REGION Network 78: ERROR - Descarga por S3
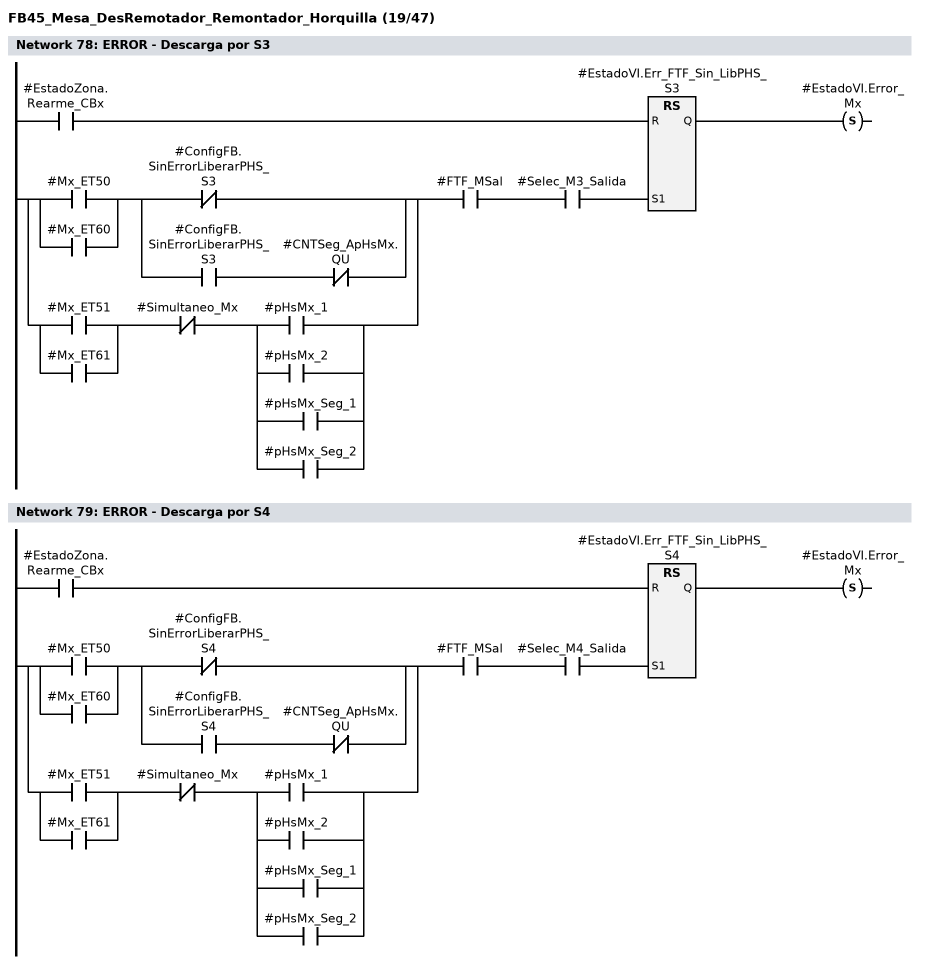
   RUNG wire#powerrail
      Contact( #EstadoZona.Rearme_CBx )
      S_RS(operand := #EstadoVI.Err_FTF_Sin_LibPHS_S3, s1 := wire#w5)
      S_Coil( #EstadoVI.Error_Mx )
   END_RUNG
   RUNG wire#powerrail
      Contact( #Mx_ET50 )
      wire#w1
      I_Contact( #ConfigFB.SinErrorLiberarPHS_S3 )
      wire#w2
      Contact( #FTF_MSal )
      Contact( #Selec_M3_Salida )
   END_RUNG wire#w5
   RUNG wire#powerrail
      Contact( #Mx_ET60 )
   END_RUNG wire#w1
   RUNG wire#w1
      Contact( #ConfigFB.SinErrorLiberarPHS_S3 )
      I_Contact( #CNTSeg_ApHsMx.QU )
   END_RUNG wire#w2
   RUNG wire#powerrail
      Contact( #Mx_ET51 )
      wire#w3
      I_Contact( #Simultaneo_Mx )
      wire#w4
      Contact( #pHsMx_1 )
   END_RUNG wire#w2
   RUNG wire#powerrail
      Contact( #Mx_ET61 )
   END_RUNG wire#w3
   RUNG wire#w4
      Contact( #pHsMx_2 )
   END_RUNG wire#w2
   RUNG wire#w4
      Contact( #pHsMx_Seg_1 )
   END_RUNG wire#w2
   RUNG wire#w4
      Contact( #pHsMx_Seg_2 )
   END_RUNG wire#w2
   // the same network as SCL:
   IF #EstadoZona.Rearme_CBx THEN
       #EstadoVI.Err_FTF_Sin_LibPHS_S3 := FALSE;   // RS flip-flop
   END_IF;
   IF (((#Mx_ET50 OR #Mx_ET60) AND (NOT #ConfigFB.SinErrorLiberarPHS_S3 OR (#ConfigFB.SinErrorLiberarPHS_S3 AND NOT #CNTSeg_ApHsMx.QU))) OR ((#Mx_ET51 OR #Mx_ET61) AND NOT #Simultaneo_Mx AND (#pHsMx_1 OR #pHsMx_2 OR #pHsMx_Seg_1 OR #pHsMx_Seg_2))) AND #FTF_MSal AND #Selec_M3_Salida THEN
       #EstadoVI.Err_FTF_Sin_LibPHS_S3 := TRUE;
   END_IF;
   IF #EstadoVI.Err_FTF_Sin_LibPHS_S3 THEN #EstadoVI.Error_Mx := TRUE; END_IF;
END_REGION

REGION Network 79: ERROR - Descarga por S4
   RUNG wire#powerrail
      Contact( #EstadoZona.Rearme_CBx )
      S_RS(operand := #EstadoVI.Err_FTF_Sin_LibPHS_S4, s1 := wire#w5)
      S_Coil( #EstadoVI.Error_Mx )
   END_RUNG
   RUNG wire#powerrail
      Contact( #Mx_ET50 )
      wire#w1
      I_Contact( #ConfigFB.SinErrorLiberarPHS_S4 )
      wire#w2
      Contact( #FTF_MSal )
      Contact( #Selec_M4_Salida )
   END_RUNG wire#w5
   RUNG wire#powerrail
      Contact( #Mx_ET60 )
   END_RUNG wire#w1
   RUNG wire#w1
      Contact( #ConfigFB.SinErrorLiberarPHS_S4 )
      I_Contact( #CNTSeg_ApHsMx.QU )
   END_RUNG wire#w2
   RUNG wire#powerrail
      Contact( #Mx_ET51 )
      wire#w3
      I_Contact( #Simultaneo_Mx )
      wire#w4
      Contact( #pHsMx_1 )
   END_RUNG wire#w2
   RUNG wire#powerrail
      Contact( #Mx_ET61 )
   END_RUNG wire#w3
   RUNG wire#w4
      Contact( #pHsMx_2 )
   END_RUNG wire#w2
   RUNG wire#w4
      Contact( #pHsMx_Seg_1 )
   END_RUNG wire#w2
   RUNG wire#w4
      Contact( #pHsMx_Seg_2 )
   END_RUNG wire#w2
   // the same network as SCL:
   IF #EstadoZona.Rearme_CBx THEN
       #EstadoVI.Err_FTF_Sin_LibPHS_S4 := FALSE;   // RS flip-flop
   END_IF;
   IF (((#Mx_ET50 OR #Mx_ET60) AND (NOT #ConfigFB.SinErrorLiberarPHS_S4 OR (#ConfigFB.SinErrorLiberarPHS_S4 AND NOT #CNTSeg_ApHsMx.QU))) OR ((#Mx_ET51 OR #Mx_ET61) AND NOT #Simultaneo_Mx AND (#pHsMx_1 OR #pHsMx_2 OR #pHsMx_Seg_1 OR #pHsMx_Seg_2))) AND #FTF_MSal AND #Selec_M4_Salida THEN
       #EstadoVI.Err_FTF_Sin_LibPHS_S4 := TRUE;
   END_IF;
   IF #EstadoVI.Err_FTF_Sin_LibPHS_S4 THEN #EstadoVI.Error_Mx := TRUE; END_IF;
END_REGION

REGION Network 80: TMP - ERROR - Tout Avance E1E3
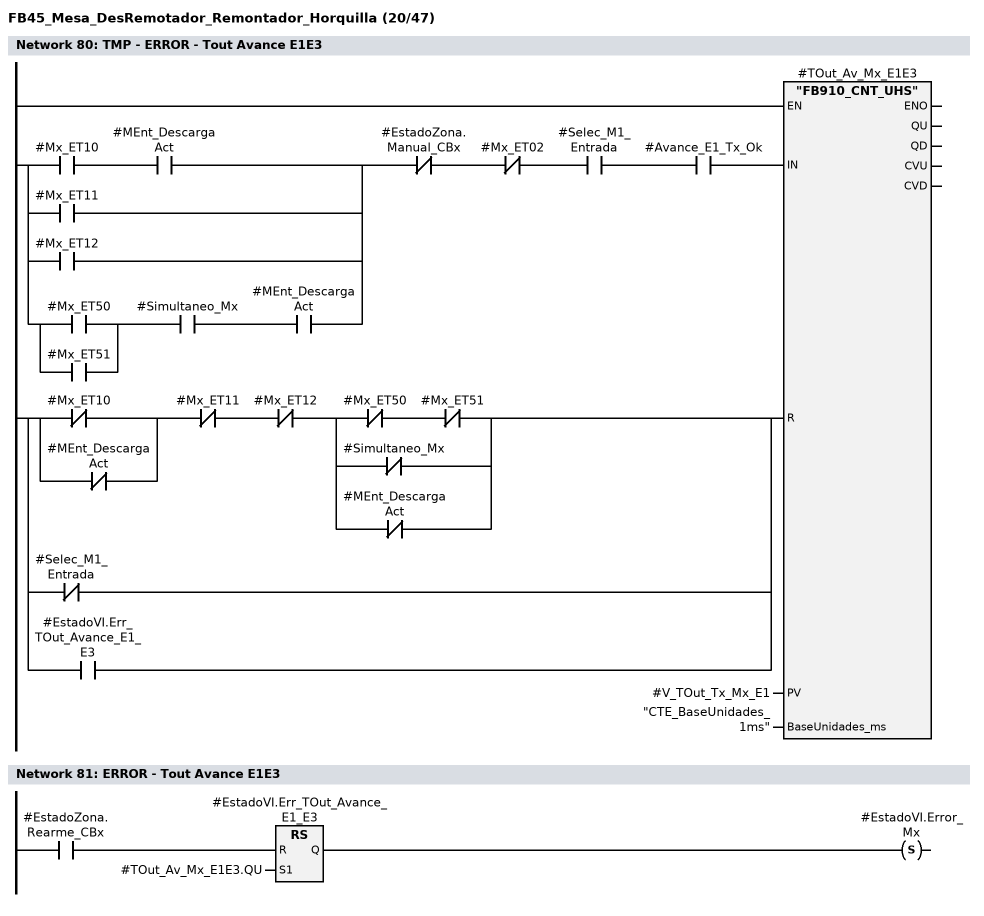
   RUNG wire#powerrail
      #TOut_Av_Mx_E1E3(IN := wire#w3, R := wire#w6, PV := #V_TOut_Tx_Mx_E1, BaseUnidades_ms := "CTE_BaseUnidades_1ms", QU =>, QD =>, CVU =>, CVD =>)
   END_RUNG
   RUNG wire#powerrail
      Contact( #Mx_ET10 )
      Contact( #MEnt_DescargaAct )
      wire#w1
      I_Contact( #EstadoZona.Manual_CBx )
      I_Contact( #Mx_ET02 )
      Contact( #Selec_M1_Entrada )
      Contact( #Avance_E1_Tx_Ok )
   END_RUNG wire#w3
   RUNG wire#powerrail
      Contact( #Mx_ET11 )
   END_RUNG wire#w1
   RUNG wire#powerrail
      Contact( #Mx_ET12 )
   END_RUNG wire#w1
   RUNG wire#powerrail
      Contact( #Mx_ET50 )
      wire#w2
      Contact( #Simultaneo_Mx )
      Contact( #MEnt_DescargaAct )
   END_RUNG wire#w1
   RUNG wire#powerrail
      Contact( #Mx_ET51 )
   END_RUNG wire#w2
   RUNG wire#powerrail
      I_Contact( #Mx_ET10 )
      wire#w4
      I_Contact( #Mx_ET11 )
      I_Contact( #Mx_ET12 )
      wire#w5
      I_Contact( #Mx_ET50 )
      I_Contact( #Mx_ET51 )
   END_RUNG wire#w6
   RUNG wire#powerrail
      I_Contact( #MEnt_DescargaAct )
   END_RUNG wire#w4
   RUNG wire#w5
      I_Contact( #Simultaneo_Mx )
   END_RUNG wire#w6
   RUNG wire#w5
      I_Contact( #MEnt_DescargaAct )
   END_RUNG wire#w6
   RUNG wire#powerrail
      I_Contact( #Selec_M1_Entrada )
   END_RUNG wire#w6
   RUNG wire#powerrail
      Contact( #EstadoVI.Err_TOut_Avance_E1_E3 )
   END_RUNG wire#w6
   // the same network as SCL:
   #TOut_Av_Mx_E1E3(IN := ((#Mx_ET10 AND #MEnt_DescargaAct) OR #Mx_ET11 OR #Mx_ET12 OR ((#Mx_ET50 OR #Mx_ET51) AND #Simultaneo_Mx AND #MEnt_DescargaAct)) AND NOT #EstadoZona.Manual_CBx AND NOT #Mx_ET02 AND #Selec_M1_Entrada AND #Avance_E1_Tx_Ok,   // "FB910_CNT_UHS"
                    R := ((NOT #Mx_ET10 OR NOT #MEnt_DescargaAct) AND NOT #Mx_ET11 AND NOT #Mx_ET12 AND ((NOT #Mx_ET50 AND NOT #Mx_ET51) OR NOT #Simultaneo_Mx OR NOT #MEnt_DescargaAct)) OR NOT #Selec_M1_Entrada OR #EstadoVI.Err_TOut_Avance_E1_E3,
                    PV := #V_TOut_Tx_Mx_E1,
                    BaseUnidades_ms := "CTE_BaseUnidades_1ms");
END_REGION

REGION Network 81: ERROR - Tout Avance E1E3
   RUNG wire#powerrail
      Contact( #EstadoZona.Rearme_CBx )
      S_RS(operand := #EstadoVI.Err_TOut_Avance_E1_E3, s1 := #TOut_Av_Mx_E1E3.QU)
      S_Coil( #EstadoVI.Error_Mx )
   END_RUNG
   // the same network as SCL:
   IF #EstadoZona.Rearme_CBx THEN
       #EstadoVI.Err_TOut_Avance_E1_E3 := FALSE;   // RS flip-flop
   END_IF;
   IF #TOut_Av_Mx_E1E3.QU THEN #EstadoVI.Err_TOut_Avance_E1_E3 := TRUE; END_IF;
   IF #EstadoVI.Err_TOut_Avance_E1_E3 THEN #EstadoVI.Error_Mx := TRUE; END_IF;
END_REGION

REGION Network 82: TMP - ERROR - Tout Retroceso E1E3
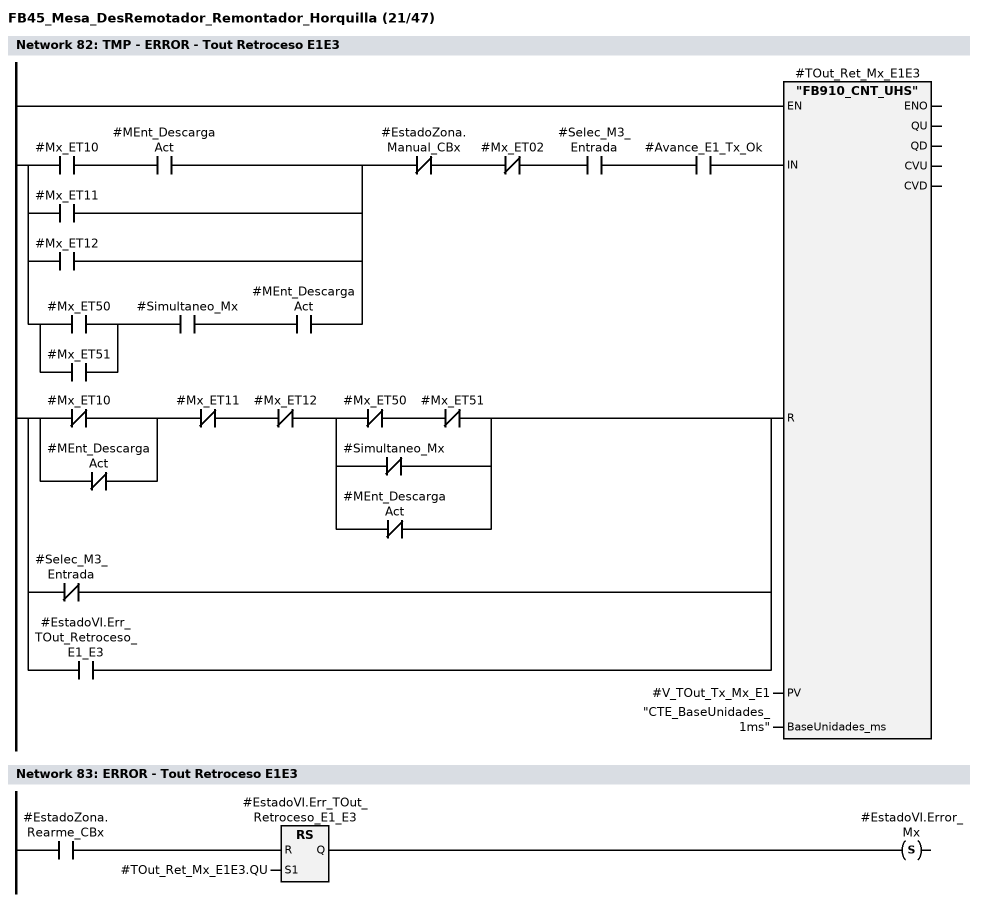
   RUNG wire#powerrail
      #TOut_Ret_Mx_E1E3(IN := wire#w3, R := wire#w6, PV := #V_TOut_Tx_Mx_E1, BaseUnidades_ms := "CTE_BaseUnidades_1ms", QU =>, QD =>, CVU =>, CVD =>)
   END_RUNG
   RUNG wire#powerrail
      Contact( #Mx_ET10 )
      Contact( #MEnt_DescargaAct )
      wire#w1
      I_Contact( #EstadoZona.Manual_CBx )
      I_Contact( #Mx_ET02 )
      Contact( #Selec_M3_Entrada )
      Contact( #Avance_E1_Tx_Ok )
   END_RUNG wire#w3
   RUNG wire#powerrail
      Contact( #Mx_ET11 )
   END_RUNG wire#w1
   RUNG wire#powerrail
      Contact( #Mx_ET12 )
   END_RUNG wire#w1
   RUNG wire#powerrail
      Contact( #Mx_ET50 )
      wire#w2
      Contact( #Simultaneo_Mx )
      Contact( #MEnt_DescargaAct )
   END_RUNG wire#w1
   RUNG wire#powerrail
      Contact( #Mx_ET51 )
   END_RUNG wire#w2
   RUNG wire#powerrail
      I_Contact( #Mx_ET10 )
      wire#w4
      I_Contact( #Mx_ET11 )
      I_Contact( #Mx_ET12 )
      wire#w5
      I_Contact( #Mx_ET50 )
      I_Contact( #Mx_ET51 )
   END_RUNG wire#w6
   RUNG wire#powerrail
      I_Contact( #MEnt_DescargaAct )
   END_RUNG wire#w4
   RUNG wire#w5
      I_Contact( #Simultaneo_Mx )
   END_RUNG wire#w6
   RUNG wire#w5
      I_Contact( #MEnt_DescargaAct )
   END_RUNG wire#w6
   RUNG wire#powerrail
      I_Contact( #Selec_M3_Entrada )
   END_RUNG wire#w6
   RUNG wire#powerrail
      Contact( #EstadoVI.Err_TOut_Retroceso_E1_E3 )
   END_RUNG wire#w6
   // the same network as SCL:
   #TOut_Ret_Mx_E1E3(IN := ((#Mx_ET10 AND #MEnt_DescargaAct) OR #Mx_ET11 OR #Mx_ET12 OR ((#Mx_ET50 OR #Mx_ET51) AND #Simultaneo_Mx AND #MEnt_DescargaAct)) AND NOT #EstadoZona.Manual_CBx AND NOT #Mx_ET02 AND #Selec_M3_Entrada AND #Avance_E1_Tx_Ok,   // "FB910_CNT_UHS"
                     R := ((NOT #Mx_ET10 OR NOT #MEnt_DescargaAct) AND NOT #Mx_ET11 AND NOT #Mx_ET12 AND ((NOT #Mx_ET50 AND NOT #Mx_ET51) OR NOT #Simultaneo_Mx OR NOT #MEnt_DescargaAct)) OR NOT #Selec_M3_Entrada OR #EstadoVI.Err_TOut_Retroceso_E1_E3,
                     PV := #V_TOut_Tx_Mx_E1,
                     BaseUnidades_ms := "CTE_BaseUnidades_1ms");
END_REGION

REGION Network 83: ERROR - Tout Retroceso E1E3
   RUNG wire#powerrail
      Contact( #EstadoZona.Rearme_CBx )
      S_RS(operand := #EstadoVI.Err_TOut_Retroceso_E1_E3, s1 := #TOut_Ret_Mx_E1E3.QU)
      S_Coil( #EstadoVI.Error_Mx )
   END_RUNG
   // the same network as SCL:
   IF #EstadoZona.Rearme_CBx THEN
       #EstadoVI.Err_TOut_Retroceso_E1_E3 := FALSE;   // RS flip-flop
   END_IF;
   IF #TOut_Ret_Mx_E1E3.QU THEN #EstadoVI.Err_TOut_Retroceso_E1_E3 := TRUE; END_IF;
   IF #EstadoVI.Err_TOut_Retroceso_E1_E3 THEN #EstadoVI.Error_Mx := TRUE; END_IF;
END_REGION

REGION Network 84: TMP - ERROR - Tout Avance E2E4
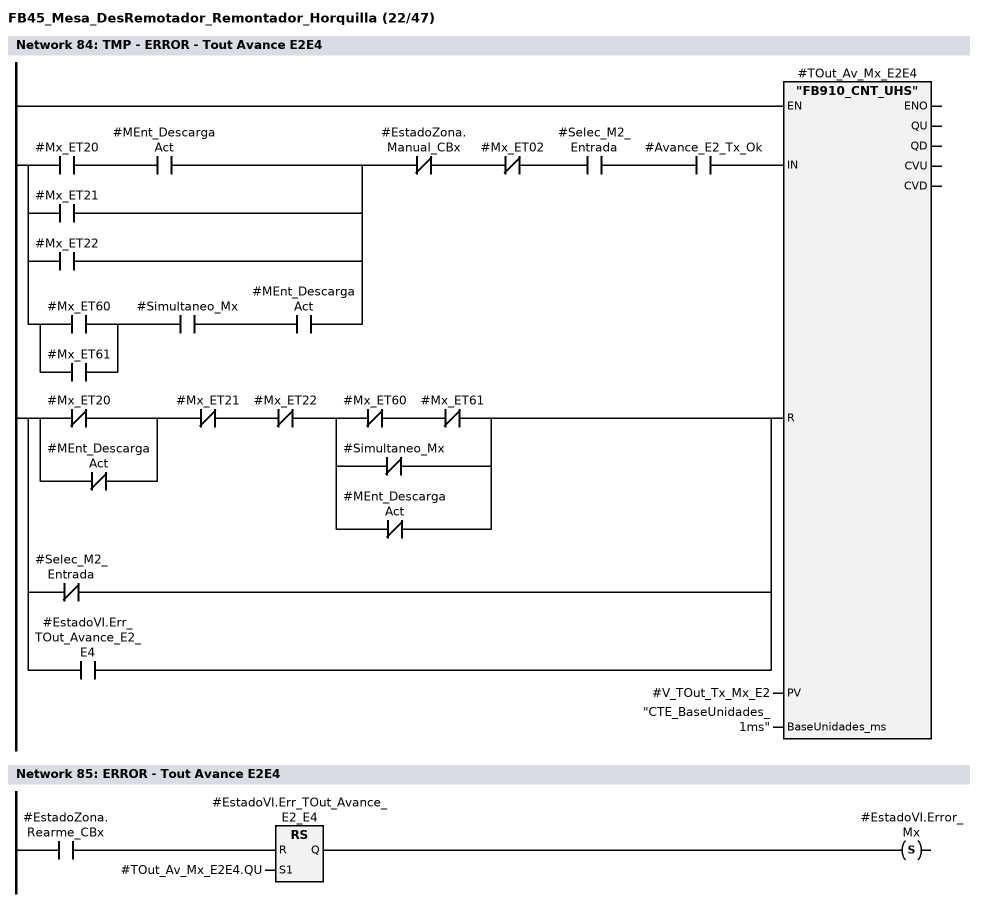
   RUNG wire#powerrail
      #TOut_Av_Mx_E2E4(IN := wire#w3, R := wire#w6, PV := #V_TOut_Tx_Mx_E2, BaseUnidades_ms := "CTE_BaseUnidades_1ms", QU =>, QD =>, CVU =>, CVD =>)
   END_RUNG
   RUNG wire#powerrail
      Contact( #Mx_ET20 )
      Contact( #MEnt_DescargaAct )
      wire#w1
      I_Contact( #EstadoZona.Manual_CBx )
      I_Contact( #Mx_ET02 )
      Contact( #Selec_M2_Entrada )
      Contact( #Avance_E2_Tx_Ok )
   END_RUNG wire#w3
   RUNG wire#powerrail
      Contact( #Mx_ET21 )
   END_RUNG wire#w1
   RUNG wire#powerrail
      Contact( #Mx_ET22 )
   END_RUNG wire#w1
   RUNG wire#powerrail
      Contact( #Mx_ET60 )
      wire#w2
      Contact( #Simultaneo_Mx )
      Contact( #MEnt_DescargaAct )
   END_RUNG wire#w1
   RUNG wire#powerrail
      Contact( #Mx_ET61 )
   END_RUNG wire#w2
   RUNG wire#powerrail
      I_Contact( #Mx_ET20 )
      wire#w4
      I_Contact( #Mx_ET21 )
      I_Contact( #Mx_ET22 )
      wire#w5
      I_Contact( #Mx_ET60 )
      I_Contact( #Mx_ET61 )
   END_RUNG wire#w6
   RUNG wire#powerrail
      I_Contact( #MEnt_DescargaAct )
   END_RUNG wire#w4
   RUNG wire#w5
      I_Contact( #Simultaneo_Mx )
   END_RUNG wire#w6
   RUNG wire#w5
      I_Contact( #MEnt_DescargaAct )
   END_RUNG wire#w6
   RUNG wire#powerrail
      I_Contact( #Selec_M2_Entrada )
   END_RUNG wire#w6
   RUNG wire#powerrail
      Contact( #EstadoVI.Err_TOut_Avance_E2_E4 )
   END_RUNG wire#w6
   // the same network as SCL:
   #TOut_Av_Mx_E2E4(IN := ((#Mx_ET20 AND #MEnt_DescargaAct) OR #Mx_ET21 OR #Mx_ET22 OR ((#Mx_ET60 OR #Mx_ET61) AND #Simultaneo_Mx AND #MEnt_DescargaAct)) AND NOT #EstadoZona.Manual_CBx AND NOT #Mx_ET02 AND #Selec_M2_Entrada AND #Avance_E2_Tx_Ok,   // "FB910_CNT_UHS"
                    R := ((NOT #Mx_ET20 OR NOT #MEnt_DescargaAct) AND NOT #Mx_ET21 AND NOT #Mx_ET22 AND ((NOT #Mx_ET60 AND NOT #Mx_ET61) OR NOT #Simultaneo_Mx OR NOT #MEnt_DescargaAct)) OR NOT #Selec_M2_Entrada OR #EstadoVI.Err_TOut_Avance_E2_E4,
                    PV := #V_TOut_Tx_Mx_E2,
                    BaseUnidades_ms := "CTE_BaseUnidades_1ms");
END_REGION

REGION Network 85: ERROR - Tout Avance E2E4
   RUNG wire#powerrail
      Contact( #EstadoZona.Rearme_CBx )
      S_RS(operand := #EstadoVI.Err_TOut_Avance_E2_E4, s1 := #TOut_Av_Mx_E2E4.QU)
      S_Coil( #EstadoVI.Error_Mx )
   END_RUNG
   // the same network as SCL:
   IF #EstadoZona.Rearme_CBx THEN
       #EstadoVI.Err_TOut_Avance_E2_E4 := FALSE;   // RS flip-flop
   END_IF;
   IF #TOut_Av_Mx_E2E4.QU THEN #EstadoVI.Err_TOut_Avance_E2_E4 := TRUE; END_IF;
   IF #EstadoVI.Err_TOut_Avance_E2_E4 THEN #EstadoVI.Error_Mx := TRUE; END_IF;
END_REGION

REGION Network 86: TMP - ERROR - Tout Retroceso E2E4
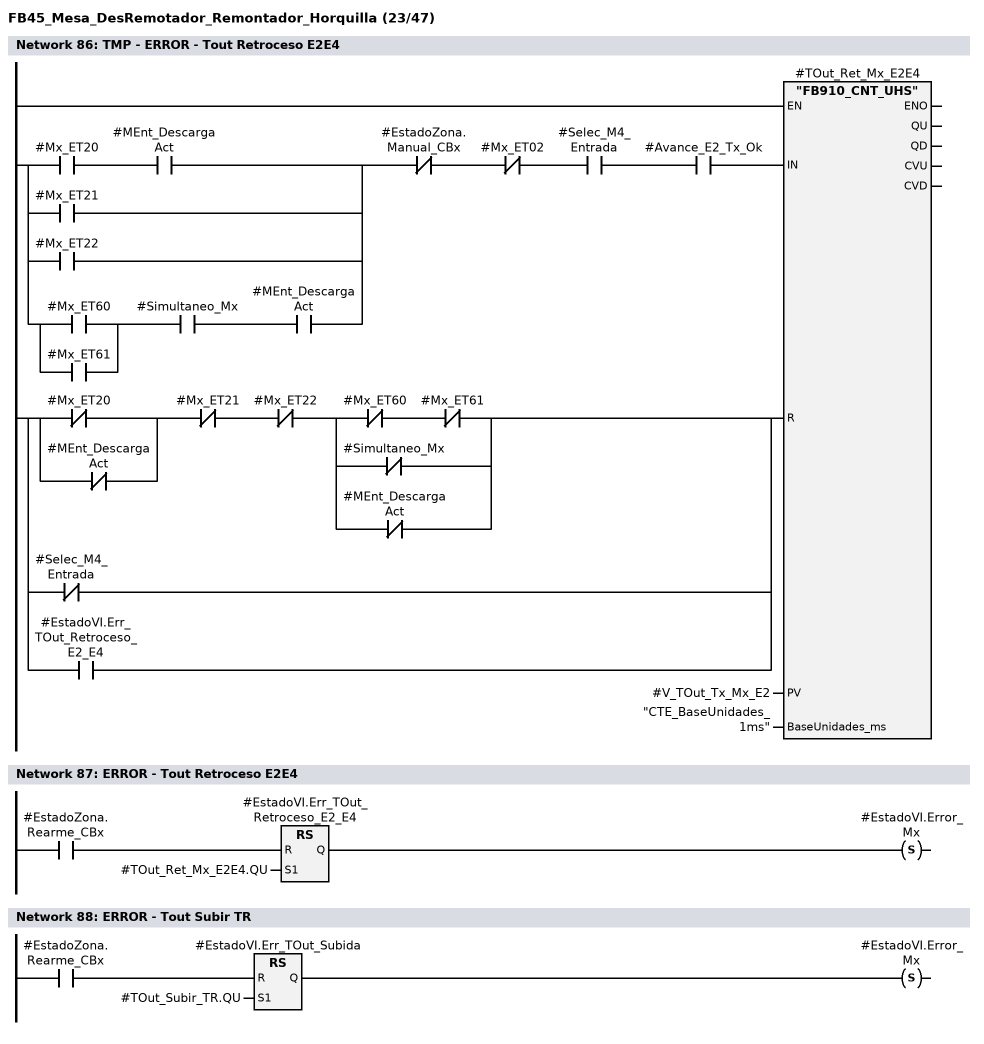
   RUNG wire#powerrail
      #TOut_Ret_Mx_E2E4(IN := wire#w3, R := wire#w6, PV := #V_TOut_Tx_Mx_E2, BaseUnidades_ms := "CTE_BaseUnidades_1ms", QU =>, QD =>, CVU =>, CVD =>)
   END_RUNG
   RUNG wire#powerrail
      Contact( #Mx_ET20 )
      Contact( #MEnt_DescargaAct )
      wire#w1
      I_Contact( #EstadoZona.Manual_CBx )
      I_Contact( #Mx_ET02 )
      Contact( #Selec_M4_Entrada )
      Contact( #Avance_E2_Tx_Ok )
   END_RUNG wire#w3
   RUNG wire#powerrail
      Contact( #Mx_ET21 )
   END_RUNG wire#w1
   RUNG wire#powerrail
      Contact( #Mx_ET22 )
   END_RUNG wire#w1
   RUNG wire#powerrail
      Contact( #Mx_ET60 )
      wire#w2
      Contact( #Simultaneo_Mx )
      Contact( #MEnt_DescargaAct )
   END_RUNG wire#w1
   RUNG wire#powerrail
      Contact( #Mx_ET61 )
   END_RUNG wire#w2
   RUNG wire#powerrail
      I_Contact( #Mx_ET20 )
      wire#w4
      I_Contact( #Mx_ET21 )
      I_Contact( #Mx_ET22 )
      wire#w5
      I_Contact( #Mx_ET60 )
      I_Contact( #Mx_ET61 )
   END_RUNG wire#w6
   RUNG wire#powerrail
      I_Contact( #MEnt_DescargaAct )
   END_RUNG wire#w4
   RUNG wire#w5
      I_Contact( #Simultaneo_Mx )
   END_RUNG wire#w6
   RUNG wire#w5
      I_Contact( #MEnt_DescargaAct )
   END_RUNG wire#w6
   RUNG wire#powerrail
      I_Contact( #Selec_M4_Entrada )
   END_RUNG wire#w6
   RUNG wire#powerrail
      Contact( #EstadoVI.Err_TOut_Retroceso_E2_E4 )
   END_RUNG wire#w6
   // the same network as SCL:
   #TOut_Ret_Mx_E2E4(IN := ((#Mx_ET20 AND #MEnt_DescargaAct) OR #Mx_ET21 OR #Mx_ET22 OR ((#Mx_ET60 OR #Mx_ET61) AND #Simultaneo_Mx AND #MEnt_DescargaAct)) AND NOT #EstadoZona.Manual_CBx AND NOT #Mx_ET02 AND #Selec_M4_Entrada AND #Avance_E2_Tx_Ok,   // "FB910_CNT_UHS"
                     R := ((NOT #Mx_ET20 OR NOT #MEnt_DescargaAct) AND NOT #Mx_ET21 AND NOT #Mx_ET22 AND ((NOT #Mx_ET60 AND NOT #Mx_ET61) OR NOT #Simultaneo_Mx OR NOT #MEnt_DescargaAct)) OR NOT #Selec_M4_Entrada OR #EstadoVI.Err_TOut_Retroceso_E2_E4,
                     PV := #V_TOut_Tx_Mx_E2,
                     BaseUnidades_ms := "CTE_BaseUnidades_1ms");
END_REGION

REGION Network 87: ERROR - Tout Retroceso E2E4
   RUNG wire#powerrail
      Contact( #EstadoZona.Rearme_CBx )
      S_RS(operand := #EstadoVI.Err_TOut_Retroceso_E2_E4, s1 := #TOut_Ret_Mx_E2E4.QU)
      S_Coil( #EstadoVI.Error_Mx )
   END_RUNG
   // the same network as SCL:
   IF #EstadoZona.Rearme_CBx THEN
       #EstadoVI.Err_TOut_Retroceso_E2_E4 := FALSE;   // RS flip-flop
   END_IF;
   IF #TOut_Ret_Mx_E2E4.QU THEN #EstadoVI.Err_TOut_Retroceso_E2_E4 := TRUE; END_IF;
   IF #EstadoVI.Err_TOut_Retroceso_E2_E4 THEN #EstadoVI.Error_Mx := TRUE; END_IF;
END_REGION

REGION Network 88: ERROR - Tout Subir TR
   RUNG wire#powerrail
      Contact( #EstadoZona.Rearme_CBx )
      S_RS(operand := #EstadoVI.Err_TOut_Subida, s1 := #TOut_Subir_TR.QU)
      S_Coil( #EstadoVI.Error_Mx )
   END_RUNG
   // the same network as SCL:
   IF #EstadoZona.Rearme_CBx THEN
       #EstadoVI.Err_TOut_Subida := FALSE;   // RS flip-flop
   END_IF;
   IF #TOut_Subir_TR.QU THEN #EstadoVI.Err_TOut_Subida := TRUE; END_IF;
   IF #EstadoVI.Err_TOut_Subida THEN #EstadoVI.Error_Mx := TRUE; END_IF;
END_REGION

REGION Network 89: TMP - ERROR - Tout Bajar Transfer
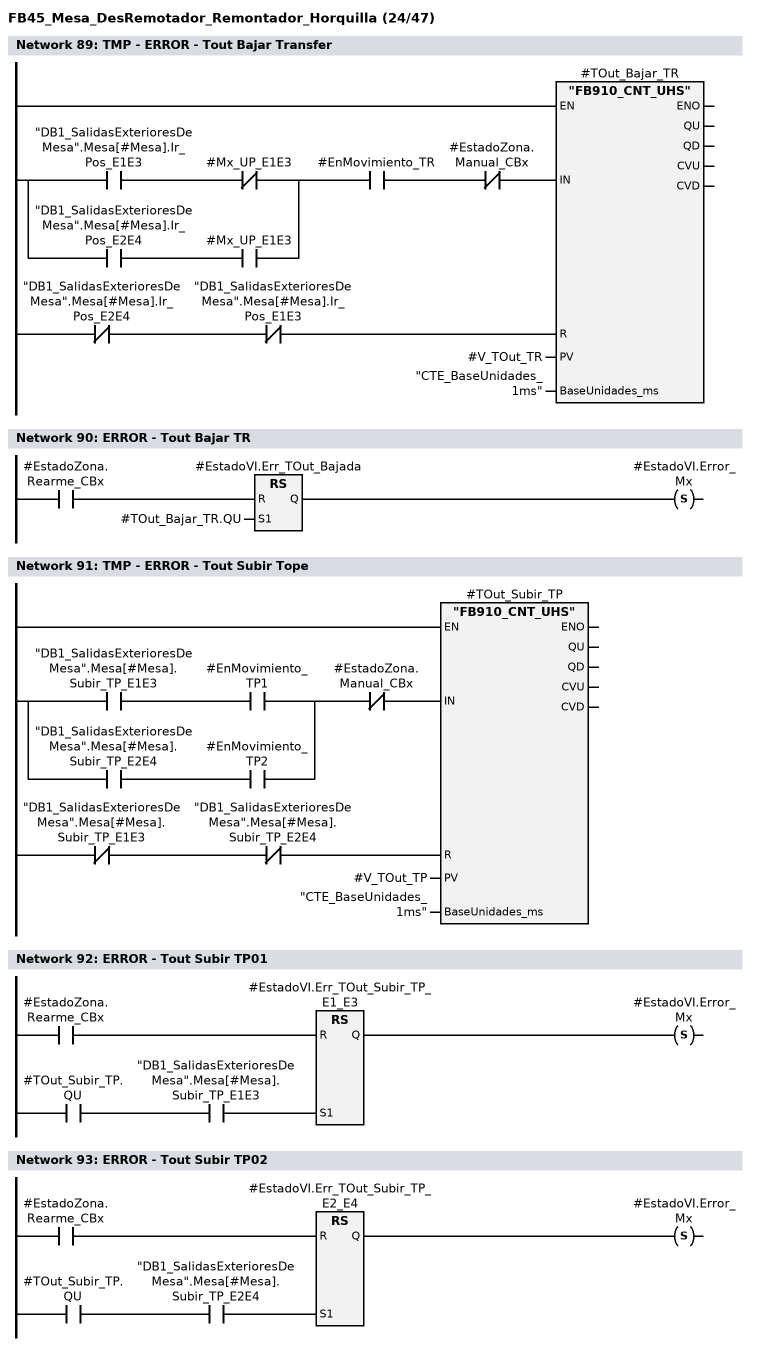
   RUNG wire#powerrail
      #TOut_Bajar_TR(IN := wire#w2, R := wire#w3, PV := #V_TOut_TR, BaseUnidades_ms := "CTE_BaseUnidades_1ms", QU =>, QD =>, CVU =>, CVD =>)
   END_RUNG
   RUNG wire#powerrail
      Contact( "DB1_SalidasExterioresDeMesa".Mesa[#Mesa].Ir_Pos_E1E3 )
      I_Contact( #Mx_UP_E1E3 )
      wire#w1
      Contact( #EnMovimiento_TR )
      I_Contact( #EstadoZona.Manual_CBx )
   END_RUNG wire#w2
   RUNG wire#powerrail
      Contact( "DB1_SalidasExterioresDeMesa".Mesa[#Mesa].Ir_Pos_E2E4 )
      Contact( #Mx_UP_E1E3 )
   END_RUNG wire#w1
   RUNG wire#powerrail
      I_Contact( "DB1_SalidasExterioresDeMesa".Mesa[#Mesa].Ir_Pos_E2E4 )
      I_Contact( "DB1_SalidasExterioresDeMesa".Mesa[#Mesa].Ir_Pos_E1E3 )
   END_RUNG wire#w3
   // the same network as SCL:
   #TOut_Bajar_TR(IN := (("DB1_SalidasExterioresDeMesa".Mesa[#Mesa].Ir_Pos_E1E3 AND NOT #Mx_UP_E1E3) OR ("DB1_SalidasExterioresDeMesa".Mesa[#Mesa].Ir_Pos_E2E4 AND #Mx_UP_E1E3)) AND #EnMovimiento_TR AND NOT #EstadoZona.Manual_CBx,   // "FB910_CNT_UHS"
                  R := NOT "DB1_SalidasExterioresDeMesa".Mesa[#Mesa].Ir_Pos_E2E4 AND NOT "DB1_SalidasExterioresDeMesa".Mesa[#Mesa].Ir_Pos_E1E3,
                  PV := #V_TOut_TR,
                  BaseUnidades_ms := "CTE_BaseUnidades_1ms");
END_REGION

REGION Network 90: ERROR - Tout Bajar TR
   RUNG wire#powerrail
      Contact( #EstadoZona.Rearme_CBx )
      S_RS(operand := #EstadoVI.Err_TOut_Bajada, s1 := #TOut_Bajar_TR.QU)
      S_Coil( #EstadoVI.Error_Mx )
   END_RUNG
   // the same network as SCL:
   IF #EstadoZona.Rearme_CBx THEN
       #EstadoVI.Err_TOut_Bajada := FALSE;   // RS flip-flop
   END_IF;
   IF #TOut_Bajar_TR.QU THEN #EstadoVI.Err_TOut_Bajada := TRUE; END_IF;
   IF #EstadoVI.Err_TOut_Bajada THEN #EstadoVI.Error_Mx := TRUE; END_IF;
END_REGION

REGION Network 91: TMP - ERROR - Tout Subir Tope
   RUNG wire#powerrail
      #TOut_Subir_TP(IN := wire#w2, R := wire#w3, PV := #V_TOut_TP, BaseUnidades_ms := "CTE_BaseUnidades_1ms", QU =>, QD =>, CVU =>, CVD =>)
   END_RUNG
   RUNG wire#powerrail
      Contact( "DB1_SalidasExterioresDeMesa".Mesa[#Mesa].Subir_TP_E1E3 )
      Contact( #EnMovimiento_TP1 )
      wire#w1
      I_Contact( #EstadoZona.Manual_CBx )
   END_RUNG wire#w2
   RUNG wire#powerrail
      Contact( "DB1_SalidasExterioresDeMesa".Mesa[#Mesa].Subir_TP_E2E4 )
      Contact( #EnMovimiento_TP2 )
   END_RUNG wire#w1
   RUNG wire#powerrail
      I_Contact( "DB1_SalidasExterioresDeMesa".Mesa[#Mesa].Subir_TP_E1E3 )
      I_Contact( "DB1_SalidasExterioresDeMesa".Mesa[#Mesa].Subir_TP_E2E4 )
   END_RUNG wire#w3
   // the same network as SCL:
   #TOut_Subir_TP(IN := (("DB1_SalidasExterioresDeMesa".Mesa[#Mesa].Subir_TP_E1E3 AND #EnMovimiento_TP1) OR ("DB1_SalidasExterioresDeMesa".Mesa[#Mesa].Subir_TP_E2E4 AND #EnMovimiento_TP2)) AND NOT #EstadoZona.Manual_CBx,   // "FB910_CNT_UHS"
                  R := NOT "DB1_SalidasExterioresDeMesa".Mesa[#Mesa].Subir_TP_E1E3 AND NOT "DB1_SalidasExterioresDeMesa".Mesa[#Mesa].Subir_TP_E2E4,
                  PV := #V_TOut_TP,
                  BaseUnidades_ms := "CTE_BaseUnidades_1ms");
END_REGION

REGION Network 92: ERROR - Tout Subir TP01
   RUNG wire#powerrail
      Contact( #EstadoZona.Rearme_CBx )
      S_RS(operand := #EstadoVI.Err_TOut_Subir_TP_E1_E3, s1 := wire#w1)
      S_Coil( #EstadoVI.Error_Mx )
   END_RUNG
   RUNG wire#powerrail
      Contact( #TOut_Subir_TP.QU )
      Contact( "DB1_SalidasExterioresDeMesa".Mesa[#Mesa].Subir_TP_E1E3 )
   END_RUNG wire#w1
   // the same network as SCL:
   IF #EstadoZona.Rearme_CBx THEN
       #EstadoVI.Err_TOut_Subir_TP_E1_E3 := FALSE;   // RS flip-flop
   END_IF;
   IF #TOut_Subir_TP.QU AND "DB1_SalidasExterioresDeMesa".Mesa[#Mesa].Subir_TP_E1E3 THEN
       #EstadoVI.Err_TOut_Subir_TP_E1_E3 := TRUE;
   END_IF;
   IF #EstadoVI.Err_TOut_Subir_TP_E1_E3 THEN #EstadoVI.Error_Mx := TRUE; END_IF;
END_REGION

REGION Network 93: ERROR - Tout Subir TP02
   RUNG wire#powerrail
      Contact( #EstadoZona.Rearme_CBx )
      S_RS(operand := #EstadoVI.Err_TOut_Subir_TP_E2_E4, s1 := wire#w1)
      S_Coil( #EstadoVI.Error_Mx )
   END_RUNG
   RUNG wire#powerrail
      Contact( #TOut_Subir_TP.QU )
      Contact( "DB1_SalidasExterioresDeMesa".Mesa[#Mesa].Subir_TP_E2E4 )
   END_RUNG wire#w1
   // the same network as SCL:
   IF #EstadoZona.Rearme_CBx THEN
       #EstadoVI.Err_TOut_Subir_TP_E2_E4 := FALSE;   // RS flip-flop
   END_IF;
   IF #TOut_Subir_TP.QU AND "DB1_SalidasExterioresDeMesa".Mesa[#Mesa].Subir_TP_E2E4 THEN
       #EstadoVI.Err_TOut_Subir_TP_E2_E4 := TRUE;
   END_IF;
   IF #EstadoVI.Err_TOut_Subir_TP_E2_E4 THEN #EstadoVI.Error_Mx := TRUE; END_IF;
END_REGION

REGION Network 94: TMP - ERROR - Tout Bajar Tope
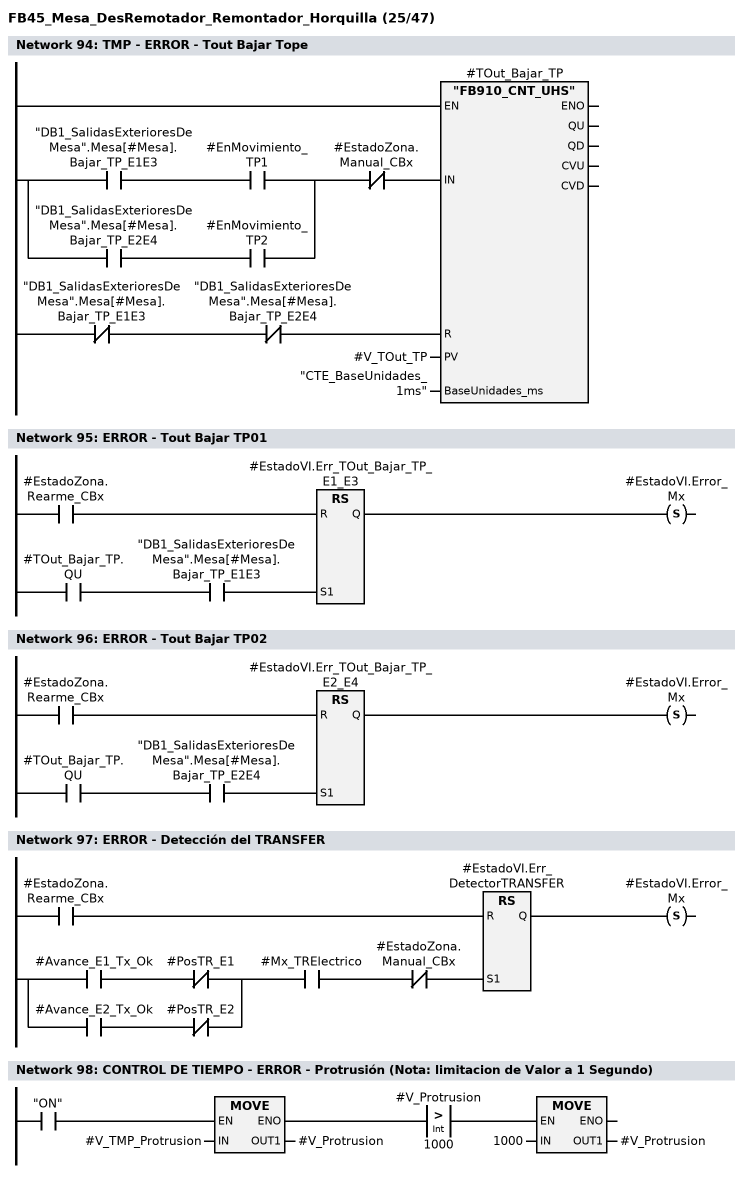
   RUNG wire#powerrail
      #TOut_Bajar_TP(IN := wire#w2, R := wire#w3, PV := #V_TOut_TP, BaseUnidades_ms := "CTE_BaseUnidades_1ms", QU =>, QD =>, CVU =>, CVD =>)
   END_RUNG
   RUNG wire#powerrail
      Contact( "DB1_SalidasExterioresDeMesa".Mesa[#Mesa].Bajar_TP_E1E3 )
      Contact( #EnMovimiento_TP1 )
      wire#w1
      I_Contact( #EstadoZona.Manual_CBx )
   END_RUNG wire#w2
   RUNG wire#powerrail
      Contact( "DB1_SalidasExterioresDeMesa".Mesa[#Mesa].Bajar_TP_E2E4 )
      Contact( #EnMovimiento_TP2 )
   END_RUNG wire#w1
   RUNG wire#powerrail
      I_Contact( "DB1_SalidasExterioresDeMesa".Mesa[#Mesa].Bajar_TP_E1E3 )
      I_Contact( "DB1_SalidasExterioresDeMesa".Mesa[#Mesa].Bajar_TP_E2E4 )
   END_RUNG wire#w3
   // the same network as SCL:
   #TOut_Bajar_TP(IN := (("DB1_SalidasExterioresDeMesa".Mesa[#Mesa].Bajar_TP_E1E3 AND #EnMovimiento_TP1) OR ("DB1_SalidasExterioresDeMesa".Mesa[#Mesa].Bajar_TP_E2E4 AND #EnMovimiento_TP2)) AND NOT #EstadoZona.Manual_CBx,   // "FB910_CNT_UHS"
                  R := NOT "DB1_SalidasExterioresDeMesa".Mesa[#Mesa].Bajar_TP_E1E3 AND NOT "DB1_SalidasExterioresDeMesa".Mesa[#Mesa].Bajar_TP_E2E4,
                  PV := #V_TOut_TP,
                  BaseUnidades_ms := "CTE_BaseUnidades_1ms");
END_REGION

REGION Network 95: ERROR - Tout Bajar TP01
   RUNG wire#powerrail
      Contact( #EstadoZona.Rearme_CBx )
      S_RS(operand := #EstadoVI.Err_TOut_Bajar_TP_E1_E3, s1 := wire#w1)
      S_Coil( #EstadoVI.Error_Mx )
   END_RUNG
   RUNG wire#powerrail
      Contact( #TOut_Bajar_TP.QU )
      Contact( "DB1_SalidasExterioresDeMesa".Mesa[#Mesa].Bajar_TP_E1E3 )
   END_RUNG wire#w1
   // the same network as SCL:
   IF #EstadoZona.Rearme_CBx THEN
       #EstadoVI.Err_TOut_Bajar_TP_E1_E3 := FALSE;   // RS flip-flop
   END_IF;
   IF #TOut_Bajar_TP.QU AND "DB1_SalidasExterioresDeMesa".Mesa[#Mesa].Bajar_TP_E1E3 THEN
       #EstadoVI.Err_TOut_Bajar_TP_E1_E3 := TRUE;
   END_IF;
   IF #EstadoVI.Err_TOut_Bajar_TP_E1_E3 THEN #EstadoVI.Error_Mx := TRUE; END_IF;
END_REGION

REGION Network 96: ERROR - Tout Bajar TP02
   RUNG wire#powerrail
      Contact( #EstadoZona.Rearme_CBx )
      S_RS(operand := #EstadoVI.Err_TOut_Bajar_TP_E2_E4, s1 := wire#w1)
      S_Coil( #EstadoVI.Error_Mx )
   END_RUNG
   RUNG wire#powerrail
      Contact( #TOut_Bajar_TP.QU )
      Contact( "DB1_SalidasExterioresDeMesa".Mesa[#Mesa].Bajar_TP_E2E4 )
   END_RUNG wire#w1
   // the same network as SCL:
   IF #EstadoZona.Rearme_CBx THEN
       #EstadoVI.Err_TOut_Bajar_TP_E2_E4 := FALSE;   // RS flip-flop
   END_IF;
   IF #TOut_Bajar_TP.QU AND "DB1_SalidasExterioresDeMesa".Mesa[#Mesa].Bajar_TP_E2E4 THEN
       #EstadoVI.Err_TOut_Bajar_TP_E2_E4 := TRUE;
   END_IF;
   IF #EstadoVI.Err_TOut_Bajar_TP_E2_E4 THEN #EstadoVI.Error_Mx := TRUE; END_IF;
END_REGION

REGION Network 97: ERROR - Detección del TRANSFER
   RUNG wire#powerrail
      Contact( #EstadoZona.Rearme_CBx )
      S_RS(operand := #EstadoVI.Err_DetectorTRANSFER, s1 := wire#w2)
      S_Coil( #EstadoVI.Error_Mx )
   END_RUNG
   RUNG wire#powerrail
      Contact( #Avance_E1_Tx_Ok )
      I_Contact( #PosTR_E1 )
      wire#w1
      Contact( #Mx_TRElectrico )
      I_Contact( #EstadoZona.Manual_CBx )
   END_RUNG wire#w2
   RUNG wire#powerrail
      Contact( #Avance_E2_Tx_Ok )
      I_Contact( #PosTR_E2 )
   END_RUNG wire#w1
   // the same network as SCL:
   IF #EstadoZona.Rearme_CBx THEN
       #EstadoVI.Err_DetectorTRANSFER := FALSE;   // RS flip-flop
   END_IF;
   IF ((#Avance_E1_Tx_Ok AND NOT #PosTR_E1) OR (#Avance_E2_Tx_Ok AND NOT #PosTR_E2)) AND #Mx_TRElectrico AND NOT #EstadoZona.Manual_CBx THEN
       #EstadoVI.Err_DetectorTRANSFER := TRUE;
   END_IF;
   IF #EstadoVI.Err_DetectorTRANSFER THEN #EstadoVI.Error_Mx := TRUE; END_IF;
END_REGION

REGION Network 98: CONTROL DE TIEMPO - ERROR - Protrusión (Nota: limitacion de Valor a 1 Segundo)
   RUNG wire#powerrail
      Contact( "ON" )
      Move(in := #V_TMP_Protrusion, out1 => #V_Protrusion)
      { S7_Templates := "SrcType := Int" } GT_Contact(in1 := #V_Protrusion, in2 := 1000)
      Move(in := 1000, out1 => #V_Protrusion)
   END_RUNG
   // the same network as SCL:
   IF "ON" THEN #V_Protrusion := #V_TMP_Protrusion; END_IF;
   IF "ON" AND (#V_Protrusion > 1000) THEN #V_Protrusion := 1000; END_IF;
END_REGION

REGION Network 99: TMP - ERROR - Protrusión
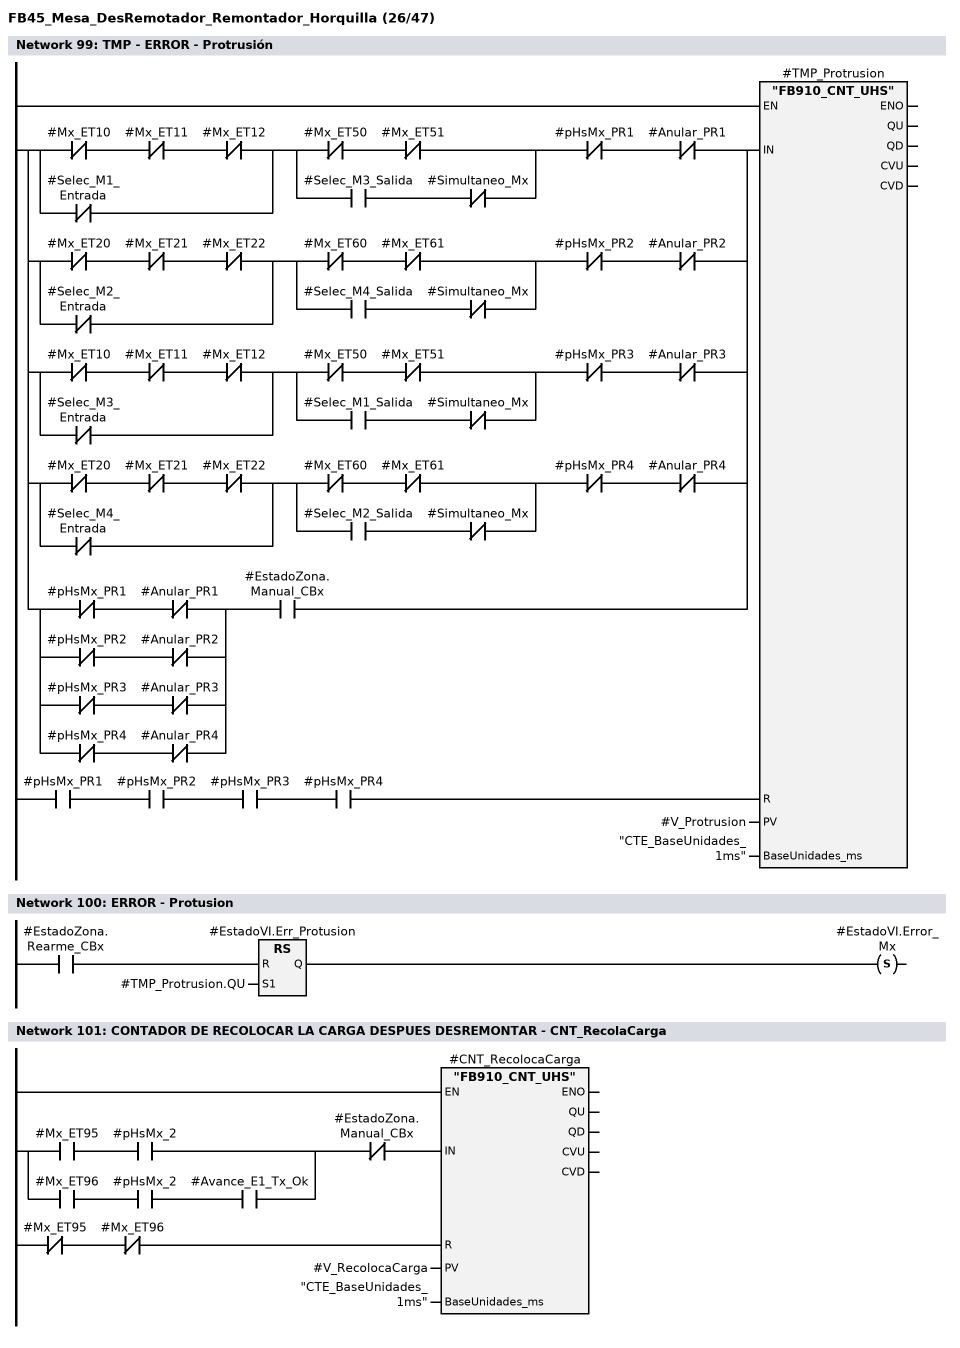
   RUNG wire#powerrail
      #TMP_Protrusion(IN := wire#w10, R := wire#w11, PV := #V_Protrusion, BaseUnidades_ms := "CTE_BaseUnidades_1ms", QU =>, QD =>, CVU =>, CVD =>)
   END_RUNG
   RUNG wire#powerrail
      I_Contact( #Mx_ET10 )
      I_Contact( #Mx_ET11 )
      I_Contact( #Mx_ET12 )
      wire#w1
      I_Contact( #Mx_ET50 )
      I_Contact( #Mx_ET51 )
      wire#w2
      I_Contact( #pHsMx_PR1 )
      I_Contact( #Anular_PR1 )
   END_RUNG wire#w10
   RUNG wire#powerrail
      I_Contact( #Selec_M1_Entrada )
   END_RUNG wire#w1
   RUNG wire#w1
      Contact( #Selec_M3_Salida )
      I_Contact( #Simultaneo_Mx )
   END_RUNG wire#w2
   RUNG wire#powerrail
      I_Contact( #Mx_ET20 )
      I_Contact( #Mx_ET21 )
      I_Contact( #Mx_ET22 )
      wire#w3
      I_Contact( #Mx_ET60 )
      I_Contact( #Mx_ET61 )
      wire#w4
      I_Contact( #pHsMx_PR2 )
      I_Contact( #Anular_PR2 )
   END_RUNG wire#w10
   RUNG wire#powerrail
      I_Contact( #Selec_M2_Entrada )
   END_RUNG wire#w3
   RUNG wire#w3
      Contact( #Selec_M4_Salida )
      I_Contact( #Simultaneo_Mx )
   END_RUNG wire#w4
   RUNG wire#powerrail
      I_Contact( #Mx_ET10 )
      I_Contact( #Mx_ET11 )
      I_Contact( #Mx_ET12 )
      wire#w5
      I_Contact( #Mx_ET50 )
      I_Contact( #Mx_ET51 )
      wire#w6
      I_Contact( #pHsMx_PR3 )
      I_Contact( #Anular_PR3 )
   END_RUNG wire#w10
   RUNG wire#powerrail
      I_Contact( #Selec_M3_Entrada )
   END_RUNG wire#w5
   RUNG wire#w5
      Contact( #Selec_M1_Salida )
      I_Contact( #Simultaneo_Mx )
   END_RUNG wire#w6
   RUNG wire#powerrail
      I_Contact( #Mx_ET20 )
      I_Contact( #Mx_ET21 )
      I_Contact( #Mx_ET22 )
      wire#w7
      I_Contact( #Mx_ET60 )
      I_Contact( #Mx_ET61 )
      wire#w8
      I_Contact( #pHsMx_PR4 )
      I_Contact( #Anular_PR4 )
   END_RUNG wire#w10
   RUNG wire#powerrail
      I_Contact( #Selec_M4_Entrada )
   END_RUNG wire#w7
   RUNG wire#w7
      Contact( #Selec_M2_Salida )
      I_Contact( #Simultaneo_Mx )
   END_RUNG wire#w8
   RUNG wire#powerrail
      I_Contact( #pHsMx_PR1 )
      I_Contact( #Anular_PR1 )
      wire#w9
      Contact( #EstadoZona.Manual_CBx )
   END_RUNG wire#w10
   RUNG wire#powerrail
      I_Contact( #pHsMx_PR2 )
      I_Contact( #Anular_PR2 )
   END_RUNG wire#w9
   RUNG wire#powerrail
      I_Contact( #pHsMx_PR3 )
      I_Contact( #Anular_PR3 )
   END_RUNG wire#w9
   RUNG wire#powerrail
      I_Contact( #pHsMx_PR4 )
      I_Contact( #Anular_PR4 )
   END_RUNG wire#w9
   RUNG wire#powerrail
      Contact( #pHsMx_PR1 )
      Contact( #pHsMx_PR2 )
      Contact( #pHsMx_PR3 )
      Contact( #pHsMx_PR4 )
   END_RUNG wire#w11
   // the same network as SCL:
   #TMP_Protrusion(IN := (((NOT #Mx_ET10 AND NOT #Mx_ET11 AND NOT #Mx_ET12) OR NOT #Selec_M1_Entrada) AND ((NOT #Mx_ET50 AND NOT #Mx_ET51) OR (#Selec_M3_Salida AND NOT #Simultaneo_Mx)) AND NOT #pHsMx_PR1 AND NOT #Anular_PR1) OR (((NOT #Mx_ET20 AND NOT #Mx_ET21 AND NOT #Mx_ET22) OR NOT #Selec_M2_Entrada) AND ((NOT #Mx_ET60 AND NOT #Mx_ET61) OR (#Selec_M4_Salida AND NOT #Simultaneo_Mx)) AND NOT #pHsMx_PR2 AND NOT #Anular_PR2) OR (((NOT #Mx_ET10 AND NOT #Mx_ET11 AND NOT #Mx_ET12) OR NOT #Selec_M3_Entrada) AND ((NOT #Mx_ET50 AND NOT #Mx_ET51) OR (#Selec_M1_Salida AND NOT #Simultaneo_Mx)) AND NOT #pHsMx_PR3 AND NOT #Anular_PR3) OR (((NOT #Mx_ET20 AND NOT #Mx_ET21 AND NOT #Mx_ET22) OR NOT #Selec_M4_Entrada) AND ((NOT #Mx_ET60 AND NOT #Mx_ET61) OR (#Selec_M2_Salida AND NOT #Simultaneo_Mx)) AND NOT #pHsMx_PR4 AND NOT #Anular_PR4) OR (((NOT #pHsMx_PR1 AND NOT #Anular_PR1) OR (NOT #pHsMx_PR2 AND NOT #Anular_PR2) OR (NOT #pHsMx_PR3 AND NOT #Anular_PR3) OR (NOT #pHsMx_PR4 AND NOT #Anular_PR4)) AND #EstadoZona.Manual_CBx),   // "FB910_CNT_UHS"
                   R := #pHsMx_PR1 AND #pHsMx_PR2 AND #pHsMx_PR3 AND #pHsMx_PR4,
                   PV := #V_Protrusion,
                   BaseUnidades_ms := "CTE_BaseUnidades_1ms");
END_REGION

REGION Network 100: ERROR - Protusion
   RUNG wire#powerrail
      Contact( #EstadoZona.Rearme_CBx )
      S_RS(operand := #EstadoVI.Err_Protusion, s1 := #TMP_Protrusion.QU)
      S_Coil( #EstadoVI.Error_Mx )
   END_RUNG
   // the same network as SCL:
   IF #EstadoZona.Rearme_CBx THEN
       #EstadoVI.Err_Protusion := FALSE;   // RS flip-flop
   END_IF;
   IF #TMP_Protrusion.QU THEN #EstadoVI.Err_Protusion := TRUE; END_IF;
   IF #EstadoVI.Err_Protusion THEN #EstadoVI.Error_Mx := TRUE; END_IF;
END_REGION

REGION Network 101: CONTADOR DE RECOLOCAR LA CARGA DESPUES DESREMONTAR - CNT_RecolaCarga
   RUNG wire#powerrail
      #CNT_RecolocaCarga(IN := wire#w2, R := wire#w3, PV := #V_RecolocaCarga, BaseUnidades_ms := "CTE_BaseUnidades_1ms", QU =>, QD =>, CVU =>, CVD =>)
   END_RUNG
   RUNG wire#powerrail
      Contact( #Mx_ET95 )
      Contact( #pHsMx_2 )
      wire#w1
      I_Contact( #EstadoZona.Manual_CBx )
   END_RUNG wire#w2
   RUNG wire#powerrail
      Contact( #Mx_ET96 )
      Contact( #pHsMx_2 )
      Contact( #Avance_E1_Tx_Ok )
   END_RUNG wire#w1
   RUNG wire#powerrail
      I_Contact( #Mx_ET95 )
      I_Contact( #Mx_ET96 )
   END_RUNG wire#w3
   // the same network as SCL:
   #CNT_RecolocaCarga(IN := ((#Mx_ET95 AND #pHsMx_2) OR (#Mx_ET96 AND #pHsMx_2 AND #Avance_E1_Tx_Ok)) AND NOT #EstadoZona.Manual_CBx,   // "FB910_CNT_UHS"
                      R := NOT #Mx_ET95 AND NOT #Mx_ET96,
                      PV := #V_RecolocaCarga,
                      BaseUnidades_ms := "CTE_BaseUnidades_1ms");
END_REGION

REGION Network 102: CONTADOR DE AUSENCIA DE LA "pHsSeg" DE CNTSeg - CNTApHs_CNTSeg_E1E3
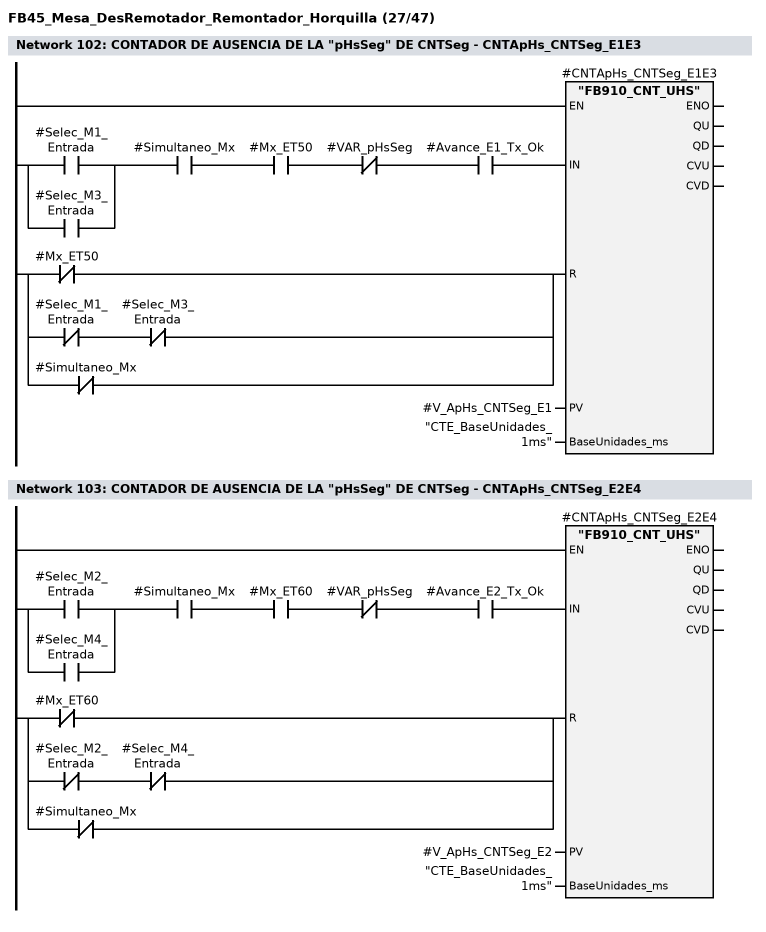
   RUNG wire#powerrail
      #CNTApHs_CNTSeg_E1E3(IN := wire#w2, R := wire#w3, PV := #V_ApHs_CNTSeg_E1, BaseUnidades_ms := "CTE_BaseUnidades_1ms", QU =>, QD =>, CVU =>, CVD =>)
   END_RUNG
   RUNG wire#powerrail
      Contact( #Selec_M1_Entrada )
      wire#w1
      Contact( #Simultaneo_Mx )
      Contact( #Mx_ET50 )
      I_Contact( #VAR_pHsSeg )
      Contact( #Avance_E1_Tx_Ok )
   END_RUNG wire#w2
   RUNG wire#powerrail
      Contact( #Selec_M3_Entrada )
   END_RUNG wire#w1
   RUNG wire#powerrail
      I_Contact( #Mx_ET50 )
   END_RUNG wire#w3
   RUNG wire#powerrail
      I_Contact( #Selec_M1_Entrada )
      I_Contact( #Selec_M3_Entrada )
   END_RUNG wire#w3
   RUNG wire#powerrail
      I_Contact( #Simultaneo_Mx )
   END_RUNG wire#w3
   // the same network as SCL:
   #CNTApHs_CNTSeg_E1E3(IN := (#Selec_M1_Entrada OR #Selec_M3_Entrada) AND #Simultaneo_Mx AND #Mx_ET50 AND NOT #VAR_pHsSeg AND #Avance_E1_Tx_Ok,   // "FB910_CNT_UHS"
                        R := NOT #Mx_ET50 OR (NOT #Selec_M1_Entrada AND NOT #Selec_M3_Entrada) OR NOT #Simultaneo_Mx,
                        PV := #V_ApHs_CNTSeg_E1,
                        BaseUnidades_ms := "CTE_BaseUnidades_1ms");
END_REGION

REGION Network 103: CONTADOR DE AUSENCIA DE LA "pHsSeg" DE CNTSeg - CNTApHs_CNTSeg_E2E4
   RUNG wire#powerrail
      #CNTApHs_CNTSeg_E2E4(IN := wire#w2, R := wire#w3, PV := #V_ApHs_CNTSeg_E2, BaseUnidades_ms := "CTE_BaseUnidades_1ms", QU =>, QD =>, CVU =>, CVD =>)
   END_RUNG
   RUNG wire#powerrail
      Contact( #Selec_M2_Entrada )
      wire#w1
      Contact( #Simultaneo_Mx )
      Contact( #Mx_ET60 )
      I_Contact( #VAR_pHsSeg )
      Contact( #Avance_E2_Tx_Ok )
   END_RUNG wire#w2
   RUNG wire#powerrail
      Contact( #Selec_M4_Entrada )
   END_RUNG wire#w1
   RUNG wire#powerrail
      I_Contact( #Mx_ET60 )
   END_RUNG wire#w3
   RUNG wire#powerrail
      I_Contact( #Selec_M2_Entrada )
      I_Contact( #Selec_M4_Entrada )
   END_RUNG wire#w3
   RUNG wire#powerrail
      I_Contact( #Simultaneo_Mx )
   END_RUNG wire#w3
   // the same network as SCL:
   #CNTApHs_CNTSeg_E2E4(IN := (#Selec_M2_Entrada OR #Selec_M4_Entrada) AND #Simultaneo_Mx AND #Mx_ET60 AND NOT #VAR_pHsSeg AND #Avance_E2_Tx_Ok,   // "FB910_CNT_UHS"
                        R := NOT #Mx_ET60 OR (NOT #Selec_M2_Entrada AND NOT #Selec_M4_Entrada) OR NOT #Simultaneo_Mx,
                        PV := #V_ApHs_CNTSeg_E2,
                        BaseUnidades_ms := "CTE_BaseUnidades_1ms");
END_REGION

REGION Network 104: CONTADOR DE SEGURIDAD DE PRESENCIA - CNTSeg_pHsMx_E1E3
   // VAR_pHsSeg ---> Inicio del CNT de Seguridad (Ha funcionar) ---- NOTA : Diferente con FB264
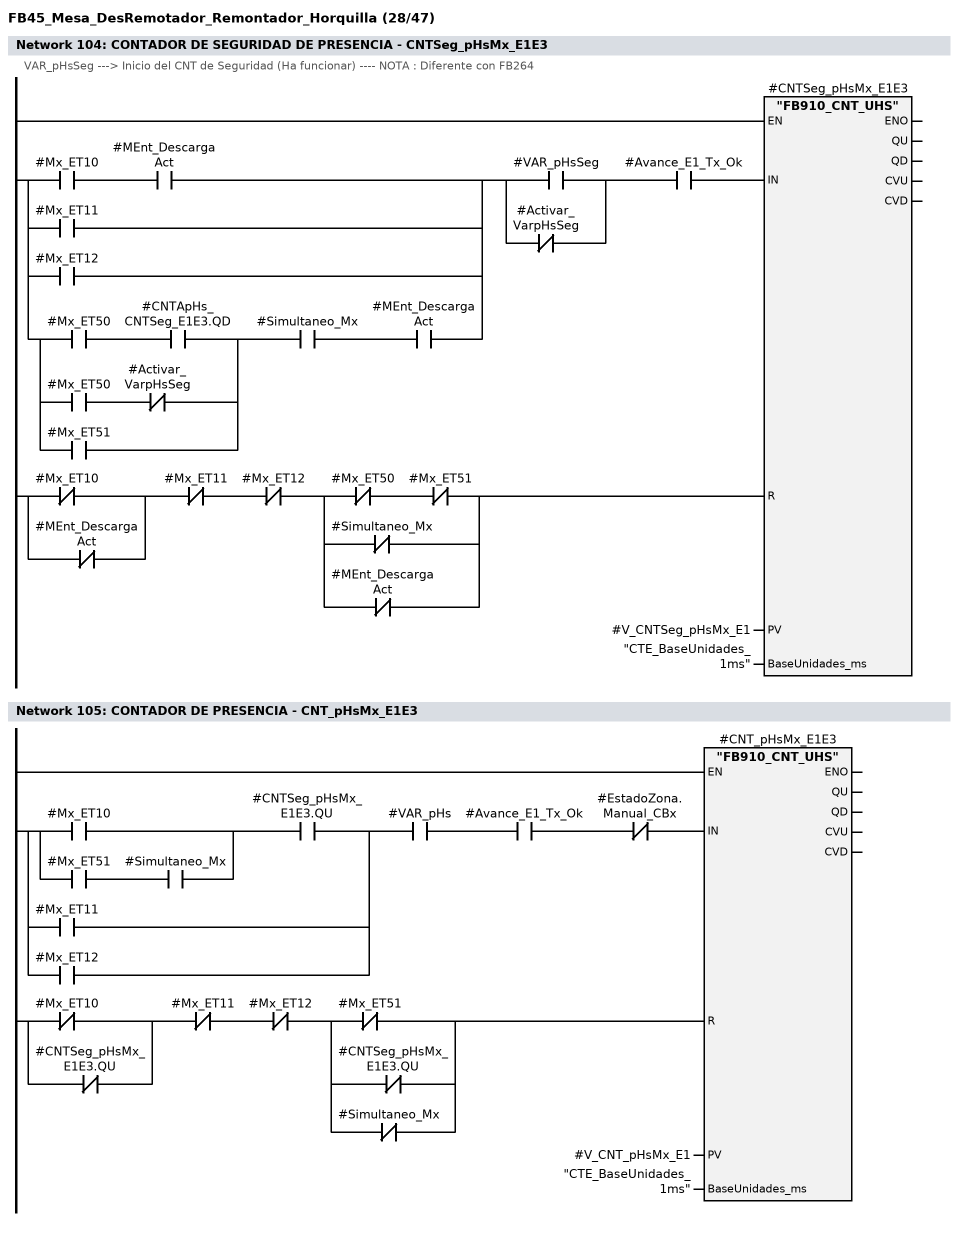
   RUNG wire#powerrail
      #CNTSeg_pHsMx_E1E3(IN := wire#w4, R := wire#w7, PV := #V_CNTSeg_pHsMx_E1, BaseUnidades_ms := "CTE_BaseUnidades_1ms", QU =>, QD =>, CVU =>, CVD =>)
   END_RUNG
   RUNG wire#powerrail
      Contact( #Mx_ET10 )
      Contact( #MEnt_DescargaAct )
      wire#w1
      Contact( #VAR_pHsSeg )
      wire#w3
      Contact( #Avance_E1_Tx_Ok )
   END_RUNG wire#w4
   RUNG wire#powerrail
      Contact( #Mx_ET11 )
   END_RUNG wire#w1
   RUNG wire#powerrail
      Contact( #Mx_ET12 )
   END_RUNG wire#w1
   RUNG wire#powerrail
      Contact( #Mx_ET50 )
      Contact( #CNTApHs_CNTSeg_E1E3.QD )
      wire#w2
      Contact( #Simultaneo_Mx )
      Contact( #MEnt_DescargaAct )
   END_RUNG wire#w1
   RUNG wire#powerrail
      Contact( #Mx_ET50 )
      I_Contact( #Activar_VarpHsSeg )
   END_RUNG wire#w2
   RUNG wire#powerrail
      Contact( #Mx_ET51 )
   END_RUNG wire#w2
   RUNG wire#w1
      I_Contact( #Activar_VarpHsSeg )
   END_RUNG wire#w3
   RUNG wire#powerrail
      I_Contact( #Mx_ET10 )
      wire#w5
      I_Contact( #Mx_ET11 )
      I_Contact( #Mx_ET12 )
      wire#w6
      I_Contact( #Mx_ET50 )
      I_Contact( #Mx_ET51 )
   END_RUNG wire#w7
   RUNG wire#powerrail
      I_Contact( #MEnt_DescargaAct )
   END_RUNG wire#w5
   RUNG wire#w6
      I_Contact( #Simultaneo_Mx )
   END_RUNG wire#w7
   RUNG wire#w6
      I_Contact( #MEnt_DescargaAct )
   END_RUNG wire#w7
   // the same network as SCL:
   #CNTSeg_pHsMx_E1E3(IN := ((#Mx_ET10 AND #MEnt_DescargaAct) OR #Mx_ET11 OR #Mx_ET12 OR (((#Mx_ET50 AND #CNTApHs_CNTSeg_E1E3.QD) OR (#Mx_ET50 AND NOT #Activar_VarpHsSeg) OR #Mx_ET51) AND #Simultaneo_Mx AND #MEnt_DescargaAct)) AND (#VAR_pHsSeg OR NOT #Activar_VarpHsSeg) AND #Avance_E1_Tx_Ok,   // "FB910_CNT_UHS"
                      R := (NOT #Mx_ET10 OR NOT #MEnt_DescargaAct) AND NOT #Mx_ET11 AND NOT #Mx_ET12 AND ((NOT #Mx_ET50 AND NOT #Mx_ET51) OR NOT #Simultaneo_Mx OR NOT #MEnt_DescargaAct),
                      PV := #V_CNTSeg_pHsMx_E1,
                      BaseUnidades_ms := "CTE_BaseUnidades_1ms");
END_REGION

REGION Network 105: CONTADOR DE PRESENCIA - CNT_pHsMx_E1E3
   RUNG wire#powerrail
      #CNT_pHsMx_E1E3(IN := wire#w3, R := wire#w6, PV := #V_CNT_pHsMx_E1, BaseUnidades_ms := "CTE_BaseUnidades_1ms", QU =>, QD =>, CVU =>, CVD =>)
   END_RUNG
   RUNG wire#powerrail
      Contact( #Mx_ET10 )
      wire#w1
      Contact( #CNTSeg_pHsMx_E1E3.QU )
      wire#w2
      Contact( #VAR_pHs )
      Contact( #Avance_E1_Tx_Ok )
      I_Contact( #EstadoZona.Manual_CBx )
   END_RUNG wire#w3
   RUNG wire#powerrail
      Contact( #Mx_ET51 )
      Contact( #Simultaneo_Mx )
   END_RUNG wire#w1
   RUNG wire#powerrail
      Contact( #Mx_ET11 )
   END_RUNG wire#w2
   RUNG wire#powerrail
      Contact( #Mx_ET12 )
   END_RUNG wire#w2
   RUNG wire#powerrail
      I_Contact( #Mx_ET10 )
      wire#w4
      I_Contact( #Mx_ET11 )
      I_Contact( #Mx_ET12 )
      wire#w5
      I_Contact( #Mx_ET51 )
   END_RUNG wire#w6
   RUNG wire#powerrail
      I_Contact( #CNTSeg_pHsMx_E1E3.QU )
   END_RUNG wire#w4
   RUNG wire#w5
      I_Contact( #CNTSeg_pHsMx_E1E3.QU )
   END_RUNG wire#w6
   RUNG wire#w5
      I_Contact( #Simultaneo_Mx )
   END_RUNG wire#w6
   // the same network as SCL:
   #CNT_pHsMx_E1E3(IN := (((#Mx_ET10 OR (#Mx_ET51 AND #Simultaneo_Mx)) AND #CNTSeg_pHsMx_E1E3.QU) OR #Mx_ET11 OR #Mx_ET12) AND #VAR_pHs AND #Avance_E1_Tx_Ok AND NOT #EstadoZona.Manual_CBx,   // "FB910_CNT_UHS"
                   R := (NOT #Mx_ET10 OR NOT #CNTSeg_pHsMx_E1E3.QU) AND NOT #Mx_ET11 AND NOT #Mx_ET12 AND (NOT #Mx_ET51 OR NOT #CNTSeg_pHsMx_E1E3.QU OR NOT #Simultaneo_Mx),
                   PV := #V_CNT_pHsMx_E1,
                   BaseUnidades_ms := "CTE_BaseUnidades_1ms");
END_REGION

REGION Network 106: DETERMINA PASO ET10 - ET11 (Nota: Control de Tiempo para dar el FTF a la Mesa Anterior)
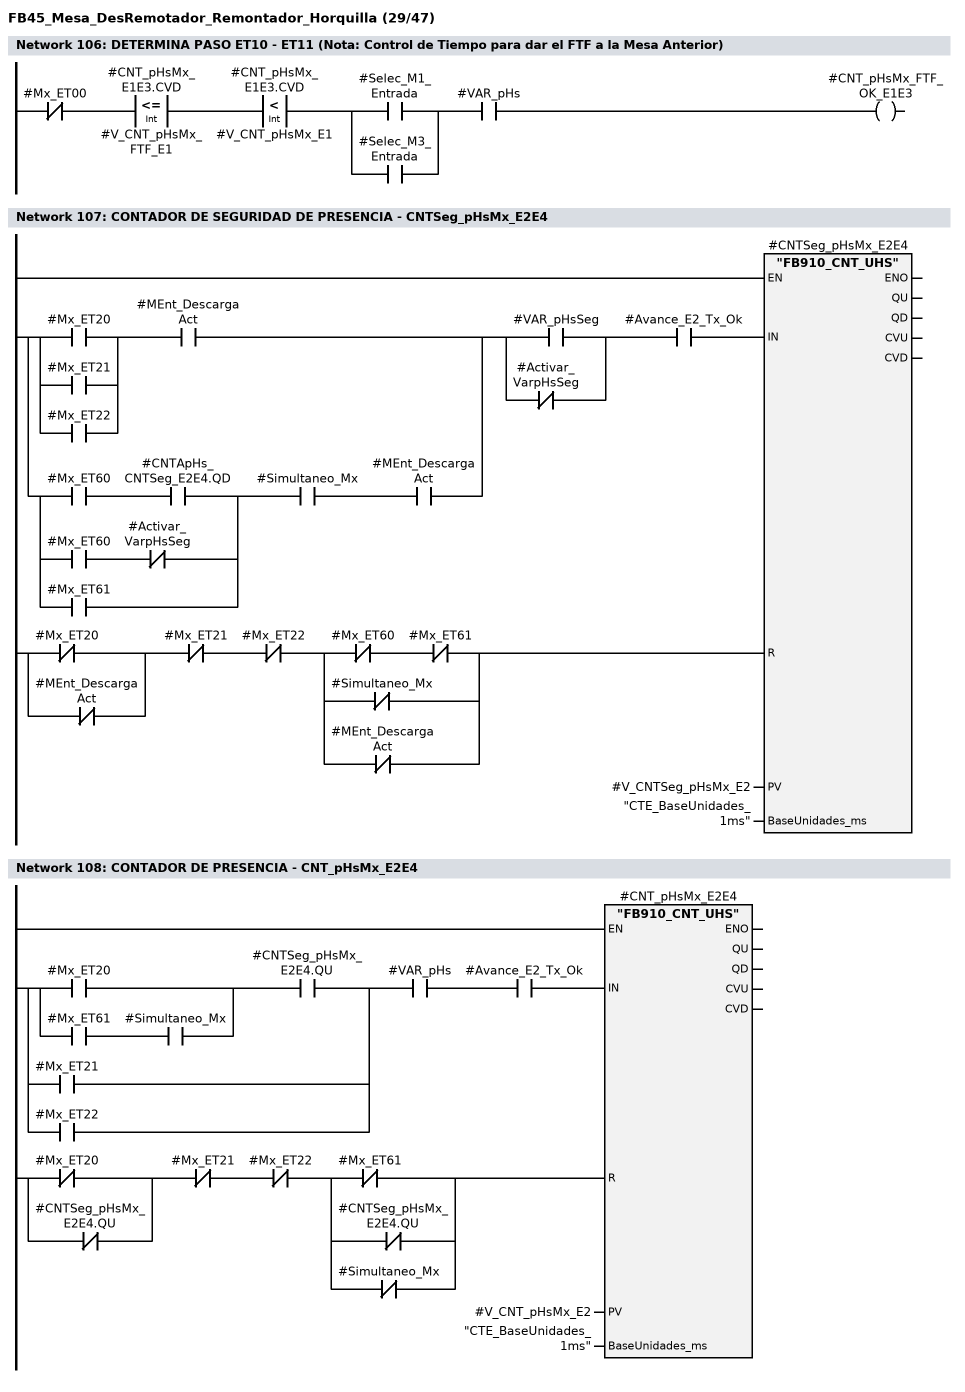
   RUNG wire#powerrail
      I_Contact( #Mx_ET00 )
      { S7_Templates := "SrcType := Int" } LE_Contact(in1 := #CNT_pHsMx_E1E3.CVD, in2 := #V_CNT_pHsMx_FTF_E1)
      { S7_Templates := "SrcType := Int" } LT_Contact(in1 := #CNT_pHsMx_E1E3.CVD, in2 := #V_CNT_pHsMx_E1)
      wire#w1
      Contact( #Selec_M1_Entrada )
      wire#w2
      Contact( #VAR_pHs )
      Coil( #CNT_pHsMx_FTF_OK_E1E3 )
   END_RUNG
   RUNG wire#w1
      Contact( #Selec_M3_Entrada )
   END_RUNG wire#w2
   // the same network as SCL:
   #CNT_pHsMx_FTF_OK_E1E3 := NOT #Mx_ET00 AND (#CNT_pHsMx_E1E3.CVD <= #V_CNT_pHsMx_FTF_E1) AND (#CNT_pHsMx_E1E3.CVD < #V_CNT_pHsMx_E1) AND (#Selec_M1_Entrada OR #Selec_M3_Entrada) AND #VAR_pHs;
END_REGION

REGION Network 107: CONTADOR DE SEGURIDAD DE PRESENCIA - CNTSeg_pHsMx_E2E4
   RUNG wire#powerrail
      #CNTSeg_pHsMx_E2E4(IN := wire#w5, R := wire#w8, PV := #V_CNTSeg_pHsMx_E2, BaseUnidades_ms := "CTE_BaseUnidades_1ms", QU =>, QD =>, CVU =>, CVD =>)
   END_RUNG
   RUNG wire#powerrail
      Contact( #Mx_ET20 )
      wire#w1
      Contact( #MEnt_DescargaAct )
      wire#w2
      Contact( #VAR_pHsSeg )
      wire#w4
      Contact( #Avance_E2_Tx_Ok )
   END_RUNG wire#w5
   RUNG wire#powerrail
      Contact( #Mx_ET21 )
   END_RUNG wire#w1
   RUNG wire#powerrail
      Contact( #Mx_ET22 )
   END_RUNG wire#w1
   RUNG wire#powerrail
      Contact( #Mx_ET60 )
      Contact( #CNTApHs_CNTSeg_E2E4.QD )
      wire#w3
      Contact( #Simultaneo_Mx )
      Contact( #MEnt_DescargaAct )
   END_RUNG wire#w2
   RUNG wire#powerrail
      Contact( #Mx_ET60 )
      I_Contact( #Activar_VarpHsSeg )
   END_RUNG wire#w3
   RUNG wire#powerrail
      Contact( #Mx_ET61 )
   END_RUNG wire#w3
   RUNG wire#w2
      I_Contact( #Activar_VarpHsSeg )
   END_RUNG wire#w4
   RUNG wire#powerrail
      I_Contact( #Mx_ET20 )
      wire#w6
      I_Contact( #Mx_ET21 )
      I_Contact( #Mx_ET22 )
      wire#w7
      I_Contact( #Mx_ET60 )
      I_Contact( #Mx_ET61 )
   END_RUNG wire#w8
   RUNG wire#powerrail
      I_Contact( #MEnt_DescargaAct )
   END_RUNG wire#w6
   RUNG wire#w7
      I_Contact( #Simultaneo_Mx )
   END_RUNG wire#w8
   RUNG wire#w7
      I_Contact( #MEnt_DescargaAct )
   END_RUNG wire#w8
   // the same network as SCL:
   #CNTSeg_pHsMx_E2E4(IN := (((#Mx_ET20 OR #Mx_ET21 OR #Mx_ET22) AND #MEnt_DescargaAct) OR (((#Mx_ET60 AND #CNTApHs_CNTSeg_E2E4.QD) OR (#Mx_ET60 AND NOT #Activar_VarpHsSeg) OR #Mx_ET61) AND #Simultaneo_Mx AND #MEnt_DescargaAct)) AND (#VAR_pHsSeg OR NOT #Activar_VarpHsSeg) AND #Avance_E2_Tx_Ok,   // "FB910_CNT_UHS"
                      R := (NOT #Mx_ET20 OR NOT #MEnt_DescargaAct) AND NOT #Mx_ET21 AND NOT #Mx_ET22 AND ((NOT #Mx_ET60 AND NOT #Mx_ET61) OR NOT #Simultaneo_Mx OR NOT #MEnt_DescargaAct),
                      PV := #V_CNTSeg_pHsMx_E2,
                      BaseUnidades_ms := "CTE_BaseUnidades_1ms");
END_REGION

REGION Network 108: CONTADOR DE PRESENCIA - CNT_pHsMx_E2E4
   RUNG wire#powerrail
      #CNT_pHsMx_E2E4(IN := wire#w3, R := wire#w6, PV := #V_CNT_pHsMx_E2, BaseUnidades_ms := "CTE_BaseUnidades_1ms", QU =>, QD =>, CVU =>, CVD =>)
   END_RUNG
   RUNG wire#powerrail
      Contact( #Mx_ET20 )
      wire#w1
      Contact( #CNTSeg_pHsMx_E2E4.QU )
      wire#w2
      Contact( #VAR_pHs )
      Contact( #Avance_E2_Tx_Ok )
   END_RUNG wire#w3
   RUNG wire#powerrail
      Contact( #Mx_ET61 )
      Contact( #Simultaneo_Mx )
   END_RUNG wire#w1
   RUNG wire#powerrail
      Contact( #Mx_ET21 )
   END_RUNG wire#w2
   RUNG wire#powerrail
      Contact( #Mx_ET22 )
   END_RUNG wire#w2
   RUNG wire#powerrail
      I_Contact( #Mx_ET20 )
      wire#w4
      I_Contact( #Mx_ET21 )
      I_Contact( #Mx_ET22 )
      wire#w5
      I_Contact( #Mx_ET61 )
   END_RUNG wire#w6
   RUNG wire#powerrail
      I_Contact( #CNTSeg_pHsMx_E2E4.QU )
   END_RUNG wire#w4
   RUNG wire#w5
      I_Contact( #CNTSeg_pHsMx_E2E4.QU )
   END_RUNG wire#w6
   RUNG wire#w5
      I_Contact( #Simultaneo_Mx )
   END_RUNG wire#w6
   // the same network as SCL:
   #CNT_pHsMx_E2E4(IN := (((#Mx_ET20 OR (#Mx_ET61 AND #Simultaneo_Mx)) AND #CNTSeg_pHsMx_E2E4.QU) OR #Mx_ET21 OR #Mx_ET22) AND #VAR_pHs AND #Avance_E2_Tx_Ok,   // "FB910_CNT_UHS"
                   R := (NOT #Mx_ET20 OR NOT #CNTSeg_pHsMx_E2E4.QU) AND NOT #Mx_ET21 AND NOT #Mx_ET22 AND (NOT #Mx_ET61 OR NOT #CNTSeg_pHsMx_E2E4.QU OR NOT #Simultaneo_Mx),
                   PV := #V_CNT_pHsMx_E2,
                   BaseUnidades_ms := "CTE_BaseUnidades_1ms");
END_REGION

REGION Network 109: DETERMINA PASO ET20 - ET21 (Nota: Control de Tiempo para dar el FTF a la Mesa Anterior)
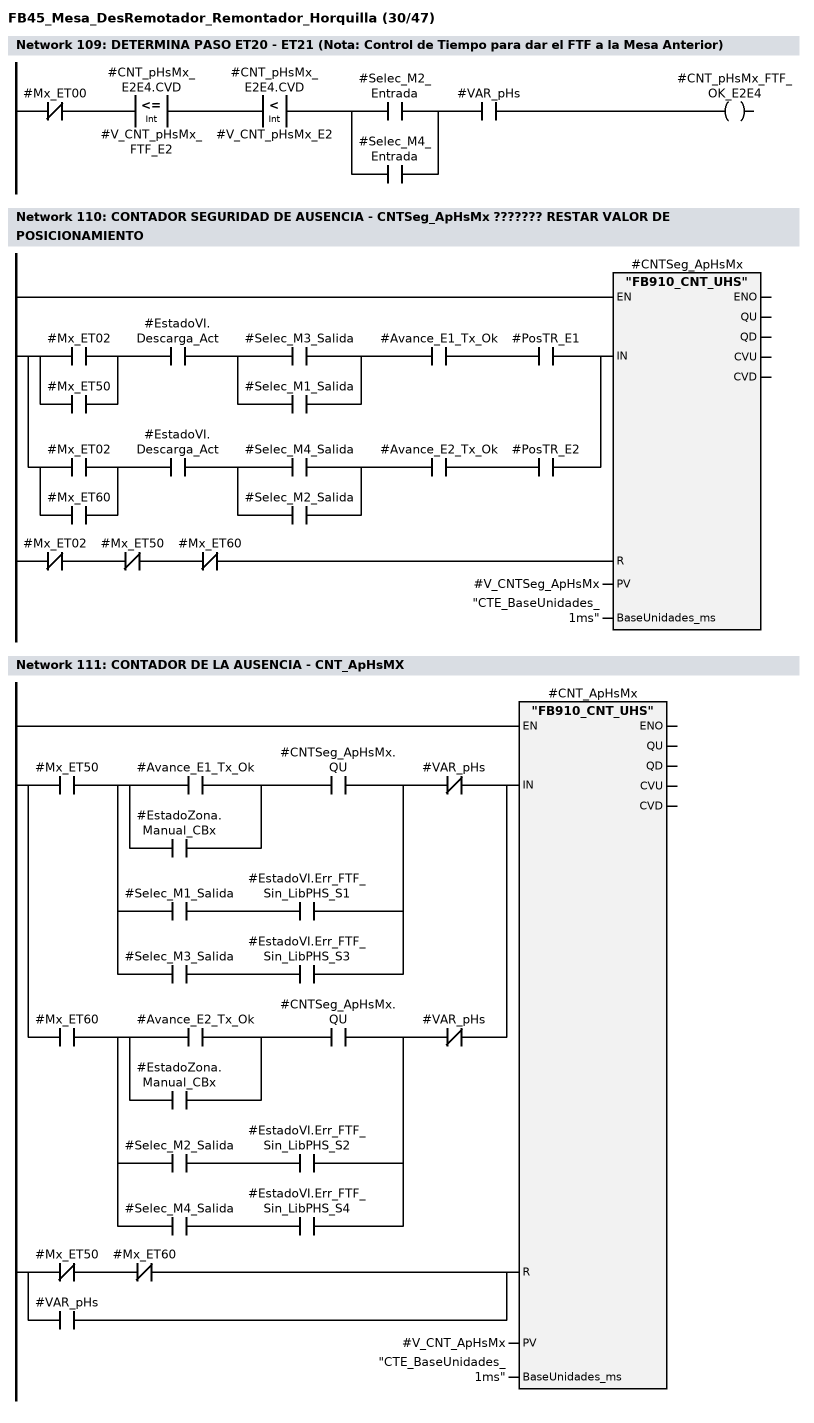
   RUNG wire#powerrail
      I_Contact( #Mx_ET00 )
      { S7_Templates := "SrcType := Int" } LE_Contact(in1 := #CNT_pHsMx_E2E4.CVD, in2 := #V_CNT_pHsMx_FTF_E2)
      { S7_Templates := "SrcType := Int" } LT_Contact(in1 := #CNT_pHsMx_E2E4.CVD, in2 := #V_CNT_pHsMx_E2)
      wire#w1
      Contact( #Selec_M2_Entrada )
      wire#w2
      Contact( #VAR_pHs )
      Coil( #CNT_pHsMx_FTF_OK_E2E4 )
   END_RUNG
   RUNG wire#w1
      Contact( #Selec_M4_Entrada )
   END_RUNG wire#w2
   // the same network as SCL:
   #CNT_pHsMx_FTF_OK_E2E4 := NOT #Mx_ET00 AND (#CNT_pHsMx_E2E4.CVD <= #V_CNT_pHsMx_FTF_E2) AND (#CNT_pHsMx_E2E4.CVD < #V_CNT_pHsMx_E2) AND (#Selec_M2_Entrada OR #Selec_M4_Entrada) AND #VAR_pHs;
END_REGION

REGION Network 110: CONTADOR SEGURIDAD DE AUSENCIA - CNTSeg_ApHsMx ??????? RESTAR VALOR DE POSICIONAMIENTO
   RUNG wire#powerrail
      #CNTSeg_ApHsMx(IN := wire#w7, R := wire#w8, PV := #V_CNTSeg_ApHsMx, BaseUnidades_ms := "CTE_BaseUnidades_1ms", QU =>, QD =>, CVU =>, CVD =>)
   END_RUNG
   RUNG wire#powerrail
      Contact( #Mx_ET02 )
      wire#w1
      Contact( #EstadoVI.Descarga_Act )
      wire#w2
      Contact( #Selec_M3_Salida )
      wire#w3
      Contact( #Avance_E1_Tx_Ok )
      Contact( #PosTR_E1 )
   END_RUNG wire#w7
   RUNG wire#powerrail
      Contact( #Mx_ET50 )
   END_RUNG wire#w1
   RUNG wire#w2
      Contact( #Selec_M1_Salida )
   END_RUNG wire#w3
   RUNG wire#powerrail
      Contact( #Mx_ET02 )
      wire#w4
      Contact( #EstadoVI.Descarga_Act )
      wire#w5
      Contact( #Selec_M4_Salida )
      wire#w6
      Contact( #Avance_E2_Tx_Ok )
      Contact( #PosTR_E2 )
   END_RUNG wire#w7
   RUNG wire#powerrail
      Contact( #Mx_ET60 )
   END_RUNG wire#w4
   RUNG wire#w5
      Contact( #Selec_M2_Salida )
   END_RUNG wire#w6
   RUNG wire#powerrail
      I_Contact( #Mx_ET02 )
      I_Contact( #Mx_ET50 )
      I_Contact( #Mx_ET60 )
   END_RUNG wire#w8
   // the same network as SCL:
   #CNTSeg_ApHsMx(IN := ((#Mx_ET02 OR #Mx_ET50) AND #EstadoVI.Descarga_Act AND (#Selec_M3_Salida OR #Selec_M1_Salida) AND #Avance_E1_Tx_Ok AND #PosTR_E1) OR ((#Mx_ET02 OR #Mx_ET60) AND #EstadoVI.Descarga_Act AND (#Selec_M4_Salida OR #Selec_M2_Salida) AND #Avance_E2_Tx_Ok AND #PosTR_E2),   // "FB910_CNT_UHS"
                  R := NOT #Mx_ET02 AND NOT #Mx_ET50 AND NOT #Mx_ET60,
                  PV := #V_CNTSeg_ApHsMx,
                  BaseUnidades_ms := "CTE_BaseUnidades_1ms");
END_REGION

REGION Network 111: CONTADOR DE LA AUSENCIA - CNT_ApHsMX
   RUNG wire#powerrail
      #CNT_ApHsMx(IN := wire#w7, R := wire#w8, PV := #V_CNT_ApHsMx, BaseUnidades_ms := "CTE_BaseUnidades_1ms", QU =>, QD =>, CVU =>, CVD =>)
   END_RUNG
   RUNG wire#powerrail
      Contact( #Mx_ET50 )
      wire#w1
      Contact( #Avance_E1_Tx_Ok )
      wire#w2
      Contact( #CNTSeg_ApHsMx.QU )
      wire#w3
      I_Contact( #VAR_pHs )
   END_RUNG wire#w7
   RUNG wire#w1
      Contact( #EstadoZona.Manual_CBx )
   END_RUNG wire#w2
   RUNG wire#w1
      Contact( #Selec_M1_Salida )
      Contact( #EstadoVI.Err_FTF_Sin_LibPHS_S1 )
   END_RUNG wire#w3
   RUNG wire#w1
      Contact( #Selec_M3_Salida )
      Contact( #EstadoVI.Err_FTF_Sin_LibPHS_S3 )
   END_RUNG wire#w3
   RUNG wire#powerrail
      Contact( #Mx_ET60 )
      wire#w4
      Contact( #Avance_E2_Tx_Ok )
      wire#w5
      Contact( #CNTSeg_ApHsMx.QU )
      wire#w6
      I_Contact( #VAR_pHs )
   END_RUNG wire#w7
   RUNG wire#w4
      Contact( #EstadoZona.Manual_CBx )
   END_RUNG wire#w5
   RUNG wire#w4
      Contact( #Selec_M2_Salida )
      Contact( #EstadoVI.Err_FTF_Sin_LibPHS_S2 )
   END_RUNG wire#w6
   RUNG wire#w4
      Contact( #Selec_M4_Salida )
      Contact( #EstadoVI.Err_FTF_Sin_LibPHS_S4 )
   END_RUNG wire#w6
   RUNG wire#powerrail
      I_Contact( #Mx_ET50 )
      I_Contact( #Mx_ET60 )
   END_RUNG wire#w8
   RUNG wire#powerrail
      Contact( #VAR_pHs )
   END_RUNG wire#w8
   // the same network as SCL:
   #CNT_ApHsMx(IN := (#Mx_ET50 AND (((#Avance_E1_Tx_Ok OR #EstadoZona.Manual_CBx) AND #CNTSeg_ApHsMx.QU) OR (#Selec_M1_Salida AND #EstadoVI.Err_FTF_Sin_LibPHS_S1) OR (#Selec_M3_Salida AND #EstadoVI.Err_FTF_Sin_LibPHS_S3)) AND NOT #VAR_pHs) OR (#Mx_ET60 AND (((#Avance_E2_Tx_Ok OR #EstadoZona.Manual_CBx) AND #CNTSeg_ApHsMx.QU) OR (#Selec_M2_Salida AND #EstadoVI.Err_FTF_Sin_LibPHS_S2) OR (#Selec_M4_Salida AND #EstadoVI.Err_FTF_Sin_LibPHS_S4)) AND NOT #VAR_pHs),   // "FB910_CNT_UHS"
               R := (NOT #Mx_ET50 AND NOT #Mx_ET60) OR #VAR_pHs,
               PV := #V_CNT_ApHsMx,
               BaseUnidades_ms := "CTE_BaseUnidades_1ms");
END_REGION

REGION Network 112: TEMPORIZADOR DE BLOQUEO DE MESA
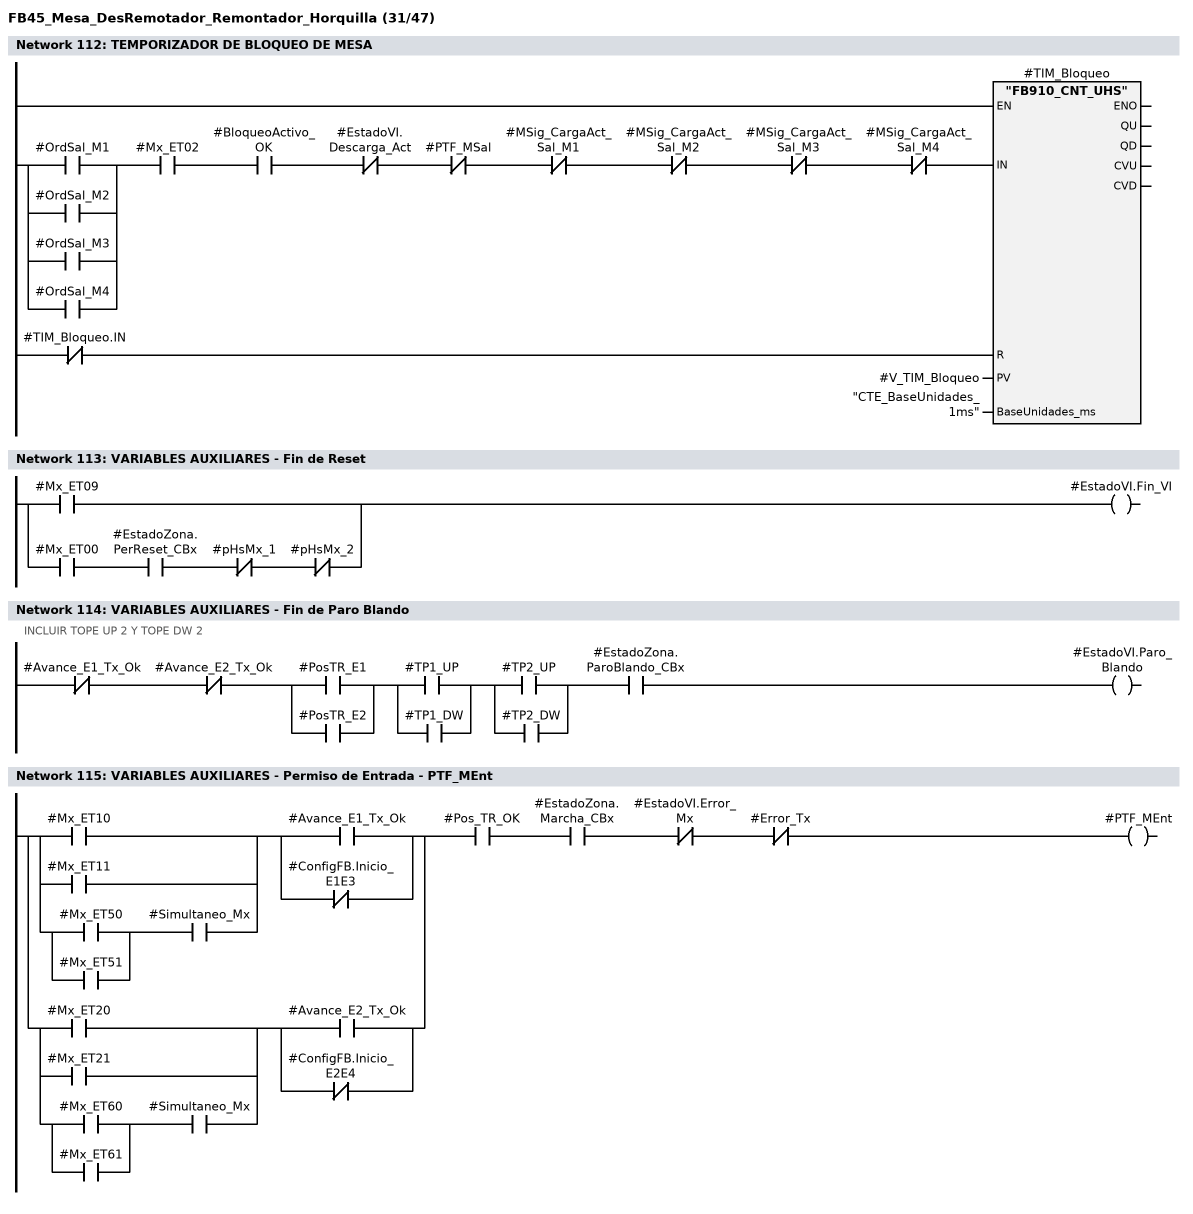
   RUNG wire#powerrail
      #TIM_Bloqueo(IN := wire#w2, R := wire#w3, PV := #V_TIM_Bloqueo, BaseUnidades_ms := "CTE_BaseUnidades_1ms", QU =>, QD =>, CVU =>, CVD =>)
   END_RUNG
   RUNG wire#powerrail
      Contact( #OrdSal_M1 )
      wire#w1
      Contact( #Mx_ET02 )
      Contact( #BloqueoActivo_OK )
      I_Contact( #EstadoVI.Descarga_Act )
      I_Contact( #PTF_MSal )
      I_Contact( #MSig_CargaAct_Sal_M1 )
      I_Contact( #MSig_CargaAct_Sal_M2 )
      I_Contact( #MSig_CargaAct_Sal_M3 )
      I_Contact( #MSig_CargaAct_Sal_M4 )
   END_RUNG wire#w2
   RUNG wire#powerrail
      Contact( #OrdSal_M2 )
   END_RUNG wire#w1
   RUNG wire#powerrail
      Contact( #OrdSal_M3 )
   END_RUNG wire#w1
   RUNG wire#powerrail
      Contact( #OrdSal_M4 )
   END_RUNG wire#w1
   RUNG wire#powerrail
      I_Contact( #TIM_Bloqueo.IN )
   END_RUNG wire#w3
   // the same network as SCL:
   #TIM_Bloqueo(IN := (#OrdSal_M1 OR #OrdSal_M2 OR #OrdSal_M3 OR #OrdSal_M4) AND #Mx_ET02 AND #BloqueoActivo_OK AND NOT #EstadoVI.Descarga_Act AND NOT #PTF_MSal AND NOT #MSig_CargaAct_Sal_M1 AND NOT #MSig_CargaAct_Sal_M2 AND NOT #MSig_CargaAct_Sal_M3 AND NOT #MSig_CargaAct_Sal_M4,   // "FB910_CNT_UHS"
                R := NOT #TIM_Bloqueo.IN,
                PV := #V_TIM_Bloqueo,
                BaseUnidades_ms := "CTE_BaseUnidades_1ms");
END_REGION

REGION Network 113: VARIABLES AUXILIARES - Fin de Reset
   RUNG wire#powerrail
      Contact( #Mx_ET09 )
      wire#w1
      Coil( #EstadoVI.Fin_VI )
   END_RUNG
   RUNG wire#powerrail
      Contact( #Mx_ET00 )
      Contact( #EstadoZona.PerReset_CBx )
      I_Contact( #pHsMx_1 )
      I_Contact( #pHsMx_2 )
   END_RUNG wire#w1
   // the same network as SCL:
   #EstadoVI.Fin_VI := #Mx_ET09 OR (#Mx_ET00 AND #EstadoZona.PerReset_CBx AND NOT #pHsMx_1 AND NOT #pHsMx_2);
END_REGION

REGION Network 114: VARIABLES AUXILIARES - Fin de Paro Blando
   // INCLUIR TOPE UP 2 Y TOPE DW 2
   RUNG wire#powerrail
      I_Contact( #Avance_E1_Tx_Ok )
      I_Contact( #Avance_E2_Tx_Ok )
      wire#w1
      Contact( #PosTR_E1 )
      wire#w2
      Contact( #TP1_UP )
      wire#w3
      Contact( #TP2_UP )
      wire#w4
      Contact( #EstadoZona.ParoBlando_CBx )
      Coil( #EstadoVI.Paro_Blando )
   END_RUNG
   RUNG wire#w1
      Contact( #PosTR_E2 )
   END_RUNG wire#w2
   RUNG wire#w2
      Contact( #TP1_DW )
   END_RUNG wire#w3
   RUNG wire#w3
      Contact( #TP2_DW )
   END_RUNG wire#w4
   // the same network as SCL:
   #EstadoVI.Paro_Blando := NOT #Avance_E1_Tx_Ok AND NOT #Avance_E2_Tx_Ok AND (#PosTR_E1 OR #PosTR_E2) AND (#TP1_UP OR #TP1_DW) AND (#TP2_UP OR #TP2_DW) AND #EstadoZona.ParoBlando_CBx;
END_REGION

REGION Network 115: VARIABLES AUXILIARES - Permiso de Entrada - PTF_MEnt
   RUNG wire#powerrail
      Contact( #Mx_ET10 )
      wire#w1
      Contact( #Avance_E1_Tx_Ok )
      wire#w3
      Contact( #Pos_TR_OK )
      Contact( #EstadoZona.Marcha_CBx )
      I_Contact( #EstadoVI.Error_Mx )
      I_Contact( #Error_Tx )
      Coil( #PTF_MEnt )
   END_RUNG
   RUNG wire#powerrail
      Contact( #Mx_ET11 )
   END_RUNG wire#w1
   RUNG wire#powerrail
      Contact( #Mx_ET50 )
      wire#w2
      Contact( #Simultaneo_Mx )
   END_RUNG wire#w1
   RUNG wire#powerrail
      Contact( #Mx_ET51 )
   END_RUNG wire#w2
   RUNG wire#w1
      I_Contact( #ConfigFB.Inicio_E1E3 )
   END_RUNG wire#w3
   RUNG wire#powerrail
      Contact( #Mx_ET20 )
      wire#w4
      Contact( #Avance_E2_Tx_Ok )
   END_RUNG wire#w3
   RUNG wire#powerrail
      Contact( #Mx_ET21 )
   END_RUNG wire#w4
   RUNG wire#powerrail
      Contact( #Mx_ET60 )
      wire#w5
      Contact( #Simultaneo_Mx )
   END_RUNG wire#w4
   RUNG wire#powerrail
      Contact( #Mx_ET61 )
   END_RUNG wire#w5
   RUNG wire#w4
      I_Contact( #ConfigFB.Inicio_E2E4 )
   END_RUNG wire#w3
   // the same network as SCL:
   #PTF_MEnt := (((#Mx_ET10 OR #Mx_ET11 OR ((#Mx_ET50 OR #Mx_ET51) AND #Simultaneo_Mx)) AND (#Avance_E1_Tx_Ok OR NOT #ConfigFB.Inicio_E1E3)) OR ((#Mx_ET20 OR #Mx_ET21 OR ((#Mx_ET60 OR #Mx_ET61) AND #Simultaneo_Mx)) AND (#Avance_E2_Tx_Ok OR NOT #ConfigFB.Inicio_E2E4))) AND #Pos_TR_OK AND #EstadoZona.Marcha_CBx AND NOT #EstadoVI.Error_Mx AND NOT #Error_Tx;
END_REGION

REGION Network 116: VARIABLES AUXILIARES - Aviso de Salida - AVTF_MSal
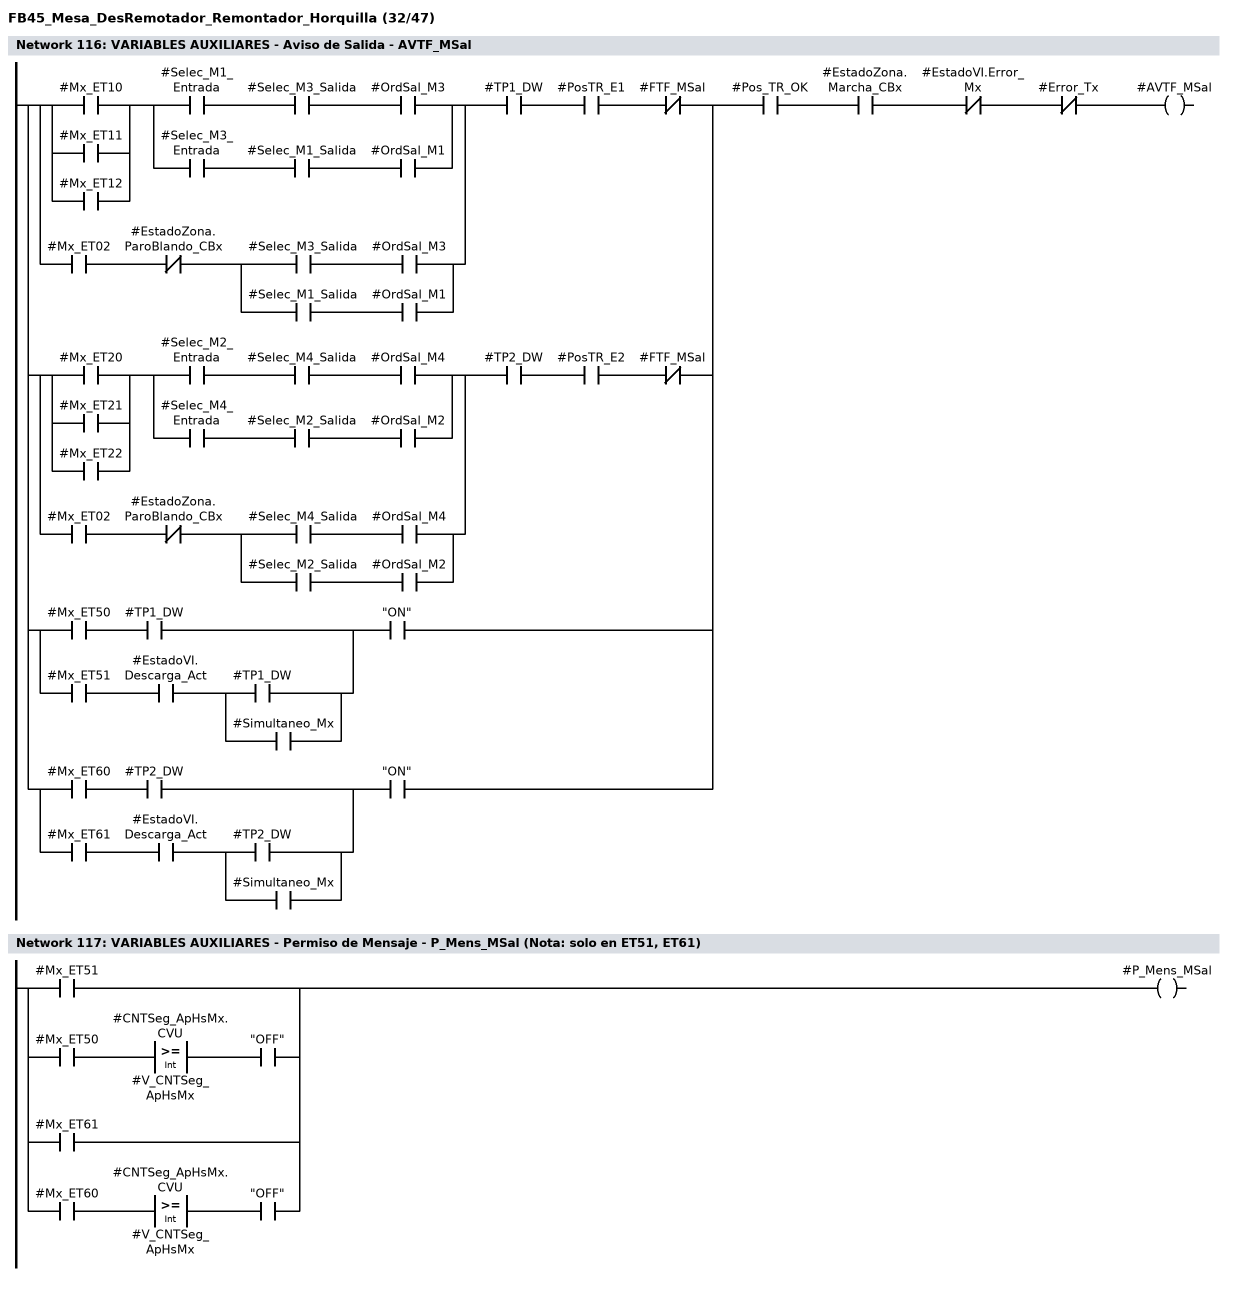
   RUNG wire#powerrail
      Contact( #Mx_ET10 )
      wire#w1
      Contact( #Selec_M1_Entrada )
      Contact( #Selec_M3_Salida )
      Contact( #OrdSal_M3 )
      wire#w2
      Contact( #TP1_DW )
      Contact( #PosTR_E1 )
      I_Contact( #FTF_MSal )
      wire#w4
      Contact( #Pos_TR_OK )
      Contact( #EstadoZona.Marcha_CBx )
      I_Contact( #EstadoVI.Error_Mx )
      I_Contact( #Error_Tx )
      Coil( #AVTF_MSal )
   END_RUNG
   RUNG wire#powerrail
      Contact( #Mx_ET11 )
   END_RUNG wire#w1
   RUNG wire#powerrail
      Contact( #Mx_ET12 )
   END_RUNG wire#w1
   RUNG wire#w1
      Contact( #Selec_M3_Entrada )
      Contact( #Selec_M1_Salida )
      Contact( #OrdSal_M1 )
   END_RUNG wire#w2
   RUNG wire#powerrail
      Contact( #Mx_ET02 )
      I_Contact( #EstadoZona.ParoBlando_CBx )
      wire#w3
      Contact( #Selec_M3_Salida )
      Contact( #OrdSal_M3 )
   END_RUNG wire#w2
   RUNG wire#w3
      Contact( #Selec_M1_Salida )
      Contact( #OrdSal_M1 )
   END_RUNG wire#w2
   RUNG wire#powerrail
      Contact( #Mx_ET20 )
      wire#w5
      Contact( #Selec_M2_Entrada )
      Contact( #Selec_M4_Salida )
      Contact( #OrdSal_M4 )
      wire#w6
      Contact( #TP2_DW )
      Contact( #PosTR_E2 )
      I_Contact( #FTF_MSal )
   END_RUNG wire#w4
   RUNG wire#powerrail
      Contact( #Mx_ET21 )
   END_RUNG wire#w5
   RUNG wire#powerrail
      Contact( #Mx_ET22 )
   END_RUNG wire#w5
   RUNG wire#w5
      Contact( #Selec_M4_Entrada )
      Contact( #Selec_M2_Salida )
      Contact( #OrdSal_M2 )
   END_RUNG wire#w6
   RUNG wire#powerrail
      Contact( #Mx_ET02 )
      I_Contact( #EstadoZona.ParoBlando_CBx )
      wire#w7
      Contact( #Selec_M4_Salida )
      Contact( #OrdSal_M4 )
   END_RUNG wire#w6
   RUNG wire#w7
      Contact( #Selec_M2_Salida )
      Contact( #OrdSal_M2 )
   END_RUNG wire#w6
   RUNG wire#powerrail
      Contact( #Mx_ET50 )
      Contact( #TP1_DW )
      wire#w8
      Contact( "ON" )
   END_RUNG wire#w4
   RUNG wire#powerrail
      Contact( #Mx_ET51 )
      Contact( #EstadoVI.Descarga_Act )
      wire#w9
      Contact( #TP1_DW )
   END_RUNG wire#w8
   RUNG wire#w9
      Contact( #Simultaneo_Mx )
   END_RUNG wire#w8
   RUNG wire#powerrail
      Contact( #Mx_ET60 )
      Contact( #TP2_DW )
      wire#w10
      Contact( "ON" )
   END_RUNG wire#w4
   RUNG wire#powerrail
      Contact( #Mx_ET61 )
      Contact( #EstadoVI.Descarga_Act )
      wire#w11
      Contact( #TP2_DW )
   END_RUNG wire#w10
   RUNG wire#w11
      Contact( #Simultaneo_Mx )
   END_RUNG wire#w10
   // the same network as SCL:
   #AVTF_MSal := (((((#Mx_ET10 OR #Mx_ET11 OR #Mx_ET12) AND ((#Selec_M1_Entrada AND #Selec_M3_Salida AND #OrdSal_M3) OR (#Selec_M3_Entrada AND #Selec_M1_Salida AND #OrdSal_M1))) OR (#Mx_ET02 AND NOT #EstadoZona.ParoBlando_CBx AND ((#Selec_M3_Salida AND #OrdSal_M3) OR (#Selec_M1_Salida AND #OrdSal_M1)))) AND #TP1_DW AND #PosTR_E1 AND NOT #FTF_MSal) OR ((((#Mx_ET20 OR #Mx_ET21 OR #Mx_ET22) AND ((#Selec_M2_Entrada AND #Selec_M4_Salida AND #OrdSal_M4) OR (#Selec_M4_Entrada AND #Selec_M2_Salida AND #OrdSal_M2))) OR (#Mx_ET02 AND NOT #EstadoZona.ParoBlando_CBx AND ((#Selec_M4_Salida AND #OrdSal_M4) OR (#Selec_M2_Salida AND #OrdSal_M2)))) AND #TP2_DW AND #PosTR_E2 AND NOT #FTF_MSal) OR (((#Mx_ET50 AND #TP1_DW) OR (#Mx_ET51 AND #EstadoVI.Descarga_Act AND (#TP1_DW OR #Simultaneo_Mx))) AND "ON") OR (((#Mx_ET60 AND #TP2_DW) OR (#Mx_ET61 AND #EstadoVI.Descarga_Act AND (#TP2_DW OR #Simultaneo_Mx))) AND "ON")) AND #Pos_TR_OK AND #EstadoZona.Marcha_CBx AND NOT #EstadoVI.Error_Mx AND NOT #Error_Tx;
END_REGION

REGION Network 117: VARIABLES AUXILIARES - Permiso de Mensaje - P_Mens_MSal (Nota: solo en ET51, ET61)
   RUNG wire#powerrail
      Contact( #Mx_ET51 )
      wire#w1
      Coil( #P_Mens_MSal )
   END_RUNG
   RUNG wire#powerrail
      Contact( #Mx_ET50 )
      { S7_Templates := "SrcType := Int" } GE_Contact(in1 := #CNTSeg_ApHsMx.CVU, in2 := #V_CNTSeg_ApHsMx)
      Contact( "OFF" )
   END_RUNG wire#w1
   RUNG wire#powerrail
      Contact( #Mx_ET61 )
   END_RUNG wire#w1
   RUNG wire#powerrail
      Contact( #Mx_ET60 )
      { S7_Templates := "SrcType := Int" } GE_Contact(in1 := #CNTSeg_ApHsMx.CVU, in2 := #V_CNTSeg_ApHsMx)
      Contact( "OFF" )
   END_RUNG wire#w1
   // the same network as SCL:
   #P_Mens_MSal := #Mx_ET51 OR (#Mx_ET50 AND (#CNTSeg_ApHsMx.CVU >= #V_CNTSeg_ApHsMx) AND "OFF") OR #Mx_ET61 OR (#Mx_ET60 AND (#CNTSeg_ApHsMx.CVU >= #V_CNTSeg_ApHsMx) AND "OFF");
END_REGION

REGION Network 118: MULTIPLEXADO FINAL SEÑALES DE ENTRADA DE CARGA - PTF_MEnt
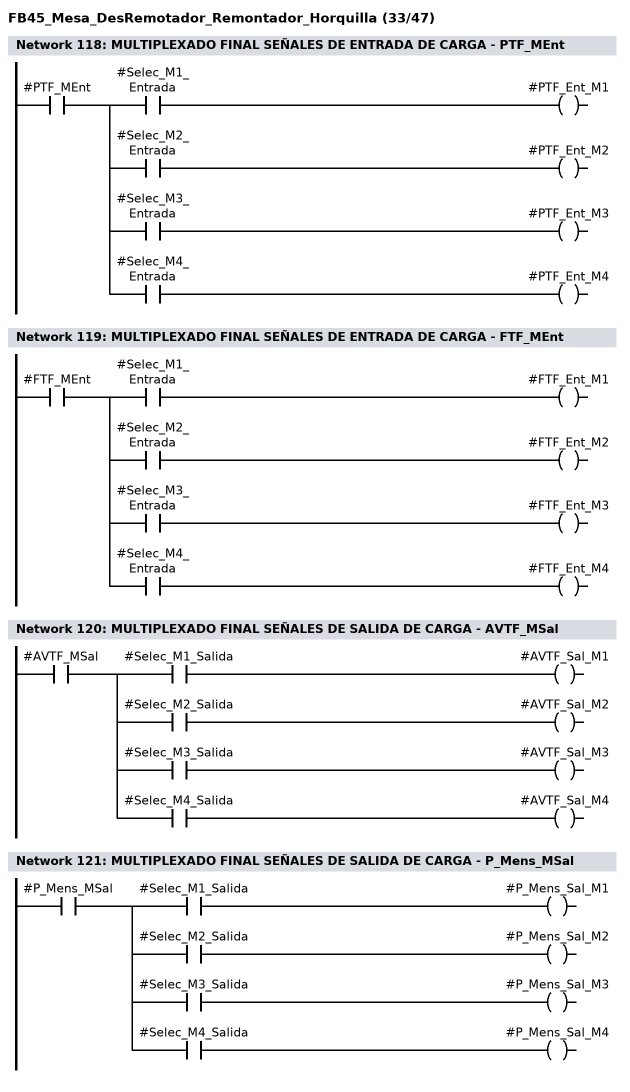
   RUNG wire#powerrail
      Contact( #PTF_MEnt )
      wire#w1
      Contact( #Selec_M1_Entrada )
      Coil( #PTF_Ent_M1 )
   END_RUNG
   RUNG wire#w1
      Contact( #Selec_M2_Entrada )
      Coil( #PTF_Ent_M2 )
   END_RUNG
   RUNG wire#w1
      Contact( #Selec_M3_Entrada )
      Coil( #PTF_Ent_M3 )
   END_RUNG
   RUNG wire#w1
      Contact( #Selec_M4_Entrada )
      Coil( #PTF_Ent_M4 )
   END_RUNG
   // the same network as SCL:
   #PTF_Ent_M1 := #PTF_MEnt AND #Selec_M1_Entrada;
   #PTF_Ent_M2 := #PTF_MEnt AND #Selec_M2_Entrada;
   #PTF_Ent_M3 := #PTF_MEnt AND #Selec_M3_Entrada;
   #PTF_Ent_M4 := #PTF_MEnt AND #Selec_M4_Entrada;
END_REGION

REGION Network 119: MULTIPLEXADO FINAL SEÑALES DE ENTRADA DE CARGA - FTF_MEnt
   RUNG wire#powerrail
      Contact( #FTF_MEnt )
      wire#w1
      Contact( #Selec_M1_Entrada )
      Coil( #FTF_Ent_M1 )
   END_RUNG
   RUNG wire#w1
      Contact( #Selec_M2_Entrada )
      Coil( #FTF_Ent_M2 )
   END_RUNG
   RUNG wire#w1
      Contact( #Selec_M3_Entrada )
      Coil( #FTF_Ent_M3 )
   END_RUNG
   RUNG wire#w1
      Contact( #Selec_M4_Entrada )
      Coil( #FTF_Ent_M4 )
   END_RUNG
   // the same network as SCL:
   #FTF_Ent_M1 := #FTF_MEnt AND #Selec_M1_Entrada;
   #FTF_Ent_M2 := #FTF_MEnt AND #Selec_M2_Entrada;
   #FTF_Ent_M3 := #FTF_MEnt AND #Selec_M3_Entrada;
   #FTF_Ent_M4 := #FTF_MEnt AND #Selec_M4_Entrada;
END_REGION

REGION Network 120: MULTIPLEXADO FINAL SEÑALES DE SALIDA DE CARGA - AVTF_MSal
   RUNG wire#powerrail
      Contact( #AVTF_MSal )
      wire#w1
      Contact( #Selec_M1_Salida )
      Coil( #AVTF_Sal_M1 )
   END_RUNG
   RUNG wire#w1
      Contact( #Selec_M2_Salida )
      Coil( #AVTF_Sal_M2 )
   END_RUNG
   RUNG wire#w1
      Contact( #Selec_M3_Salida )
      Coil( #AVTF_Sal_M3 )
   END_RUNG
   RUNG wire#w1
      Contact( #Selec_M4_Salida )
      Coil( #AVTF_Sal_M4 )
   END_RUNG
   // the same network as SCL:
   #AVTF_Sal_M1 := #AVTF_MSal AND #Selec_M1_Salida;
   #AVTF_Sal_M2 := #AVTF_MSal AND #Selec_M2_Salida;
   #AVTF_Sal_M3 := #AVTF_MSal AND #Selec_M3_Salida;
   #AVTF_Sal_M4 := #AVTF_MSal AND #Selec_M4_Salida;
END_REGION

REGION Network 121: MULTIPLEXADO FINAL SEÑALES DE SALIDA DE CARGA - P_Mens_MSal
   RUNG wire#powerrail
      Contact( #P_Mens_MSal )
      wire#w1
      Contact( #Selec_M1_Salida )
      Coil( #P_Mens_Sal_M1 )
   END_RUNG
   RUNG wire#w1
      Contact( #Selec_M2_Salida )
      Coil( #P_Mens_Sal_M2 )
   END_RUNG
   RUNG wire#w1
      Contact( #Selec_M3_Salida )
      Coil( #P_Mens_Sal_M3 )
   END_RUNG
   RUNG wire#w1
      Contact( #Selec_M4_Salida )
      Coil( #P_Mens_Sal_M4 )
   END_RUNG
   // the same network as SCL:
   #P_Mens_Sal_M1 := #P_Mens_MSal AND #Selec_M1_Salida;
   #P_Mens_Sal_M2 := #P_Mens_MSal AND #Selec_M2_Salida;
   #P_Mens_Sal_M3 := #P_Mens_MSal AND #Selec_M3_Salida;
   #P_Mens_Sal_M4 := #P_Mens_MSal AND #Selec_M4_Salida;
END_REGION

REGION Network 122: VARIABLES AUXILIRES - Memoria de DESREMONTADO
   // dani: 08/09/2018 reseteamos con eta60 y 61 para que no entre en etapa 95
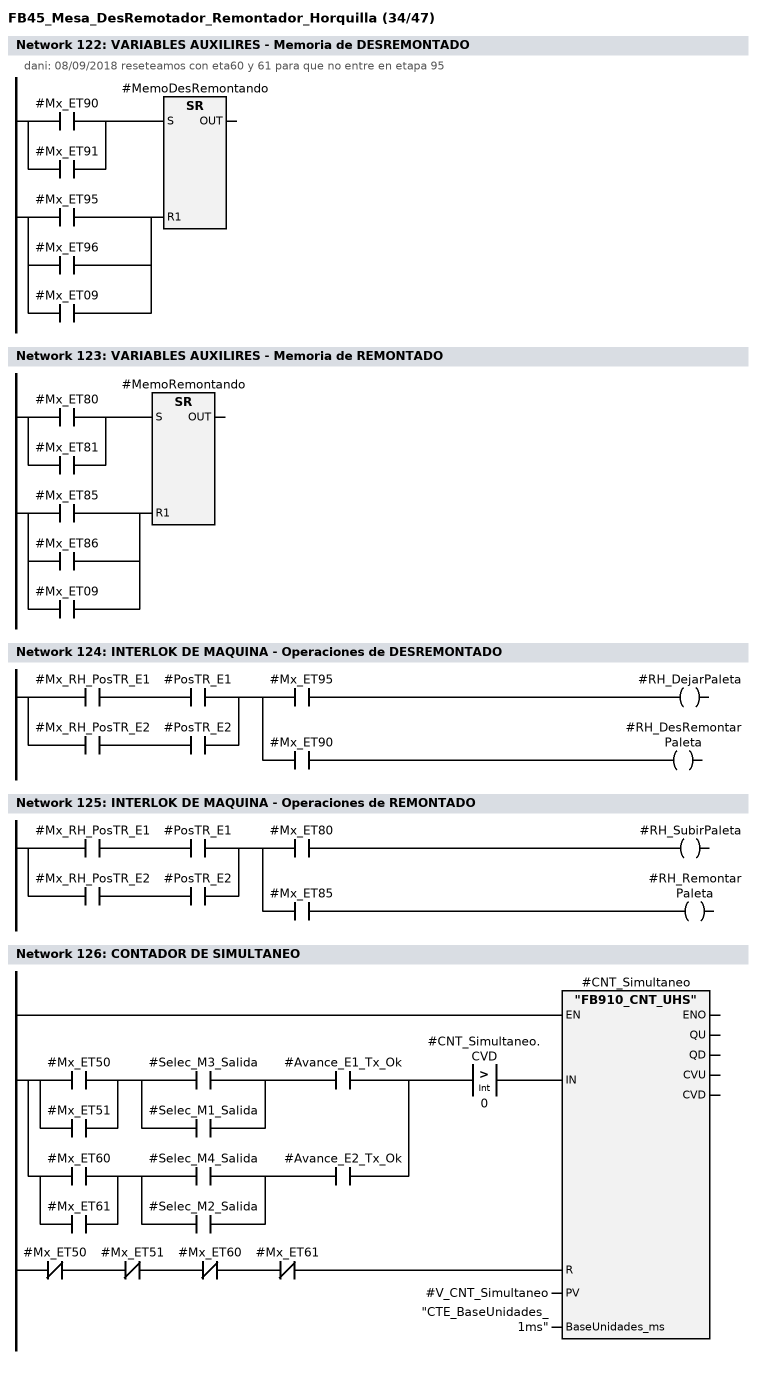
   RUNG wire#powerrail
      Contact( #Mx_ET90 )
      wire#w1
      S_SR(operand := #MemoDesRemontando, r1 := wire#w2)
   END_RUNG
   RUNG wire#powerrail
      Contact( #Mx_ET91 )
   END_RUNG wire#w1
   RUNG wire#powerrail
      Contact( #Mx_ET95 )
   END_RUNG wire#w2
   RUNG wire#powerrail
      Contact( #Mx_ET96 )
   END_RUNG wire#w2
   RUNG wire#powerrail
      Contact( #Mx_ET09 )
   END_RUNG wire#w2
   // the same network as SCL:
   IF #Mx_ET90 OR #Mx_ET91 THEN
       #MemoDesRemontando := TRUE;   // SR flip-flop
   END_IF;
   IF #Mx_ET95 OR #Mx_ET96 OR #Mx_ET09 THEN #MemoDesRemontando := FALSE; END_IF;
END_REGION

REGION Network 123: VARIABLES AUXILIRES - Memoria de REMONTADO
   RUNG wire#powerrail
      Contact( #Mx_ET80 )
      wire#w1
      S_SR(operand := #MemoRemontando, r1 := wire#w2)
   END_RUNG
   RUNG wire#powerrail
      Contact( #Mx_ET81 )
   END_RUNG wire#w1
   RUNG wire#powerrail
      Contact( #Mx_ET85 )
   END_RUNG wire#w2
   RUNG wire#powerrail
      Contact( #Mx_ET86 )
   END_RUNG wire#w2
   RUNG wire#powerrail
      Contact( #Mx_ET09 )
   END_RUNG wire#w2
   // the same network as SCL:
   IF #Mx_ET80 OR #Mx_ET81 THEN
       #MemoRemontando := TRUE;   // SR flip-flop
   END_IF;
   IF #Mx_ET85 OR #Mx_ET86 OR #Mx_ET09 THEN #MemoRemontando := FALSE; END_IF;
END_REGION

REGION Network 124: INTERLOK DE MAQUINA - Operaciones de DESREMONTADO
   RUNG wire#powerrail
      Contact( #Mx_RH_PosTR_E1 )
      Contact( #PosTR_E1 )
      wire#w1
      Contact( #Mx_ET95 )
      Coil( #RH_DejarPaleta )
   END_RUNG
   RUNG wire#powerrail
      Contact( #Mx_RH_PosTR_E2 )
      Contact( #PosTR_E2 )
   END_RUNG wire#w1
   RUNG wire#w1
      Contact( #Mx_ET90 )
      Coil( #RH_DesRemontarPaleta )
   END_RUNG
   // the same network as SCL:
   #_w1 := (#Mx_RH_PosTR_E1 AND #PosTR_E1) OR (#Mx_RH_PosTR_E2 AND #PosTR_E2);
   #RH_DejarPaleta := #_w1 AND #Mx_ET95;
   #RH_DesRemontarPaleta := #_w1 AND #Mx_ET90;
END_REGION

REGION Network 125: INTERLOK DE MAQUINA - Operaciones de REMONTADO
   RUNG wire#powerrail
      Contact( #Mx_RH_PosTR_E1 )
      Contact( #PosTR_E1 )
      wire#w1
      Contact( #Mx_ET80 )
      Coil( #RH_SubirPaleta )
   END_RUNG
   RUNG wire#powerrail
      Contact( #Mx_RH_PosTR_E2 )
      Contact( #PosTR_E2 )
   END_RUNG wire#w1
   RUNG wire#w1
      Contact( #Mx_ET85 )
      Coil( #RH_RemontarPaleta )
   END_RUNG
   // the same network as SCL:
   #_w1 := (#Mx_RH_PosTR_E1 AND #PosTR_E1) OR (#Mx_RH_PosTR_E2 AND #PosTR_E2);
   #RH_SubirPaleta := #_w1 AND #Mx_ET80;
   #RH_RemontarPaleta := #_w1 AND #Mx_ET85;
END_REGION

REGION Network 126: CONTADOR DE SIMULTANEO
   RUNG wire#powerrail
      #CNT_Simultaneo(IN := wire#w6, R := wire#w7, PV := #V_CNT_Simultaneo, BaseUnidades_ms := "CTE_BaseUnidades_1ms", QU =>, QD =>, CVU =>, CVD =>)
   END_RUNG
   RUNG wire#powerrail
      Contact( #Mx_ET50 )
      wire#w1
      Contact( #Selec_M3_Salida )
      wire#w2
      Contact( #Avance_E1_Tx_Ok )
      wire#w3
      { S7_Templates := "SrcType := Int" } GT_Contact(in1 := #CNT_Simultaneo.CVD, in2 := 0)
   END_RUNG wire#w6
   RUNG wire#powerrail
      Contact( #Mx_ET51 )
   END_RUNG wire#w1
   RUNG wire#w1
      Contact( #Selec_M1_Salida )
   END_RUNG wire#w2
   RUNG wire#powerrail
      Contact( #Mx_ET60 )
      wire#w4
      Contact( #Selec_M4_Salida )
      wire#w5
      Contact( #Avance_E2_Tx_Ok )
   END_RUNG wire#w3
   RUNG wire#powerrail
      Contact( #Mx_ET61 )
   END_RUNG wire#w4
   RUNG wire#w4
      Contact( #Selec_M2_Salida )
   END_RUNG wire#w5
   RUNG wire#powerrail
      I_Contact( #Mx_ET50 )
      I_Contact( #Mx_ET51 )
      I_Contact( #Mx_ET60 )
      I_Contact( #Mx_ET61 )
   END_RUNG wire#w7
   // the same network as SCL:
   #CNT_Simultaneo(IN := (((#Mx_ET50 OR #Mx_ET51) AND (#Selec_M3_Salida OR #Selec_M1_Salida) AND #Avance_E1_Tx_Ok) OR ((#Mx_ET60 OR #Mx_ET61) AND (#Selec_M4_Salida OR #Selec_M2_Salida) AND #Avance_E2_Tx_Ok)) AND (#CNT_Simultaneo.CVD > 0),   // "FB910_CNT_UHS"
                   R := NOT #Mx_ET50 AND NOT #Mx_ET51 AND NOT #Mx_ET60 AND NOT #Mx_ET61,
                   PV := #V_CNT_Simultaneo,
                   BaseUnidades_ms := "CTE_BaseUnidades_1ms");
END_REGION

REGION Network 127: CONTROL DE MOVIMIENTO SIMULTANEO
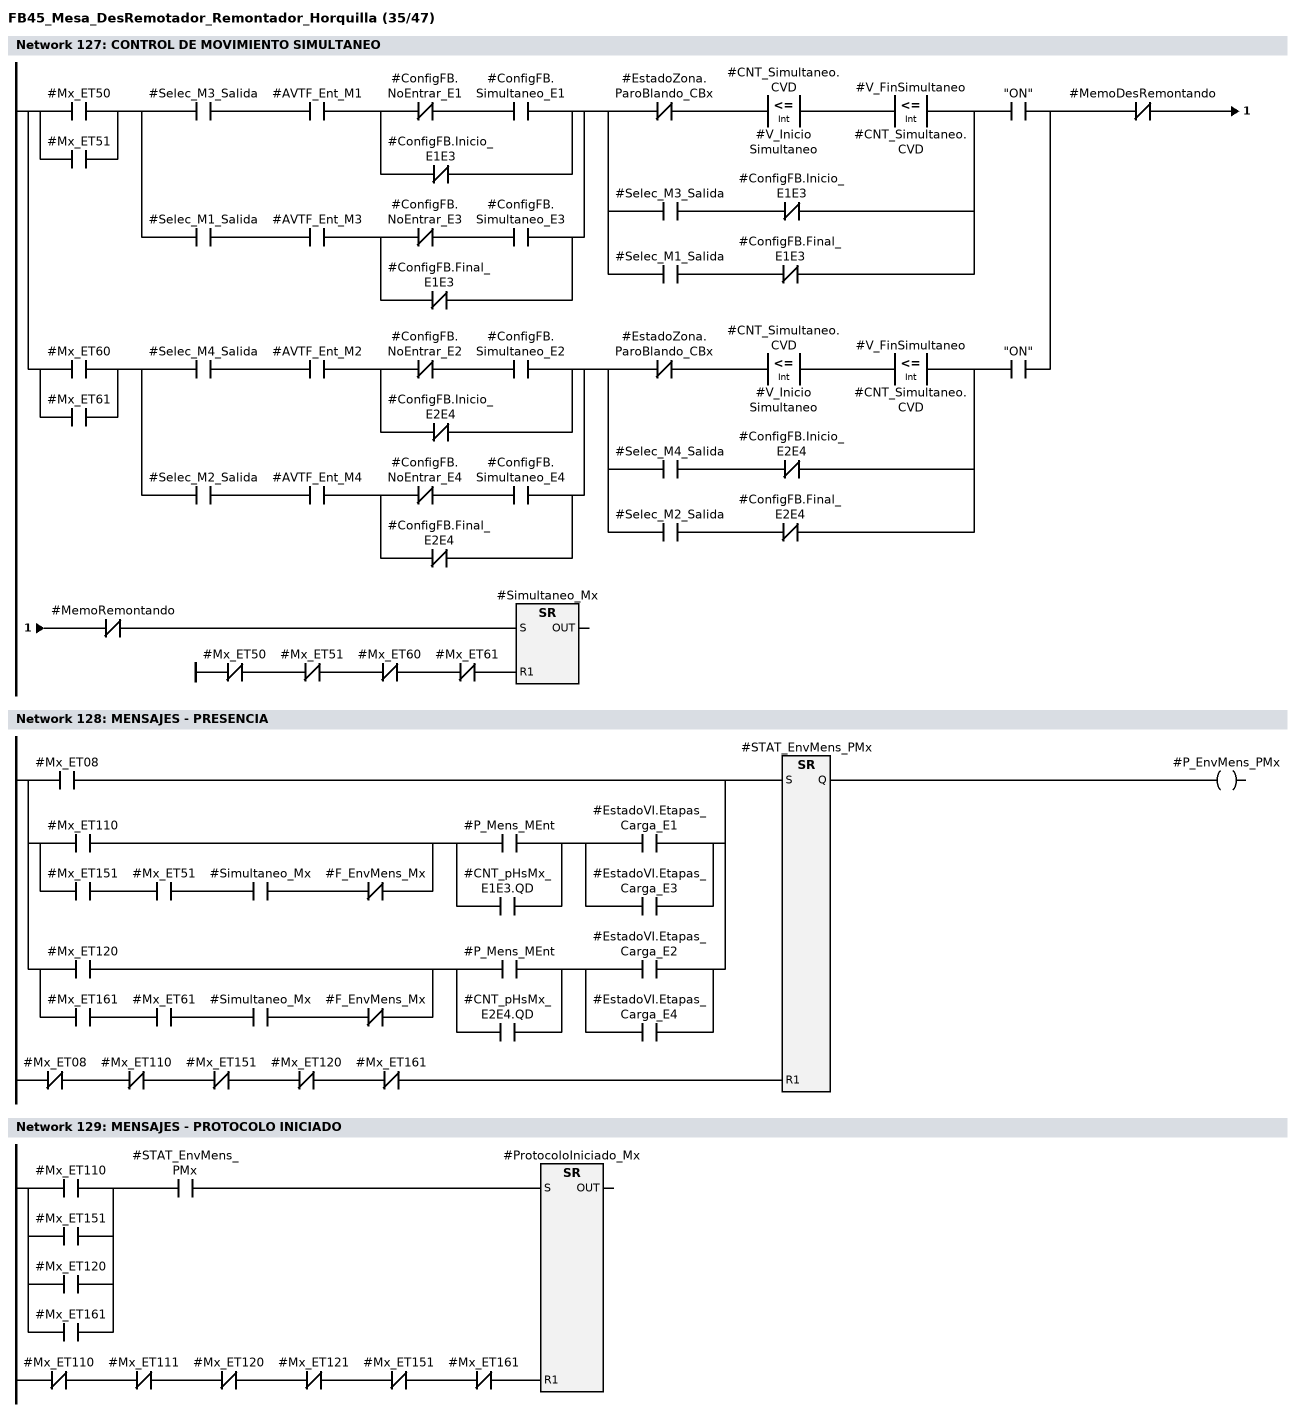
   RUNG wire#powerrail
      Contact( #Mx_ET50 )
      wire#w1
      Contact( #Selec_M3_Salida )
      Contact( #AVTF_Ent_M1 )
      wire#w2
      I_Contact( #ConfigFB.NoEntrar_E1 )
      Contact( #ConfigFB.Simultaneo_E1 )
      wire#w3
      I_Contact( #EstadoZona.ParoBlando_CBx )
      { S7_Templates := "SrcType := Int" } LE_Contact(in1 := #CNT_Simultaneo.CVD, in2 := #V_InicioSimultaneo)
      { S7_Templates := "SrcType := Int" } LE_Contact(in1 := #V_FinSimultaneo, in2 := #CNT_Simultaneo.CVD)
      wire#w5
      Contact( "ON" )
      wire#w6
      I_Contact( #MemoDesRemontando )
      I_Contact( #MemoRemontando )
      S_SR(operand := #Simultaneo_Mx, r1 := wire#w12)
   END_RUNG
   RUNG wire#powerrail
      Contact( #Mx_ET51 )
   END_RUNG wire#w1
   RUNG wire#w2
      I_Contact( #ConfigFB.Inicio_E1E3 )
   END_RUNG wire#w3
   RUNG wire#w1
      Contact( #Selec_M1_Salida )
      Contact( #AVTF_Ent_M3 )
      wire#w4
      I_Contact( #ConfigFB.NoEntrar_E3 )
      Contact( #ConfigFB.Simultaneo_E3 )
   END_RUNG wire#w3
   RUNG wire#w4
      I_Contact( #ConfigFB.Final_E1E3 )
   END_RUNG wire#w3
   RUNG wire#w3
      Contact( #Selec_M3_Salida )
      I_Contact( #ConfigFB.Inicio_E1E3 )
   END_RUNG wire#w5
   RUNG wire#w3
      Contact( #Selec_M1_Salida )
      I_Contact( #ConfigFB.Final_E1E3 )
   END_RUNG wire#w5
   RUNG wire#powerrail
      Contact( #Mx_ET60 )
      wire#w7
      Contact( #Selec_M4_Salida )
      Contact( #AVTF_Ent_M2 )
      wire#w8
      I_Contact( #ConfigFB.NoEntrar_E2 )
      Contact( #ConfigFB.Simultaneo_E2 )
      wire#w9
      I_Contact( #EstadoZona.ParoBlando_CBx )
      { S7_Templates := "SrcType := Int" } LE_Contact(in1 := #CNT_Simultaneo.CVD, in2 := #V_InicioSimultaneo)
      { S7_Templates := "SrcType := Int" } LE_Contact(in1 := #V_FinSimultaneo, in2 := #CNT_Simultaneo.CVD)
      wire#w11
      Contact( "ON" )
   END_RUNG wire#w6
   RUNG wire#powerrail
      Contact( #Mx_ET61 )
   END_RUNG wire#w7
   RUNG wire#w8
      I_Contact( #ConfigFB.Inicio_E2E4 )
   END_RUNG wire#w9
   RUNG wire#w7
      Contact( #Selec_M2_Salida )
      Contact( #AVTF_Ent_M4 )
      wire#w10
      I_Contact( #ConfigFB.NoEntrar_E4 )
      Contact( #ConfigFB.Simultaneo_E4 )
   END_RUNG wire#w9
   RUNG wire#w10
      I_Contact( #ConfigFB.Final_E2E4 )
   END_RUNG wire#w9
   RUNG wire#w9
      Contact( #Selec_M4_Salida )
      I_Contact( #ConfigFB.Inicio_E2E4 )
   END_RUNG wire#w11
   RUNG wire#w9
      Contact( #Selec_M2_Salida )
      I_Contact( #ConfigFB.Final_E2E4 )
   END_RUNG wire#w11
   RUNG wire#powerrail
      I_Contact( #Mx_ET50 )
      I_Contact( #Mx_ET51 )
      I_Contact( #Mx_ET60 )
      I_Contact( #Mx_ET61 )
   END_RUNG wire#w12
   // the same network as SCL:
   IF (((#Mx_ET50 OR #Mx_ET51) AND ((#Selec_M3_Salida AND #AVTF_Ent_M1 AND ((NOT #ConfigFB.NoEntrar_E1 AND #ConfigFB.Simultaneo_E1) OR NOT #ConfigFB.Inicio_E1E3)) OR (#Selec_M1_Salida AND #AVTF_Ent_M3 AND ((NOT #ConfigFB.NoEntrar_E3 AND #ConfigFB.Simultaneo_E3) OR NOT #ConfigFB.Final_E1E3))) AND ((NOT #EstadoZona.ParoBlando_CBx AND (#CNT_Simultaneo.CVD <= #V_InicioSimultaneo) AND (#V_FinSimultaneo <= #CNT_Simultaneo.CVD)) OR (#Selec_M3_Salida AND NOT #ConfigFB.Inicio_E1E3) OR (#Selec_M1_Salida AND NOT #ConfigFB.Final_E1E3)) AND "ON") OR ((#Mx_ET60 OR #Mx_ET61) AND ((#Selec_M4_Salida AND #AVTF_Ent_M2 AND ((NOT #ConfigFB.NoEntrar_E2 AND #ConfigFB.Simultaneo_E2) OR NOT #ConfigFB.Inicio_E2E4)) OR (#Selec_M2_Salida AND #AVTF_Ent_M4 AND ((NOT #ConfigFB.NoEntrar_E4 AND #ConfigFB.Simultaneo_E4) OR NOT #ConfigFB.Final_E2E4))) AND ((NOT #EstadoZona.ParoBlando_CBx AND (#CNT_Simultaneo.CVD <= #V_InicioSimultaneo) AND (#V_FinSimultaneo <= #CNT_Simultaneo.CVD)) OR (#Selec_M4_Salida AND NOT #ConfigFB.Inicio_E2E4) OR (#Selec_M2_Salida AND NOT #ConfigFB.Final_E2E4)) AND "ON")) AND NOT #MemoDesRemontando AND NOT #MemoRemontando THEN
       #Simultaneo_Mx := TRUE;   // SR flip-flop
   END_IF;
   IF NOT #Mx_ET50 AND NOT #Mx_ET51 AND NOT #Mx_ET60 AND NOT #Mx_ET61 THEN #Simultaneo_Mx := FALSE; END_IF;
END_REGION

REGION Network 128: MENSAJES - PRESENCIA
   RUNG wire#powerrail
      Contact( #Mx_ET08 )
      wire#w1
      S_SR(operand := #STAT_EnvMens_PMx, r1 := wire#w6)
      Coil( #P_EnvMens_PMx )
   END_RUNG
   RUNG wire#powerrail
      Contact( #Mx_ET110 )
      wire#w2
      Contact( #P_Mens_MEnt )
      wire#w3
      Contact( #EstadoVI.Etapas_Carga_E1 )
   END_RUNG wire#w1
   RUNG wire#powerrail
      Contact( #Mx_ET151 )
      Contact( #Mx_ET51 )
      Contact( #Simultaneo_Mx )
      I_Contact( #F_EnvMens_Mx )
   END_RUNG wire#w2
   RUNG wire#w2
      Contact( #CNT_pHsMx_E1E3.QD )
   END_RUNG wire#w3
   RUNG wire#w3
      Contact( #EstadoVI.Etapas_Carga_E3 )
   END_RUNG wire#w1
   RUNG wire#powerrail
      Contact( #Mx_ET120 )
      wire#w4
      Contact( #P_Mens_MEnt )
      wire#w5
      Contact( #EstadoVI.Etapas_Carga_E2 )
   END_RUNG wire#w1
   RUNG wire#powerrail
      Contact( #Mx_ET161 )
      Contact( #Mx_ET61 )
      Contact( #Simultaneo_Mx )
      I_Contact( #F_EnvMens_Mx )
   END_RUNG wire#w4
   RUNG wire#w4
      Contact( #CNT_pHsMx_E2E4.QD )
   END_RUNG wire#w5
   RUNG wire#w5
      Contact( #EstadoVI.Etapas_Carga_E4 )
   END_RUNG wire#w1
   RUNG wire#powerrail
      I_Contact( #Mx_ET08 )
      I_Contact( #Mx_ET110 )
      I_Contact( #Mx_ET151 )
      I_Contact( #Mx_ET120 )
      I_Contact( #Mx_ET161 )
   END_RUNG wire#w6
   // the same network as SCL:
   IF #Mx_ET08 OR ((#Mx_ET110 OR (#Mx_ET151 AND #Mx_ET51 AND #Simultaneo_Mx AND NOT #F_EnvMens_Mx)) AND (#P_Mens_MEnt OR #CNT_pHsMx_E1E3.QD) AND (#EstadoVI.Etapas_Carga_E1 OR #EstadoVI.Etapas_Carga_E3)) OR ((#Mx_ET120 OR (#Mx_ET161 AND #Mx_ET61 AND #Simultaneo_Mx AND NOT #F_EnvMens_Mx)) AND (#P_Mens_MEnt OR #CNT_pHsMx_E2E4.QD) AND (#EstadoVI.Etapas_Carga_E2 OR #EstadoVI.Etapas_Carga_E4)) THEN
       #STAT_EnvMens_PMx := TRUE;   // SR flip-flop
   END_IF;
   IF NOT #Mx_ET08 AND NOT #Mx_ET110 AND NOT #Mx_ET151 AND NOT #Mx_ET120 AND NOT #Mx_ET161 THEN
       #STAT_EnvMens_PMx := FALSE;
   END_IF;
   #P_EnvMens_PMx := #STAT_EnvMens_PMx;
END_REGION

REGION Network 129: MENSAJES - PROTOCOLO INICIADO
   RUNG wire#powerrail
      Contact( #Mx_ET110 )
      wire#w1
      Contact( #STAT_EnvMens_PMx )
      S_SR(operand := #ProtocoloIniciado_Mx, r1 := wire#w2)
   END_RUNG
   RUNG wire#powerrail
      Contact( #Mx_ET151 )
   END_RUNG wire#w1
   RUNG wire#powerrail
      Contact( #Mx_ET120 )
   END_RUNG wire#w1
   RUNG wire#powerrail
      Contact( #Mx_ET161 )
   END_RUNG wire#w1
   RUNG wire#powerrail
      I_Contact( #Mx_ET110 )
      I_Contact( #Mx_ET111 )
      I_Contact( #Mx_ET120 )
      I_Contact( #Mx_ET121 )
      I_Contact( #Mx_ET151 )
      I_Contact( #Mx_ET161 )
   END_RUNG wire#w2
   // the same network as SCL:
   IF (#Mx_ET110 OR #Mx_ET151 OR #Mx_ET120 OR #Mx_ET161) AND #STAT_EnvMens_PMx THEN
       #ProtocoloIniciado_Mx := TRUE;   // SR flip-flop
   END_IF;
   IF NOT #Mx_ET110 AND NOT #Mx_ET111 AND NOT #Mx_ET120 AND NOT #Mx_ET121 AND NOT #Mx_ET151 AND NOT #Mx_ET161 THEN
       #ProtocoloIniciado_Mx := FALSE;
   END_IF;
END_REGION

REGION Network 130: MENSAJES - BLOQUEO
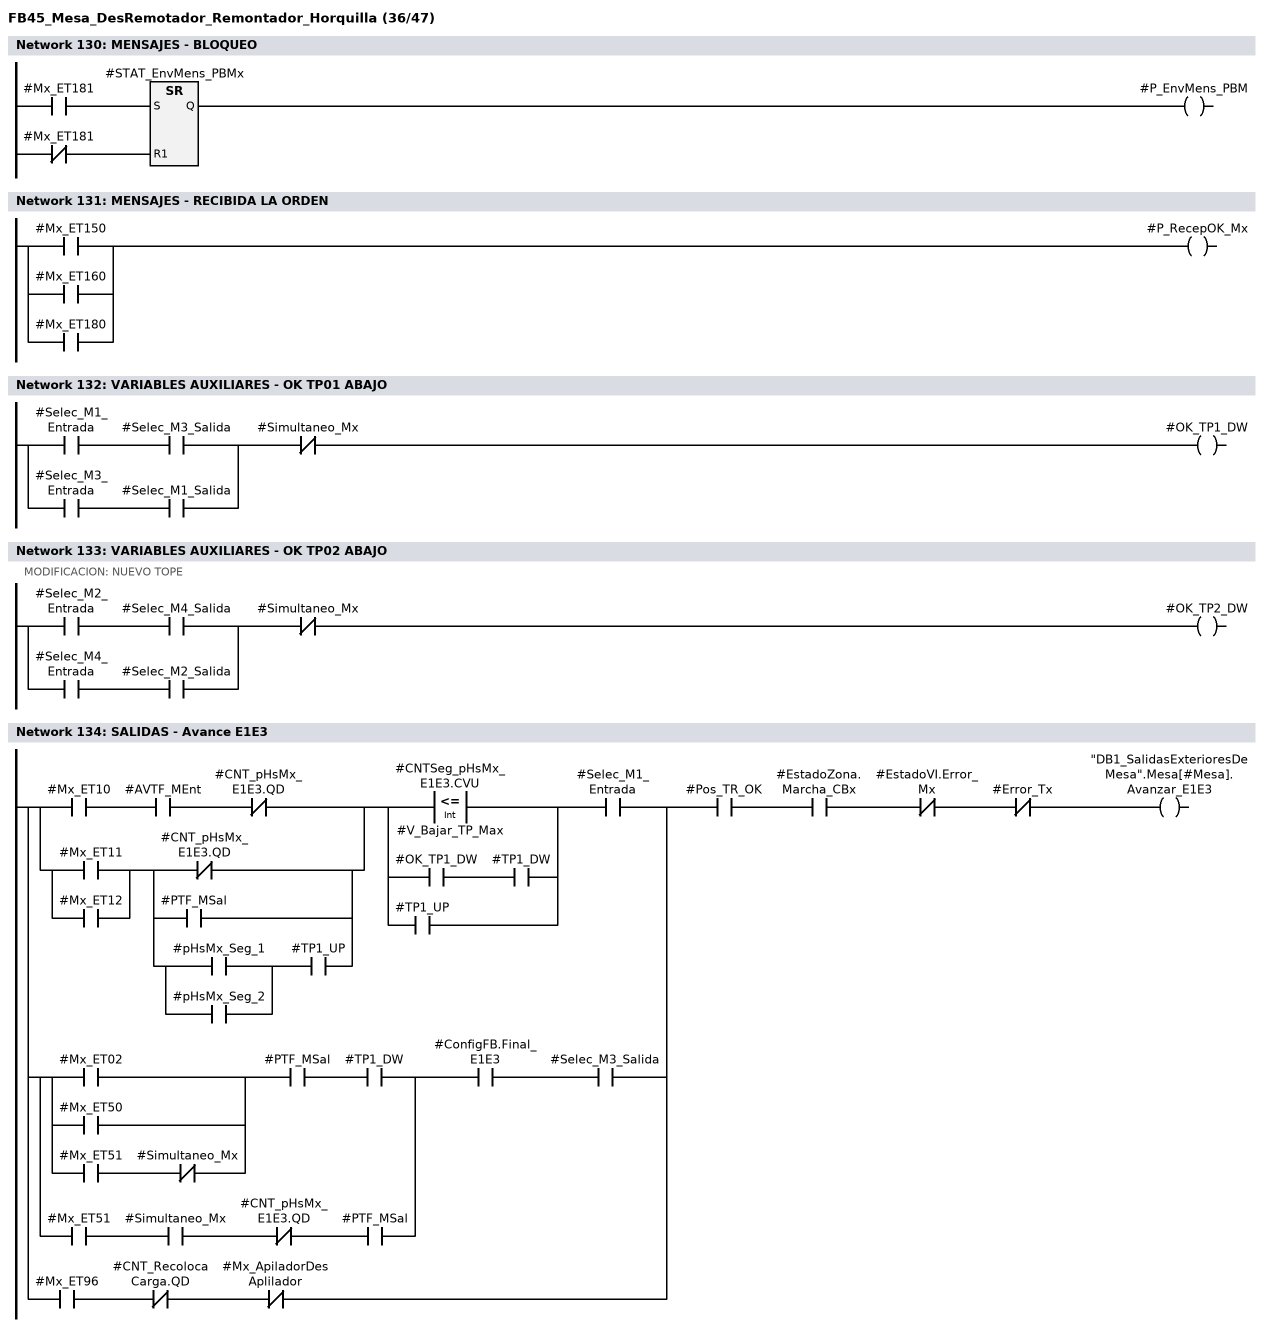
   RUNG wire#powerrail
      Contact( #Mx_ET181 )
      S_SR(operand := #STAT_EnvMens_PBMx, r1 := wire#w1)
      Coil( #P_EnvMens_PBM )
   END_RUNG
   RUNG wire#powerrail
      I_Contact( #Mx_ET181 )
   END_RUNG wire#w1
   // the same network as SCL:
   IF #Mx_ET181 THEN
       #STAT_EnvMens_PBMx := TRUE;   // SR flip-flop
   END_IF;
   IF NOT #Mx_ET181 THEN #STAT_EnvMens_PBMx := FALSE; END_IF;
   #P_EnvMens_PBM := #STAT_EnvMens_PBMx;
END_REGION

REGION Network 131: MENSAJES - RECIBIDA LA ORDEN
   RUNG wire#powerrail
      Contact( #Mx_ET150 )
      wire#w1
      Coil( #P_RecepOK_Mx )
   END_RUNG
   RUNG wire#powerrail
      Contact( #Mx_ET160 )
   END_RUNG wire#w1
   RUNG wire#powerrail
      Contact( #Mx_ET180 )
   END_RUNG wire#w1
   // the same network as SCL:
   #P_RecepOK_Mx := #Mx_ET150 OR #Mx_ET160 OR #Mx_ET180;
END_REGION

REGION Network 132: VARIABLES AUXILIARES - OK TP01 ABAJO
   RUNG wire#powerrail
      Contact( #Selec_M1_Entrada )
      Contact( #Selec_M3_Salida )
      wire#w1
      I_Contact( #Simultaneo_Mx )
      Coil( #OK_TP1_DW )
   END_RUNG
   RUNG wire#powerrail
      Contact( #Selec_M3_Entrada )
      Contact( #Selec_M1_Salida )
   END_RUNG wire#w1
   // the same network as SCL:
   #OK_TP1_DW := ((#Selec_M1_Entrada AND #Selec_M3_Salida) OR (#Selec_M3_Entrada AND #Selec_M1_Salida)) AND NOT #Simultaneo_Mx;
END_REGION

REGION Network 133: VARIABLES AUXILIARES - OK TP02 ABAJO
   // MODIFICACION: NUEVO TOPE
   RUNG wire#powerrail
      Contact( #Selec_M2_Entrada )
      Contact( #Selec_M4_Salida )
      wire#w1
      I_Contact( #Simultaneo_Mx )
      Coil( #OK_TP2_DW )
   END_RUNG
   RUNG wire#powerrail
      Contact( #Selec_M4_Entrada )
      Contact( #Selec_M2_Salida )
   END_RUNG wire#w1
   // the same network as SCL:
   #OK_TP2_DW := ((#Selec_M2_Entrada AND #Selec_M4_Salida) OR (#Selec_M4_Entrada AND #Selec_M2_Salida)) AND NOT #Simultaneo_Mx;
END_REGION

REGION Network 134: SALIDAS - Avance E1E3
   RUNG wire#powerrail
      Contact( #Mx_ET10 )
      Contact( #AVTF_MEnt )
      I_Contact( #CNT_pHsMx_E1E3.QD )
      wire#w1
      { S7_Templates := "SrcType := Int" } LE_Contact(in1 := #CNTSeg_pHsMx_E1E3.CVU, in2 := #V_Bajar_TP_Max)
      wire#w4
      Contact( #Selec_M1_Entrada )
      wire#w5
      Contact( #Pos_TR_OK )
      Contact( #EstadoZona.Marcha_CBx )
      I_Contact( #EstadoVI.Error_Mx )
      I_Contact( #Error_Tx )
      Coil( "DB1_SalidasExterioresDeMesa".Mesa[#Mesa].Avanzar_E1E3 )
   END_RUNG
   RUNG wire#powerrail
      Contact( #Mx_ET11 )
      wire#w2
      I_Contact( #CNT_pHsMx_E1E3.QD )
   END_RUNG wire#w1
   RUNG wire#powerrail
      Contact( #Mx_ET12 )
   END_RUNG wire#w2
   RUNG wire#w2
      Contact( #PTF_MSal )
   END_RUNG wire#w1
   RUNG wire#w2
      Contact( #pHsMx_Seg_1 )
      wire#w3
      Contact( #TP1_UP )
   END_RUNG wire#w1
   RUNG wire#w2
      Contact( #pHsMx_Seg_2 )
   END_RUNG wire#w3
   RUNG wire#w1
      Contact( #OK_TP1_DW )
      Contact( #TP1_DW )
   END_RUNG wire#w4
   RUNG wire#w1
      Contact( #TP1_UP )
   END_RUNG wire#w4
   RUNG wire#powerrail
      Contact( #Mx_ET02 )
      wire#w6
      Contact( #PTF_MSal )
      Contact( #TP1_DW )
      wire#w7
      Contact( #ConfigFB.Final_E1E3 )
      Contact( #Selec_M3_Salida )
   END_RUNG wire#w5
   RUNG wire#powerrail
      Contact( #Mx_ET50 )
   END_RUNG wire#w6
   RUNG wire#powerrail
      Contact( #Mx_ET51 )
      I_Contact( #Simultaneo_Mx )
   END_RUNG wire#w6
   RUNG wire#powerrail
      Contact( #Mx_ET51 )
      Contact( #Simultaneo_Mx )
      I_Contact( #CNT_pHsMx_E1E3.QD )
      Contact( #PTF_MSal )
   END_RUNG wire#w7
   RUNG wire#powerrail
      Contact( #Mx_ET96 )
      I_Contact( #CNT_RecolocaCarga.QD )
      I_Contact( #Mx_ApiladorDesAplilador )
   END_RUNG wire#w5
   // the same network as SCL:
   "DB1_SalidasExterioresDeMesa".Mesa[#Mesa].Avanzar_E1E3 := ((((#Mx_ET10 AND #AVTF_MEnt AND NOT #CNT_pHsMx_E1E3.QD) OR ((#Mx_ET11 OR #Mx_ET12) AND (NOT #CNT_pHsMx_E1E3.QD OR #PTF_MSal OR ((#pHsMx_Seg_1 OR #pHsMx_Seg_2) AND #TP1_UP)))) AND ((#CNTSeg_pHsMx_E1E3.CVU <= #V_Bajar_TP_Max) OR (#OK_TP1_DW AND #TP1_DW) OR #TP1_UP) AND #Selec_M1_Entrada) OR ((((#Mx_ET02 OR #Mx_ET50 OR (#Mx_ET51 AND NOT #Simultaneo_Mx)) AND #PTF_MSal AND #TP1_DW) OR (#Mx_ET51 AND #Simultaneo_Mx AND NOT #CNT_pHsMx_E1E3.QD AND #PTF_MSal)) AND #ConfigFB.Final_E1E3 AND #Selec_M3_Salida) OR (#Mx_ET96 AND NOT #CNT_RecolocaCarga.QD AND NOT #Mx_ApiladorDesAplilador)) AND #Pos_TR_OK AND #EstadoZona.Marcha_CBx AND NOT #EstadoVI.Error_Mx AND NOT #Error_Tx;
END_REGION

REGION Network 135: SALIDAS - Retroceso E1E3
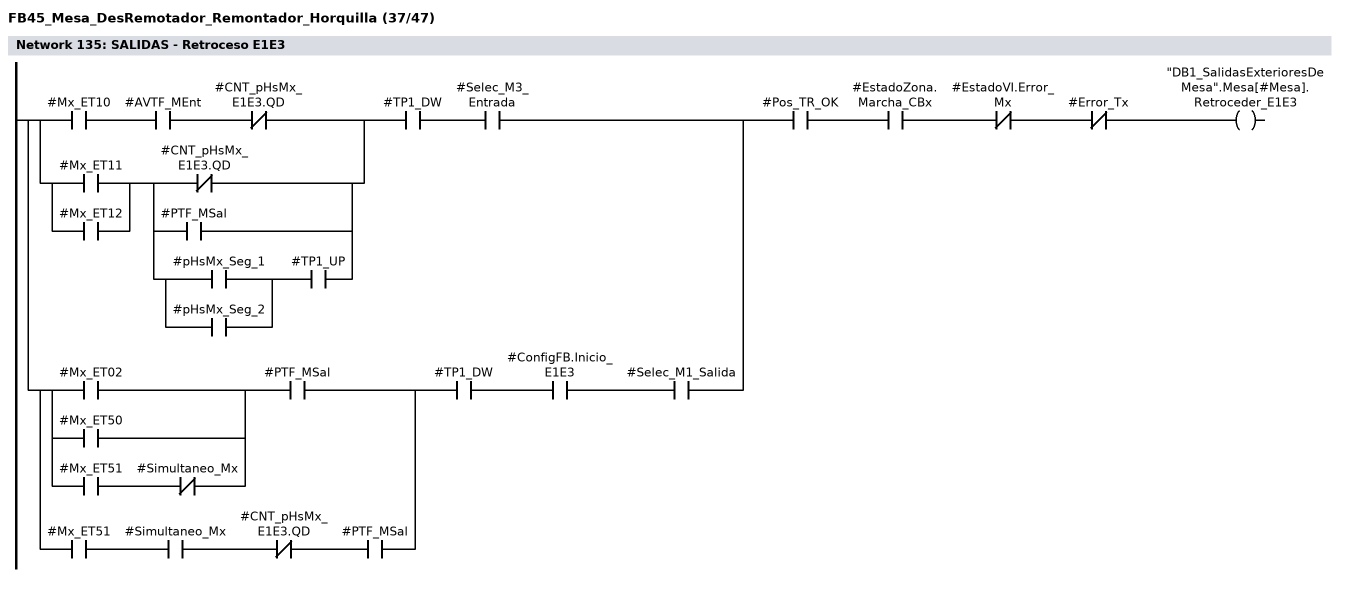
   RUNG wire#powerrail
      Contact( #Mx_ET10 )
      Contact( #AVTF_MEnt )
      I_Contact( #CNT_pHsMx_E1E3.QD )
      wire#w1
      Contact( #TP1_DW )
      Contact( #Selec_M3_Entrada )
      wire#w4
      Contact( #Pos_TR_OK )
      Contact( #EstadoZona.Marcha_CBx )
      I_Contact( #EstadoVI.Error_Mx )
      I_Contact( #Error_Tx )
      Coil( "DB1_SalidasExterioresDeMesa".Mesa[#Mesa].Retroceder_E1E3 )
   END_RUNG
   RUNG wire#powerrail
      Contact( #Mx_ET11 )
      wire#w2
      I_Contact( #CNT_pHsMx_E1E3.QD )
   END_RUNG wire#w1
   RUNG wire#powerrail
      Contact( #Mx_ET12 )
   END_RUNG wire#w2
   RUNG wire#w2
      Contact( #PTF_MSal )
   END_RUNG wire#w1
   RUNG wire#w2
      Contact( #pHsMx_Seg_1 )
      wire#w3
      Contact( #TP1_UP )
   END_RUNG wire#w1
   RUNG wire#w2
      Contact( #pHsMx_Seg_2 )
   END_RUNG wire#w3
   RUNG wire#powerrail
      Contact( #Mx_ET02 )
      wire#w5
      Contact( #PTF_MSal )
      wire#w6
      Contact( #TP1_DW )
      Contact( #ConfigFB.Inicio_E1E3 )
      Contact( #Selec_M1_Salida )
   END_RUNG wire#w4
   RUNG wire#powerrail
      Contact( #Mx_ET50 )
   END_RUNG wire#w5
   RUNG wire#powerrail
      Contact( #Mx_ET51 )
      I_Contact( #Simultaneo_Mx )
   END_RUNG wire#w5
   RUNG wire#powerrail
      Contact( #Mx_ET51 )
      Contact( #Simultaneo_Mx )
      I_Contact( #CNT_pHsMx_E1E3.QD )
      Contact( #PTF_MSal )
   END_RUNG wire#w6
   // the same network as SCL:
   "DB1_SalidasExterioresDeMesa".Mesa[#Mesa].Retroceder_E1E3 := ((((#Mx_ET10 AND #AVTF_MEnt AND NOT #CNT_pHsMx_E1E3.QD) OR ((#Mx_ET11 OR #Mx_ET12) AND (NOT #CNT_pHsMx_E1E3.QD OR #PTF_MSal OR ((#pHsMx_Seg_1 OR #pHsMx_Seg_2) AND #TP1_UP)))) AND #TP1_DW AND #Selec_M3_Entrada) OR ((((#Mx_ET02 OR #Mx_ET50 OR (#Mx_ET51 AND NOT #Simultaneo_Mx)) AND #PTF_MSal) OR (#Mx_ET51 AND #Simultaneo_Mx AND NOT #CNT_pHsMx_E1E3.QD AND #PTF_MSal)) AND #TP1_DW AND #ConfigFB.Inicio_E1E3 AND #Selec_M1_Salida)) AND #Pos_TR_OK AND #EstadoZona.Marcha_CBx AND NOT #EstadoVI.Error_Mx AND NOT #Error_Tx;
END_REGION

REGION Network 136: SALIDAS - Parar E1E3 // MODIFICADO
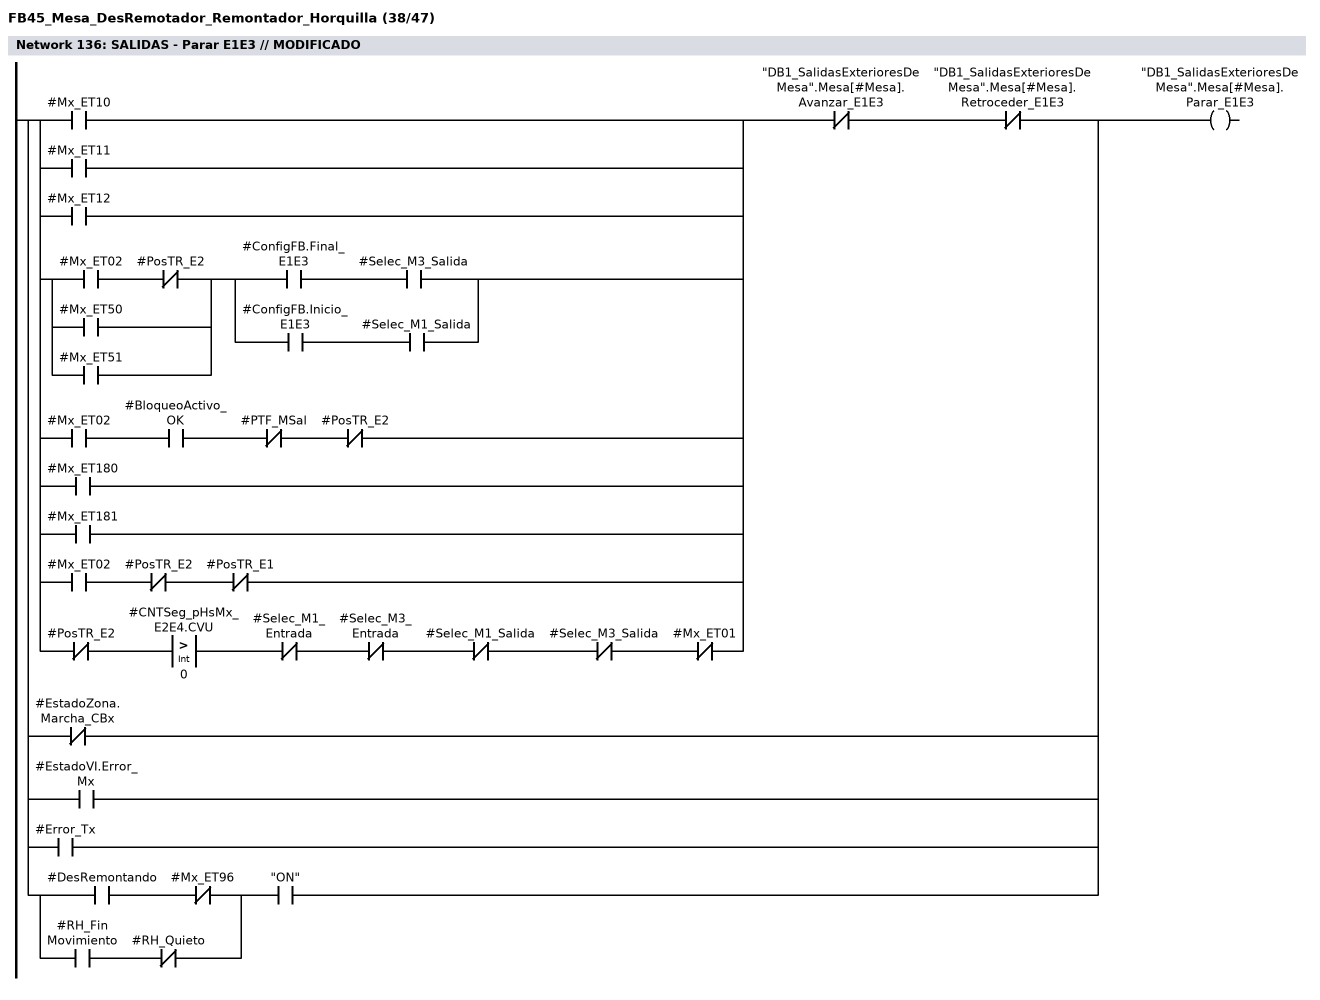
   RUNG wire#powerrail
      Contact( #Mx_ET10 )
      wire#w1
      I_Contact( "DB1_SalidasExterioresDeMesa".Mesa[#Mesa].Avanzar_E1E3 )
      I_Contact( "DB1_SalidasExterioresDeMesa".Mesa[#Mesa].Retroceder_E1E3 )
      wire#w3
      Coil( "DB1_SalidasExterioresDeMesa".Mesa[#Mesa].Parar_E1E3 )
   END_RUNG
   RUNG wire#powerrail
      Contact( #Mx_ET11 )
   END_RUNG wire#w1
   RUNG wire#powerrail
      Contact( #Mx_ET12 )
   END_RUNG wire#w1
   RUNG wire#powerrail
      Contact( #Mx_ET02 )
      I_Contact( #PosTR_E2 )
      wire#w2
      Contact( #ConfigFB.Final_E1E3 )
      Contact( #Selec_M3_Salida )
   END_RUNG wire#w1
   RUNG wire#powerrail
      Contact( #Mx_ET50 )
   END_RUNG wire#w2
   RUNG wire#powerrail
      Contact( #Mx_ET51 )
   END_RUNG wire#w2
   RUNG wire#w2
      Contact( #ConfigFB.Inicio_E1E3 )
      Contact( #Selec_M1_Salida )
   END_RUNG wire#w1
   RUNG wire#powerrail
      Contact( #Mx_ET02 )
      Contact( #BloqueoActivo_OK )
      I_Contact( #PTF_MSal )
      I_Contact( #PosTR_E2 )
   END_RUNG wire#w1
   RUNG wire#powerrail
      Contact( #Mx_ET180 )
   END_RUNG wire#w1
   RUNG wire#powerrail
      Contact( #Mx_ET181 )
   END_RUNG wire#w1
   RUNG wire#powerrail
      Contact( #Mx_ET02 )
      I_Contact( #PosTR_E2 )
      I_Contact( #PosTR_E1 )
   END_RUNG wire#w1
   RUNG wire#powerrail
      I_Contact( #PosTR_E2 )
      { S7_Templates := "SrcType := Int" } GT_Contact(in1 := #CNTSeg_pHsMx_E2E4.CVU, in2 := 0)
      I_Contact( #Selec_M1_Entrada )
      I_Contact( #Selec_M3_Entrada )
      I_Contact( #Selec_M1_Salida )
      I_Contact( #Selec_M3_Salida )
      I_Contact( #Mx_ET01 )
   END_RUNG wire#w1
   RUNG wire#powerrail
      I_Contact( #EstadoZona.Marcha_CBx )
   END_RUNG wire#w3
   RUNG wire#powerrail
      Contact( #EstadoVI.Error_Mx )
   END_RUNG wire#w3
   RUNG wire#powerrail
      Contact( #Error_Tx )
   END_RUNG wire#w3
   RUNG wire#powerrail
      Contact( #DesRemontando )
      I_Contact( #Mx_ET96 )
      wire#w4
      Contact( "ON" )
   END_RUNG wire#w3
   RUNG wire#powerrail
      Contact( #RH_FinMovimiento )
      I_Contact( #RH_Quieto )
   END_RUNG wire#w4
   // the same network as SCL:
   "DB1_SalidasExterioresDeMesa".Mesa[#Mesa].Parar_E1E3 := ((#Mx_ET10 OR #Mx_ET11 OR #Mx_ET12 OR (((#Mx_ET02 AND NOT #PosTR_E2) OR #Mx_ET50 OR #Mx_ET51) AND ((#ConfigFB.Final_E1E3 AND #Selec_M3_Salida) OR (#ConfigFB.Inicio_E1E3 AND #Selec_M1_Salida))) OR (#Mx_ET02 AND #BloqueoActivo_OK AND NOT #PTF_MSal AND NOT #PosTR_E2) OR #Mx_ET180 OR #Mx_ET181 OR (#Mx_ET02 AND NOT #PosTR_E2 AND NOT #PosTR_E1) OR (NOT #PosTR_E2 AND (#CNTSeg_pHsMx_E2E4.CVU > 0) AND NOT #Selec_M1_Entrada AND NOT #Selec_M3_Entrada AND NOT #Selec_M1_Salida AND NOT #Selec_M3_Salida AND NOT #Mx_ET01)) AND NOT "DB1_SalidasExterioresDeMesa".Mesa[#Mesa].Avanzar_E1E3 AND NOT "DB1_SalidasExterioresDeMesa".Mesa[#Mesa].Retroceder_E1E3) OR NOT #EstadoZona.Marcha_CBx OR #EstadoVI.Error_Mx OR #Error_Tx OR (((#DesRemontando AND NOT #Mx_ET96) OR (#RH_FinMovimiento AND NOT #RH_Quieto)) AND "ON");
END_REGION

REGION Network 137: SALIDAS - Valor Frecuencia Lenta E1E3
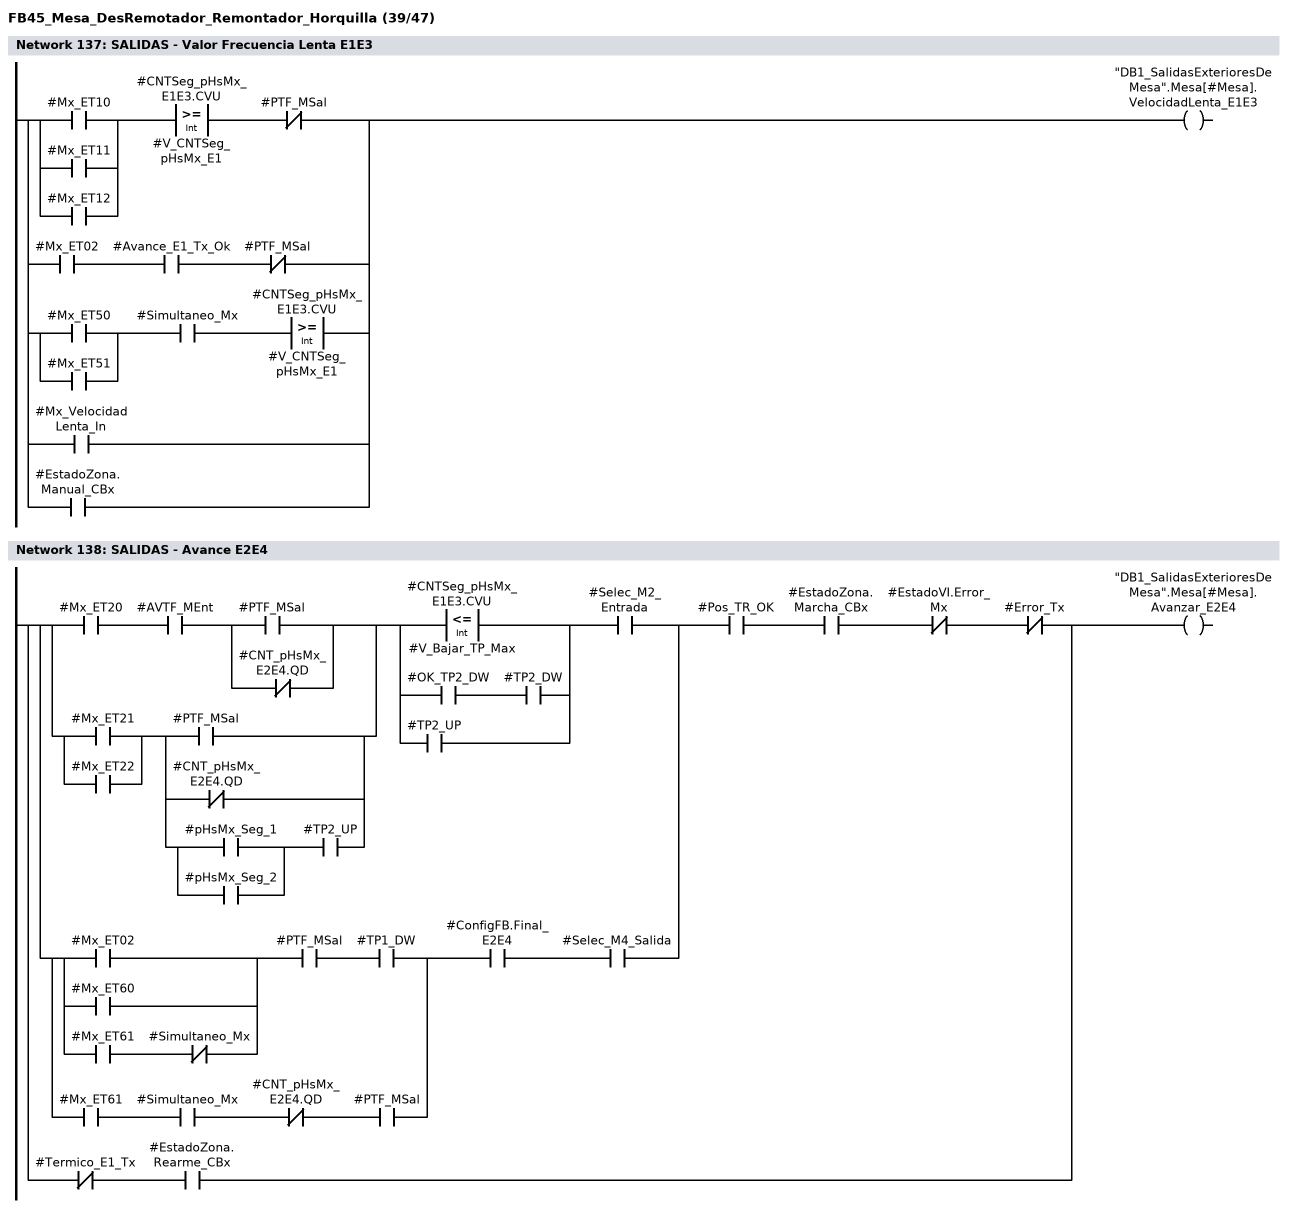
   RUNG wire#powerrail
      Contact( #Mx_ET10 )
      wire#w1
      { S7_Templates := "SrcType := Int" } GE_Contact(in1 := #CNTSeg_pHsMx_E1E3.CVU, in2 := #V_CNTSeg_pHsMx_E1)
      I_Contact( #PTF_MSal )
      wire#w2
      Coil( "DB1_SalidasExterioresDeMesa".Mesa[#Mesa].VelocidadLenta_E1E3 )
   END_RUNG
   RUNG wire#powerrail
      Contact( #Mx_ET11 )
   END_RUNG wire#w1
   RUNG wire#powerrail
      Contact( #Mx_ET12 )
   END_RUNG wire#w1
   RUNG wire#powerrail
      Contact( #Mx_ET02 )
      Contact( #Avance_E1_Tx_Ok )
      I_Contact( #PTF_MSal )
   END_RUNG wire#w2
   RUNG wire#powerrail
      Contact( #Mx_ET50 )
      wire#w3
      Contact( #Simultaneo_Mx )
      { S7_Templates := "SrcType := Int" } GE_Contact(in1 := #CNTSeg_pHsMx_E1E3.CVU, in2 := #V_CNTSeg_pHsMx_E1)
   END_RUNG wire#w2
   RUNG wire#powerrail
      Contact( #Mx_ET51 )
   END_RUNG wire#w3
   RUNG wire#powerrail
      Contact( #Mx_VelocidadLenta_In )
   END_RUNG wire#w2
   RUNG wire#powerrail
      Contact( #EstadoZona.Manual_CBx )
   END_RUNG wire#w2
   // the same network as SCL:
   "DB1_SalidasExterioresDeMesa".Mesa[#Mesa].VelocidadLenta_E1E3 := ((#Mx_ET10 OR #Mx_ET11 OR #Mx_ET12) AND (#CNTSeg_pHsMx_E1E3.CVU >= #V_CNTSeg_pHsMx_E1) AND NOT #PTF_MSal) OR (#Mx_ET02 AND #Avance_E1_Tx_Ok AND NOT #PTF_MSal) OR ((#Mx_ET50 OR #Mx_ET51) AND #Simultaneo_Mx AND (#CNTSeg_pHsMx_E1E3.CVU >= #V_CNTSeg_pHsMx_E1)) OR #Mx_VelocidadLenta_In OR #EstadoZona.Manual_CBx;
END_REGION

REGION Network 138: SALIDAS - Avance E2E4
   RUNG wire#powerrail
      Contact( #Mx_ET20 )
      Contact( #AVTF_MEnt )
      wire#w1
      Contact( #PTF_MSal )
      wire#w2
      { S7_Templates := "SrcType := Int" } LE_Contact(in1 := #CNTSeg_pHsMx_E1E3.CVU, in2 := #V_Bajar_TP_Max)
      wire#w5
      Contact( #Selec_M2_Entrada )
      wire#w6
      Contact( #Pos_TR_OK )
      Contact( #EstadoZona.Marcha_CBx )
      I_Contact( #EstadoVI.Error_Mx )
      I_Contact( #Error_Tx )
      wire#w9
      Coil( "DB1_SalidasExterioresDeMesa".Mesa[#Mesa].Avanzar_E2E4 )
   END_RUNG
   RUNG wire#w1
      I_Contact( #CNT_pHsMx_E2E4.QD )
   END_RUNG wire#w2
   RUNG wire#powerrail
      Contact( #Mx_ET21 )
      wire#w3
      Contact( #PTF_MSal )
   END_RUNG wire#w2
   RUNG wire#powerrail
      Contact( #Mx_ET22 )
   END_RUNG wire#w3
   RUNG wire#w3
      I_Contact( #CNT_pHsMx_E2E4.QD )
   END_RUNG wire#w2
   RUNG wire#w3
      Contact( #pHsMx_Seg_1 )
      wire#w4
      Contact( #TP2_UP )
   END_RUNG wire#w2
   RUNG wire#w3
      Contact( #pHsMx_Seg_2 )
   END_RUNG wire#w4
   RUNG wire#w2
      Contact( #OK_TP2_DW )
      Contact( #TP2_DW )
   END_RUNG wire#w5
   RUNG wire#w2
      Contact( #TP2_UP )
   END_RUNG wire#w5
   RUNG wire#powerrail
      Contact( #Mx_ET02 )
      wire#w7
      Contact( #PTF_MSal )
      Contact( #TP1_DW )
      wire#w8
      Contact( #ConfigFB.Final_E2E4 )
      Contact( #Selec_M4_Salida )
   END_RUNG wire#w6
   RUNG wire#powerrail
      Contact( #Mx_ET60 )
   END_RUNG wire#w7
   RUNG wire#powerrail
      Contact( #Mx_ET61 )
      I_Contact( #Simultaneo_Mx )
   END_RUNG wire#w7
   RUNG wire#powerrail
      Contact( #Mx_ET61 )
      Contact( #Simultaneo_Mx )
      I_Contact( #CNT_pHsMx_E2E4.QD )
      Contact( #PTF_MSal )
   END_RUNG wire#w8
   RUNG wire#powerrail
      I_Contact( #Termico_E1_Tx )
      Contact( #EstadoZona.Rearme_CBx )
   END_RUNG wire#w9
   // the same network as SCL:
   "DB1_SalidasExterioresDeMesa".Mesa[#Mesa].Avanzar_E2E4 := (((((#Mx_ET20 AND #AVTF_MEnt AND (#PTF_MSal OR NOT #CNT_pHsMx_E2E4.QD)) OR ((#Mx_ET21 OR #Mx_ET22) AND (#PTF_MSal OR NOT #CNT_pHsMx_E2E4.QD OR ((#pHsMx_Seg_1 OR #pHsMx_Seg_2) AND #TP2_UP)))) AND ((#CNTSeg_pHsMx_E1E3.CVU <= #V_Bajar_TP_Max) OR (#OK_TP2_DW AND #TP2_DW) OR #TP2_UP) AND #Selec_M2_Entrada) OR ((((#Mx_ET02 OR #Mx_ET60 OR (#Mx_ET61 AND NOT #Simultaneo_Mx)) AND #PTF_MSal AND #TP1_DW) OR (#Mx_ET61 AND #Simultaneo_Mx AND NOT #CNT_pHsMx_E2E4.QD AND #PTF_MSal)) AND #ConfigFB.Final_E2E4 AND #Selec_M4_Salida)) AND #Pos_TR_OK AND #EstadoZona.Marcha_CBx AND NOT #EstadoVI.Error_Mx AND NOT #Error_Tx) OR (NOT #Termico_E1_Tx AND #EstadoZona.Rearme_CBx);
END_REGION

REGION Network 139: SALIDAS - Retroceso E2E4
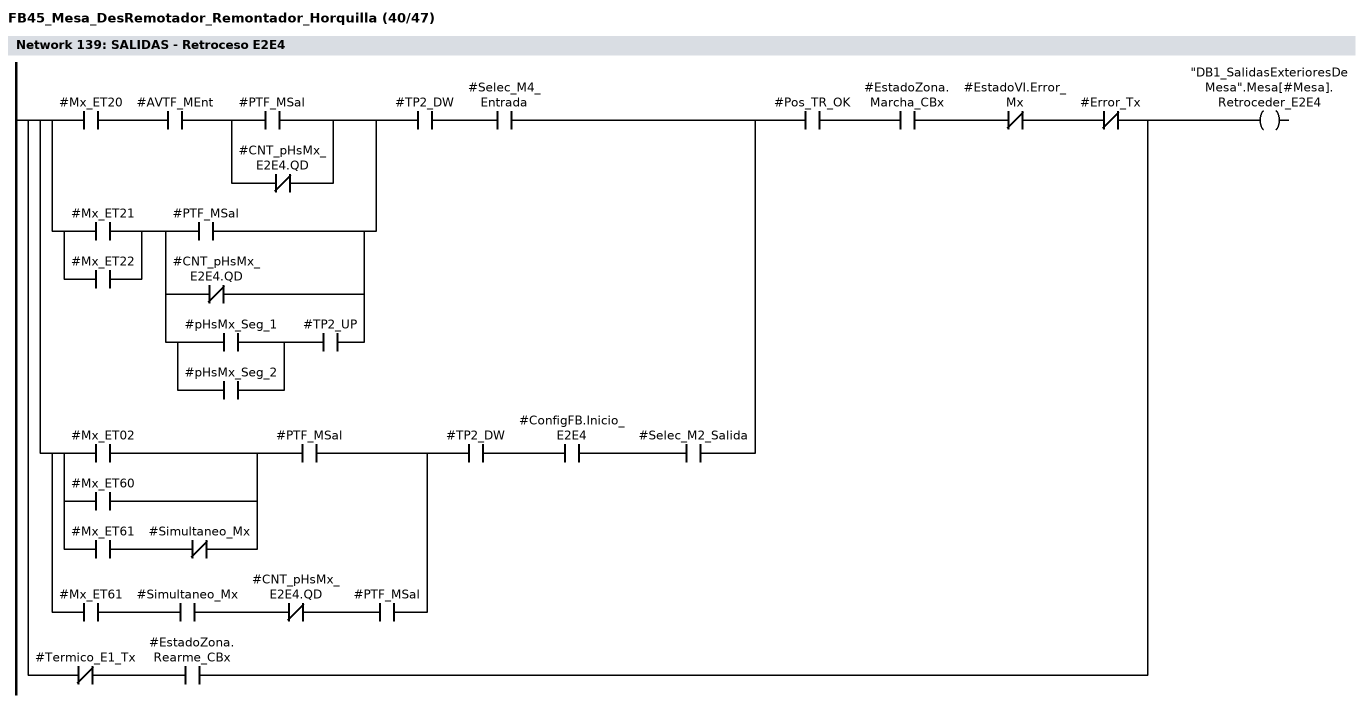
   RUNG wire#powerrail
      Contact( #Mx_ET20 )
      Contact( #AVTF_MEnt )
      wire#w1
      Contact( #PTF_MSal )
      wire#w2
      Contact( #TP2_DW )
      Contact( #Selec_M4_Entrada )
      wire#w5
      Contact( #Pos_TR_OK )
      Contact( #EstadoZona.Marcha_CBx )
      I_Contact( #EstadoVI.Error_Mx )
      I_Contact( #Error_Tx )
      wire#w8
      Coil( "DB1_SalidasExterioresDeMesa".Mesa[#Mesa].Retroceder_E2E4 )
   END_RUNG
   RUNG wire#w1
      I_Contact( #CNT_pHsMx_E2E4.QD )
   END_RUNG wire#w2
   RUNG wire#powerrail
      Contact( #Mx_ET21 )
      wire#w3
      Contact( #PTF_MSal )
   END_RUNG wire#w2
   RUNG wire#powerrail
      Contact( #Mx_ET22 )
   END_RUNG wire#w3
   RUNG wire#w3
      I_Contact( #CNT_pHsMx_E2E4.QD )
   END_RUNG wire#w2
   RUNG wire#w3
      Contact( #pHsMx_Seg_1 )
      wire#w4
      Contact( #TP2_UP )
   END_RUNG wire#w2
   RUNG wire#w3
      Contact( #pHsMx_Seg_2 )
   END_RUNG wire#w4
   RUNG wire#powerrail
      Contact( #Mx_ET02 )
      wire#w6
      Contact( #PTF_MSal )
      wire#w7
      Contact( #TP2_DW )
      Contact( #ConfigFB.Inicio_E2E4 )
      Contact( #Selec_M2_Salida )
   END_RUNG wire#w5
   RUNG wire#powerrail
      Contact( #Mx_ET60 )
   END_RUNG wire#w6
   RUNG wire#powerrail
      Contact( #Mx_ET61 )
      I_Contact( #Simultaneo_Mx )
   END_RUNG wire#w6
   RUNG wire#powerrail
      Contact( #Mx_ET61 )
      Contact( #Simultaneo_Mx )
      I_Contact( #CNT_pHsMx_E2E4.QD )
      Contact( #PTF_MSal )
   END_RUNG wire#w7
   RUNG wire#powerrail
      I_Contact( #Termico_E1_Tx )
      Contact( #EstadoZona.Rearme_CBx )
   END_RUNG wire#w8
   // the same network as SCL:
   "DB1_SalidasExterioresDeMesa".Mesa[#Mesa].Retroceder_E2E4 := (((((#Mx_ET20 AND #AVTF_MEnt AND (#PTF_MSal OR NOT #CNT_pHsMx_E2E4.QD)) OR ((#Mx_ET21 OR #Mx_ET22) AND (#PTF_MSal OR NOT #CNT_pHsMx_E2E4.QD OR ((#pHsMx_Seg_1 OR #pHsMx_Seg_2) AND #TP2_UP)))) AND #TP2_DW AND #Selec_M4_Entrada) OR ((((#Mx_ET02 OR #Mx_ET60 OR (#Mx_ET61 AND NOT #Simultaneo_Mx)) AND #PTF_MSal) OR (#Mx_ET61 AND #Simultaneo_Mx AND NOT #CNT_pHsMx_E2E4.QD AND #PTF_MSal)) AND #TP2_DW AND #ConfigFB.Inicio_E2E4 AND #Selec_M2_Salida)) AND #Pos_TR_OK AND #EstadoZona.Marcha_CBx AND NOT #EstadoVI.Error_Mx AND NOT #Error_Tx) OR (NOT #Termico_E1_Tx AND #EstadoZona.Rearme_CBx);
END_REGION

REGION Network 140: SALIDAS - Parar E2E4
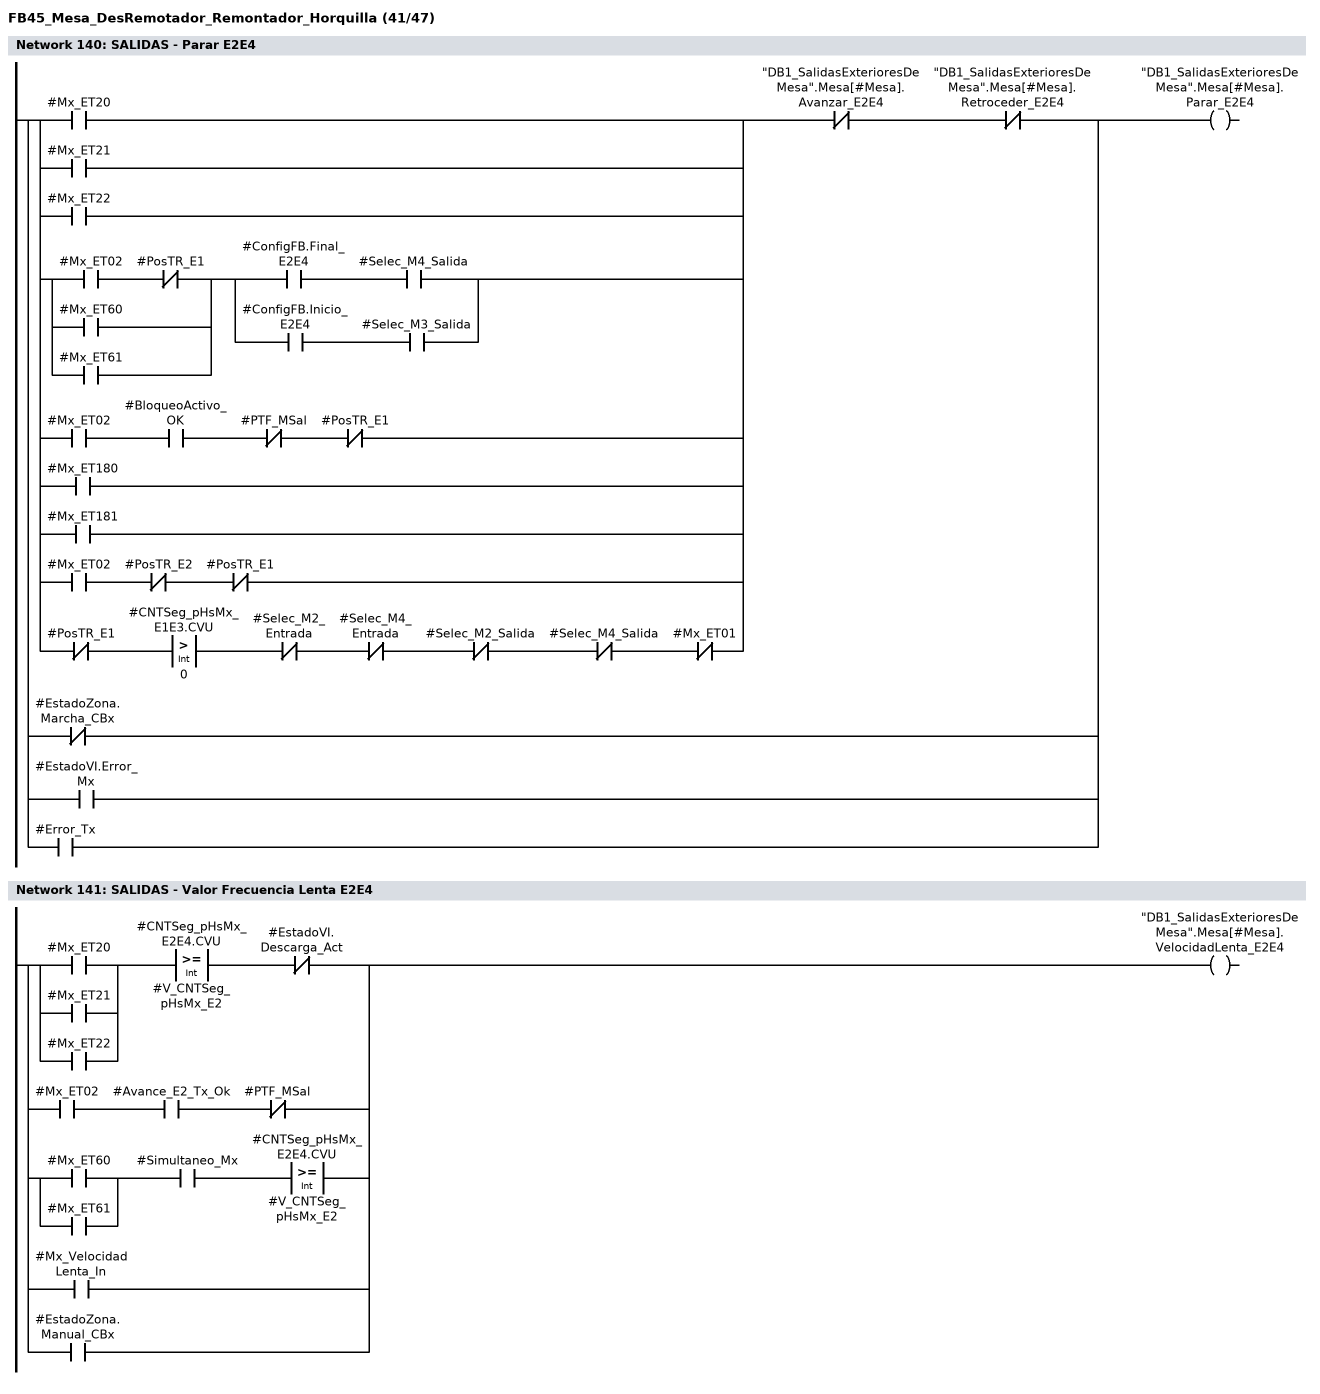
   RUNG wire#powerrail
      Contact( #Mx_ET20 )
      wire#w1
      I_Contact( "DB1_SalidasExterioresDeMesa".Mesa[#Mesa].Avanzar_E2E4 )
      I_Contact( "DB1_SalidasExterioresDeMesa".Mesa[#Mesa].Retroceder_E2E4 )
      wire#w3
      Coil( "DB1_SalidasExterioresDeMesa".Mesa[#Mesa].Parar_E2E4 )
   END_RUNG
   RUNG wire#powerrail
      Contact( #Mx_ET21 )
   END_RUNG wire#w1
   RUNG wire#powerrail
      Contact( #Mx_ET22 )
   END_RUNG wire#w1
   RUNG wire#powerrail
      Contact( #Mx_ET02 )
      I_Contact( #PosTR_E1 )
      wire#w2
      Contact( #ConfigFB.Final_E2E4 )
      Contact( #Selec_M4_Salida )
   END_RUNG wire#w1
   RUNG wire#powerrail
      Contact( #Mx_ET60 )
   END_RUNG wire#w2
   RUNG wire#powerrail
      Contact( #Mx_ET61 )
   END_RUNG wire#w2
   RUNG wire#w2
      Contact( #ConfigFB.Inicio_E2E4 )
      Contact( #Selec_M3_Salida )
   END_RUNG wire#w1
   RUNG wire#powerrail
      Contact( #Mx_ET02 )
      Contact( #BloqueoActivo_OK )
      I_Contact( #PTF_MSal )
      I_Contact( #PosTR_E1 )
   END_RUNG wire#w1
   RUNG wire#powerrail
      Contact( #Mx_ET180 )
   END_RUNG wire#w1
   RUNG wire#powerrail
      Contact( #Mx_ET181 )
   END_RUNG wire#w1
   RUNG wire#powerrail
      Contact( #Mx_ET02 )
      I_Contact( #PosTR_E2 )
      I_Contact( #PosTR_E1 )
   END_RUNG wire#w1
   RUNG wire#powerrail
      I_Contact( #PosTR_E1 )
      { S7_Templates := "SrcType := Int" } GT_Contact(in1 := #CNTSeg_pHsMx_E1E3.CVU, in2 := 0)
      I_Contact( #Selec_M2_Entrada )
      I_Contact( #Selec_M4_Entrada )
      I_Contact( #Selec_M2_Salida )
      I_Contact( #Selec_M4_Salida )
      I_Contact( #Mx_ET01 )
   END_RUNG wire#w1
   RUNG wire#powerrail
      I_Contact( #EstadoZona.Marcha_CBx )
   END_RUNG wire#w3
   RUNG wire#powerrail
      Contact( #EstadoVI.Error_Mx )
   END_RUNG wire#w3
   RUNG wire#powerrail
      Contact( #Error_Tx )
   END_RUNG wire#w3
   // the same network as SCL:
   "DB1_SalidasExterioresDeMesa".Mesa[#Mesa].Parar_E2E4 := ((#Mx_ET20 OR #Mx_ET21 OR #Mx_ET22 OR (((#Mx_ET02 AND NOT #PosTR_E1) OR #Mx_ET60 OR #Mx_ET61) AND ((#ConfigFB.Final_E2E4 AND #Selec_M4_Salida) OR (#ConfigFB.Inicio_E2E4 AND #Selec_M3_Salida))) OR (#Mx_ET02 AND #BloqueoActivo_OK AND NOT #PTF_MSal AND NOT #PosTR_E1) OR #Mx_ET180 OR #Mx_ET181 OR (#Mx_ET02 AND NOT #PosTR_E2 AND NOT #PosTR_E1) OR (NOT #PosTR_E1 AND (#CNTSeg_pHsMx_E1E3.CVU > 0) AND NOT #Selec_M2_Entrada AND NOT #Selec_M4_Entrada AND NOT #Selec_M2_Salida AND NOT #Selec_M4_Salida AND NOT #Mx_ET01)) AND NOT "DB1_SalidasExterioresDeMesa".Mesa[#Mesa].Avanzar_E2E4 AND NOT "DB1_SalidasExterioresDeMesa".Mesa[#Mesa].Retroceder_E2E4) OR NOT #EstadoZona.Marcha_CBx OR #EstadoVI.Error_Mx OR #Error_Tx;
END_REGION

REGION Network 141: SALIDAS - Valor Frecuencia Lenta E2E4
   RUNG wire#powerrail
      Contact( #Mx_ET20 )
      wire#w1
      { S7_Templates := "SrcType := Int" } GE_Contact(in1 := #CNTSeg_pHsMx_E2E4.CVU, in2 := #V_CNTSeg_pHsMx_E2)
      I_Contact( #EstadoVI.Descarga_Act )
      wire#w2
      Coil( "DB1_SalidasExterioresDeMesa".Mesa[#Mesa].VelocidadLenta_E2E4 )
   END_RUNG
   RUNG wire#powerrail
      Contact( #Mx_ET21 )
   END_RUNG wire#w1
   RUNG wire#powerrail
      Contact( #Mx_ET22 )
   END_RUNG wire#w1
   RUNG wire#powerrail
      Contact( #Mx_ET02 )
      Contact( #Avance_E2_Tx_Ok )
      I_Contact( #PTF_MSal )
   END_RUNG wire#w2
   RUNG wire#powerrail
      Contact( #Mx_ET60 )
      wire#w3
      Contact( #Simultaneo_Mx )
      { S7_Templates := "SrcType := Int" } GE_Contact(in1 := #CNTSeg_pHsMx_E2E4.CVU, in2 := #V_CNTSeg_pHsMx_E2)
   END_RUNG wire#w2
   RUNG wire#powerrail
      Contact( #Mx_ET61 )
   END_RUNG wire#w3
   RUNG wire#powerrail
      Contact( #Mx_VelocidadLenta_In )
   END_RUNG wire#w2
   RUNG wire#powerrail
      Contact( #EstadoZona.Manual_CBx )
   END_RUNG wire#w2
   // the same network as SCL:
   "DB1_SalidasExterioresDeMesa".Mesa[#Mesa].VelocidadLenta_E2E4 := ((#Mx_ET20 OR #Mx_ET21 OR #Mx_ET22) AND (#CNTSeg_pHsMx_E2E4.CVU >= #V_CNTSeg_pHsMx_E2) AND NOT #EstadoVI.Descarga_Act) OR (#Mx_ET02 AND #Avance_E2_Tx_Ok AND NOT #PTF_MSal) OR ((#Mx_ET60 OR #Mx_ET61) AND #Simultaneo_Mx AND (#CNTSeg_pHsMx_E2E4.CVU >= #V_CNTSeg_pHsMx_E2)) OR #Mx_VelocidadLenta_In OR #EstadoZona.Manual_CBx;
END_REGION

REGION Network 142: SALIDAS - Ir a posicion E1E3
   // DANI: 2021/06/28. BAJAR EL TOPE DE CADENAS SI HAY S2 O S4 EN ETAPA2 Y TR POS RODILLOS
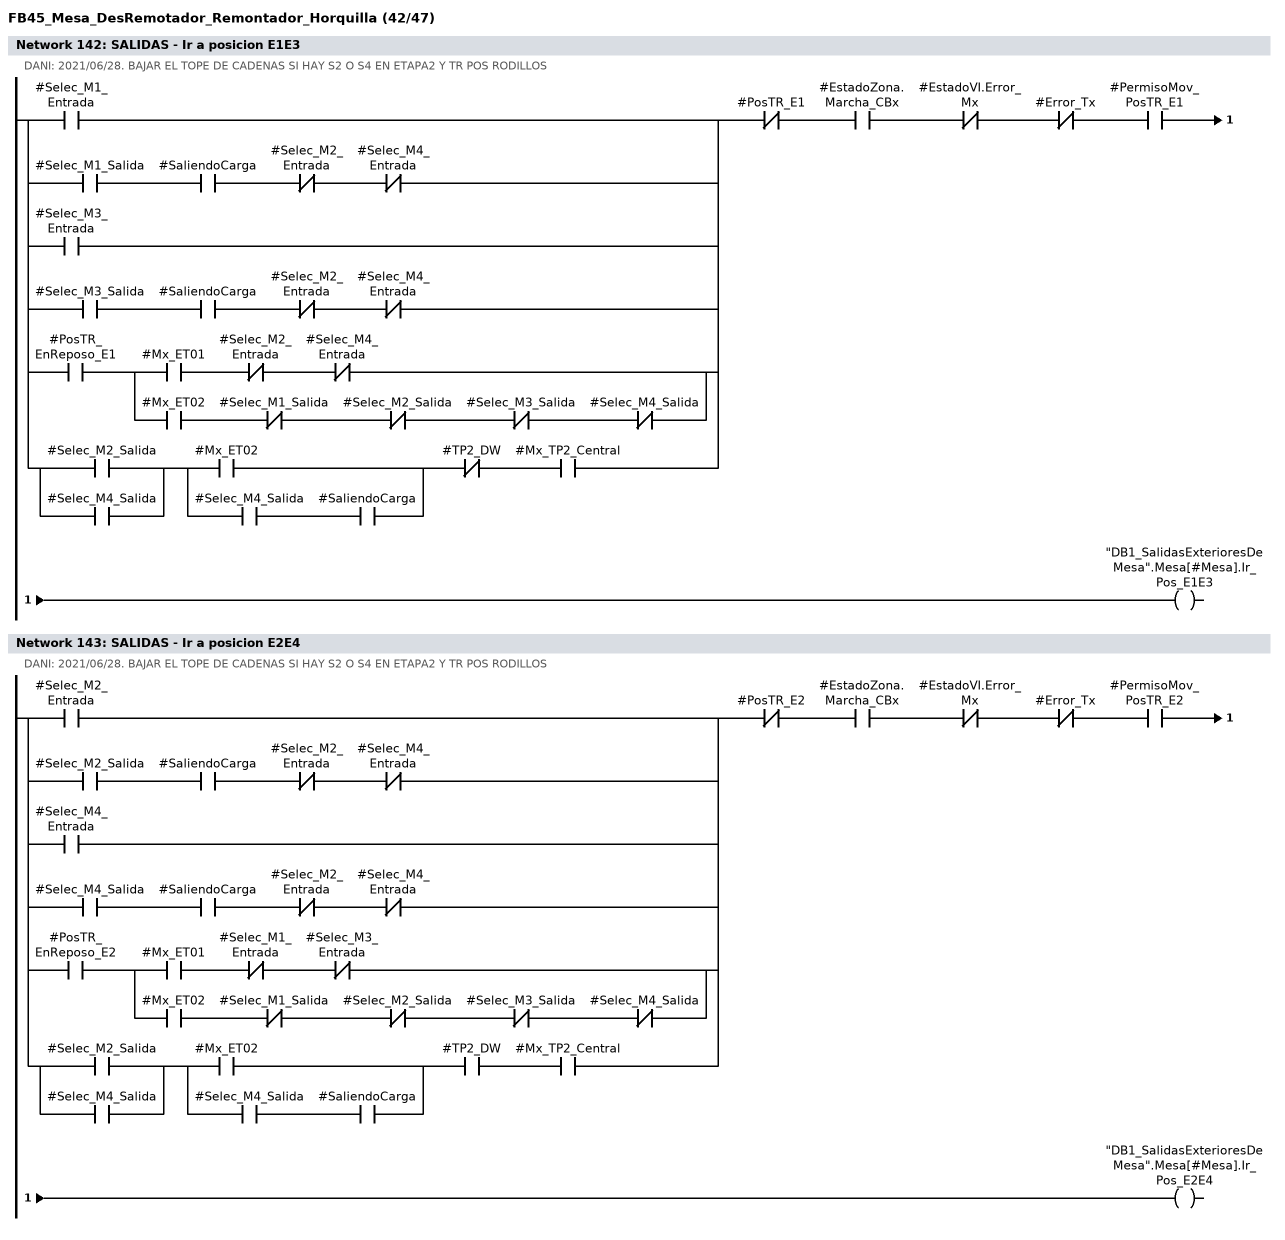
   RUNG wire#powerrail
      Contact( #Selec_M1_Entrada )
      wire#w1
      I_Contact( #PosTR_E1 )
      Contact( #EstadoZona.Marcha_CBx )
      I_Contact( #EstadoVI.Error_Mx )
      I_Contact( #Error_Tx )
      Contact( #PermisoMov_PosTR_E1 )
      Coil( "DB1_SalidasExterioresDeMesa".Mesa[#Mesa].Ir_Pos_E1E3 )
   END_RUNG
   RUNG wire#powerrail
      Contact( #Selec_M1_Salida )
      Contact( #SaliendoCarga )
      I_Contact( #Selec_M2_Entrada )
      I_Contact( #Selec_M4_Entrada )
   END_RUNG wire#w1
   RUNG wire#powerrail
      Contact( #Selec_M3_Entrada )
   END_RUNG wire#w1
   RUNG wire#powerrail
      Contact( #Selec_M3_Salida )
      Contact( #SaliendoCarga )
      I_Contact( #Selec_M2_Entrada )
      I_Contact( #Selec_M4_Entrada )
   END_RUNG wire#w1
   RUNG wire#powerrail
      Contact( #PosTR_EnReposo_E1 )
      wire#w2
      Contact( #Mx_ET01 )
      I_Contact( #Selec_M2_Entrada )
      I_Contact( #Selec_M4_Entrada )
   END_RUNG wire#w1
   RUNG wire#w2
      Contact( #Mx_ET02 )
      I_Contact( #Selec_M1_Salida )
      I_Contact( #Selec_M2_Salida )
      I_Contact( #Selec_M3_Salida )
      I_Contact( #Selec_M4_Salida )
   END_RUNG wire#w1
   RUNG wire#powerrail
      Contact( #Selec_M2_Salida )
      wire#w3
      Contact( #Mx_ET02 )
      wire#w4
      I_Contact( #TP2_DW )
      Contact( #Mx_TP2_Central )
   END_RUNG wire#w1
   RUNG wire#powerrail
      Contact( #Selec_M4_Salida )
   END_RUNG wire#w3
   RUNG wire#w3
      Contact( #Selec_M4_Salida )
      Contact( #SaliendoCarga )
   END_RUNG wire#w4
   // the same network as SCL:
   "DB1_SalidasExterioresDeMesa".Mesa[#Mesa].Ir_Pos_E1E3 := (#Selec_M1_Entrada OR (#Selec_M1_Salida AND #SaliendoCarga AND NOT #Selec_M2_Entrada AND NOT #Selec_M4_Entrada) OR #Selec_M3_Entrada OR (#Selec_M3_Salida AND #SaliendoCarga AND NOT #Selec_M2_Entrada AND NOT #Selec_M4_Entrada) OR (#PosTR_EnReposo_E1 AND ((#Mx_ET01 AND NOT #Selec_M2_Entrada AND NOT #Selec_M4_Entrada) OR (#Mx_ET02 AND NOT #Selec_M1_Salida AND NOT #Selec_M2_Salida AND NOT #Selec_M3_Salida AND NOT #Selec_M4_Salida))) OR ((#Selec_M2_Salida OR #Selec_M4_Salida) AND (#Mx_ET02 OR (#Selec_M4_Salida AND #SaliendoCarga)) AND NOT #TP2_DW AND #Mx_TP2_Central)) AND NOT #PosTR_E1 AND #EstadoZona.Marcha_CBx AND NOT #EstadoVI.Error_Mx AND NOT #Error_Tx AND #PermisoMov_PosTR_E1;
END_REGION

REGION Network 143: SALIDAS - Ir a posicion E2E4
   // DANI: 2021/06/28. BAJAR EL TOPE DE CADENAS SI HAY S2 O S4 EN ETAPA2 Y TR POS RODILLOS
   RUNG wire#powerrail
      Contact( #Selec_M2_Entrada )
      wire#w1
      I_Contact( #PosTR_E2 )
      Contact( #EstadoZona.Marcha_CBx )
      I_Contact( #EstadoVI.Error_Mx )
      I_Contact( #Error_Tx )
      Contact( #PermisoMov_PosTR_E2 )
      Coil( "DB1_SalidasExterioresDeMesa".Mesa[#Mesa].Ir_Pos_E2E4 )
   END_RUNG
   RUNG wire#powerrail
      Contact( #Selec_M2_Salida )
      Contact( #SaliendoCarga )
      I_Contact( #Selec_M2_Entrada )
      I_Contact( #Selec_M4_Entrada )
   END_RUNG wire#w1
   RUNG wire#powerrail
      Contact( #Selec_M4_Entrada )
   END_RUNG wire#w1
   RUNG wire#powerrail
      Contact( #Selec_M4_Salida )
      Contact( #SaliendoCarga )
      I_Contact( #Selec_M2_Entrada )
      I_Contact( #Selec_M4_Entrada )
   END_RUNG wire#w1
   RUNG wire#powerrail
      Contact( #PosTR_EnReposo_E2 )
      wire#w2
      Contact( #Mx_ET01 )
      I_Contact( #Selec_M1_Entrada )
      I_Contact( #Selec_M3_Entrada )
   END_RUNG wire#w1
   RUNG wire#w2
      Contact( #Mx_ET02 )
      I_Contact( #Selec_M1_Salida )
      I_Contact( #Selec_M2_Salida )
      I_Contact( #Selec_M3_Salida )
      I_Contact( #Selec_M4_Salida )
   END_RUNG wire#w1
   RUNG wire#powerrail
      Contact( #Selec_M2_Salida )
      wire#w3
      Contact( #Mx_ET02 )
      wire#w4
      Contact( #TP2_DW )
      Contact( #Mx_TP2_Central )
   END_RUNG wire#w1
   RUNG wire#powerrail
      Contact( #Selec_M4_Salida )
   END_RUNG wire#w3
   RUNG wire#w3
      Contact( #Selec_M4_Salida )
      Contact( #SaliendoCarga )
   END_RUNG wire#w4
   // the same network as SCL:
   "DB1_SalidasExterioresDeMesa".Mesa[#Mesa].Ir_Pos_E2E4 := (#Selec_M2_Entrada OR (#Selec_M2_Salida AND #SaliendoCarga AND NOT #Selec_M2_Entrada AND NOT #Selec_M4_Entrada) OR #Selec_M4_Entrada OR (#Selec_M4_Salida AND #SaliendoCarga AND NOT #Selec_M2_Entrada AND NOT #Selec_M4_Entrada) OR (#PosTR_EnReposo_E2 AND ((#Mx_ET01 AND NOT #Selec_M1_Entrada AND NOT #Selec_M3_Entrada) OR (#Mx_ET02 AND NOT #Selec_M1_Salida AND NOT #Selec_M2_Salida AND NOT #Selec_M3_Salida AND NOT #Selec_M4_Salida))) OR ((#Selec_M2_Salida OR #Selec_M4_Salida) AND (#Mx_ET02 OR (#Selec_M4_Salida AND #SaliendoCarga)) AND #TP2_DW AND #Mx_TP2_Central)) AND NOT #PosTR_E2 AND #EstadoZona.Marcha_CBx AND NOT #EstadoVI.Error_Mx AND NOT #Error_Tx AND #PermisoMov_PosTR_E2;
END_REGION

REGION Network 144: SALIDAS - Bajar TP1
